// TIA Portal V19 export
FUNCTION "INTERLOCK" : Void   // FC8, LAD
{ S7_Optimized_Access := 'TRUE' }
// stored: SetENOAutomatically false
   VAR_TEMP   // added for the SCL form of the ladder/FBD networks
      _w1 : Bool;
      _w2 : Bool;
   END_VAR
BEGIN

REGION Network 1: RO-1 RESET INTERLOCK
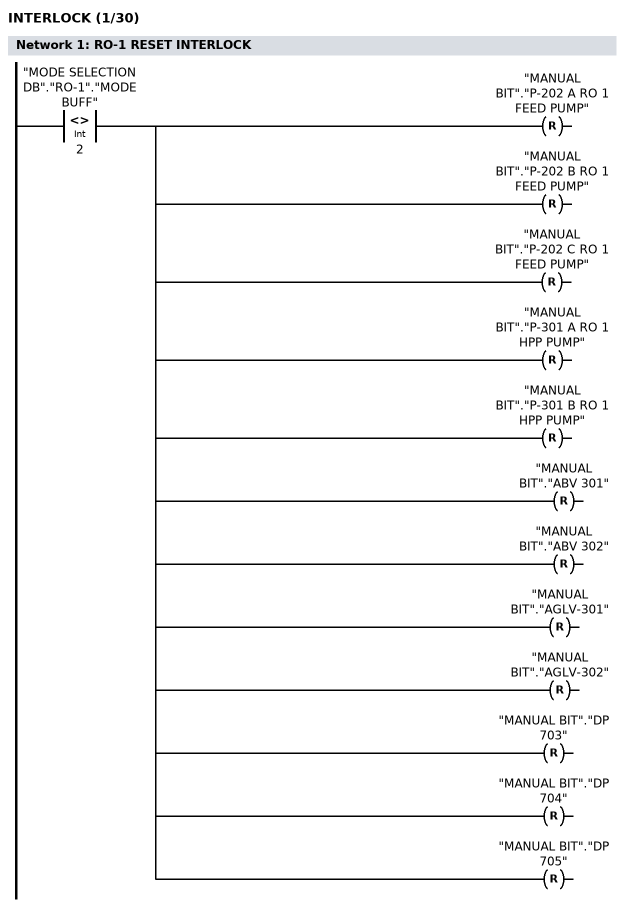
   RUNG wire#powerrail
      { S7_Templates := "SrcType := Int" } NE_Contact(in1 := "MODE SELECTION DB"."RO-1"."MODE BUFF", in2 := 2)
      wire#w1
      R_Coil( "MANUAL BIT"."P-202 A RO 1 FEED PUMP" )
   END_RUNG
   RUNG wire#w1
      R_Coil( "MANUAL BIT"."P-202 B RO 1 FEED PUMP" )
   END_RUNG
   RUNG wire#w1
      R_Coil( "MANUAL BIT"."P-202 C RO 1 FEED PUMP" )
   END_RUNG
   RUNG wire#w1
      R_Coil( "MANUAL BIT"."P-301 A RO 1 HPP PUMP" )
   END_RUNG
   RUNG wire#w1
      R_Coil( "MANUAL BIT"."P-301 B RO 1 HPP PUMP" )
   END_RUNG
   RUNG wire#w1
      R_Coil( "MANUAL BIT"."ABV 301" )
   END_RUNG
   RUNG wire#w1
      R_Coil( "MANUAL BIT"."ABV 302" )
   END_RUNG
   RUNG wire#w1
      R_Coil( "MANUAL BIT"."AGLV-301" )
   END_RUNG
   RUNG wire#w1
      R_Coil( "MANUAL BIT"."AGLV-302" )
   END_RUNG
   RUNG wire#w1
      R_Coil( "MANUAL BIT"."DP 703" )
   END_RUNG
   RUNG wire#w1
      R_Coil( "MANUAL BIT"."DP 704" )
   END_RUNG
   RUNG wire#w1
      R_Coil( "MANUAL BIT"."DP 705" )
   END_RUNG
   // the same network as SCL:
   IF "MODE SELECTION DB"."RO-1"."MODE BUFF" <> 2 THEN
       "MANUAL BIT"."P-202 A RO 1 FEED PUMP" := FALSE;
       "MANUAL BIT"."P-202 B RO 1 FEED PUMP" := FALSE;
       "MANUAL BIT"."P-202 C RO 1 FEED PUMP" := FALSE;
       "MANUAL BIT"."P-301 A RO 1 HPP PUMP" := FALSE;
       "MANUAL BIT"."P-301 B RO 1 HPP PUMP" := FALSE;
       "MANUAL BIT"."ABV 301" := FALSE;
       "MANUAL BIT"."ABV 302" := FALSE;
       "MANUAL BIT"."AGLV-301" := FALSE;
       "MANUAL BIT"."AGLV-302" := FALSE;
       "MANUAL BIT"."DP 703" := FALSE;
       "MANUAL BIT"."DP 704" := FALSE;
       "MANUAL BIT"."DP 705" := FALSE;
   END_IF;
END_REGION

REGION Network 2: RO-2 RESET INTERLOCK
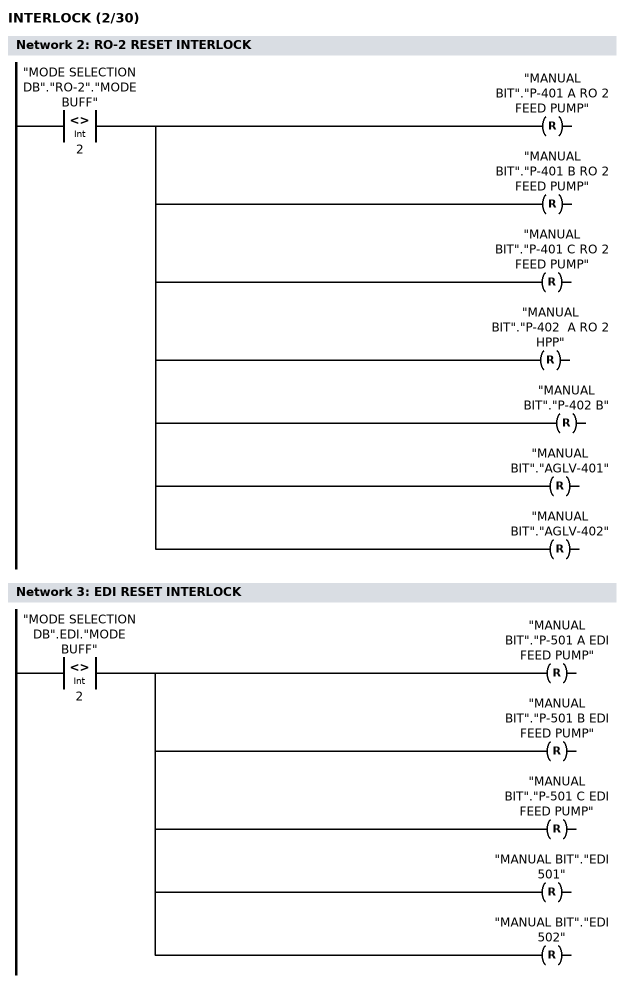
   RUNG wire#powerrail
      { S7_Templates := "SrcType := Int" } NE_Contact(in1 := "MODE SELECTION DB"."RO-2"."MODE BUFF", in2 := 2)
      wire#w1
      R_Coil( "MANUAL BIT"."P-401 A RO 2 FEED PUMP" )
   END_RUNG
   RUNG wire#w1
      R_Coil( "MANUAL BIT"."P-401 B RO 2 FEED PUMP" )
   END_RUNG
   RUNG wire#w1
      R_Coil( "MANUAL BIT"."P-401 C RO 2 FEED PUMP" )
   END_RUNG
   RUNG wire#w1
      R_Coil( "MANUAL BIT"."P-402  A RO 2 HPP" )
   END_RUNG
   RUNG wire#w1
      R_Coil( "MANUAL BIT"."P-402 B" )
   END_RUNG
   RUNG wire#w1
      R_Coil( "MANUAL BIT"."AGLV-401" )
   END_RUNG
   RUNG wire#w1
      R_Coil( "MANUAL BIT"."AGLV-402" )
   END_RUNG
   // the same network as SCL:
   IF "MODE SELECTION DB"."RO-2"."MODE BUFF" <> 2 THEN
       "MANUAL BIT"."P-401 A RO 2 FEED PUMP" := FALSE;
       "MANUAL BIT"."P-401 B RO 2 FEED PUMP" := FALSE;
       "MANUAL BIT"."P-401 C RO 2 FEED PUMP" := FALSE;
       "MANUAL BIT"."P-402  A RO 2 HPP" := FALSE;
       "MANUAL BIT"."P-402 B" := FALSE;
       "MANUAL BIT"."AGLV-401" := FALSE;
       "MANUAL BIT"."AGLV-402" := FALSE;
   END_IF;
END_REGION

REGION Network 3: EDI RESET INTERLOCK
   RUNG wire#powerrail
      { S7_Templates := "SrcType := Int" } NE_Contact(in1 := "MODE SELECTION DB".EDI."MODE BUFF", in2 := 2)
      wire#w1
      R_Coil( "MANUAL BIT"."P-501 A EDI FEED PUMP" )
   END_RUNG
   RUNG wire#w1
      R_Coil( "MANUAL BIT"."P-501 B EDI FEED PUMP" )
   END_RUNG
   RUNG wire#w1
      R_Coil( "MANUAL BIT"."P-501 C EDI FEED PUMP" )
   END_RUNG
   RUNG wire#w1
      R_Coil( "MANUAL BIT"."EDI 501" )
   END_RUNG
   RUNG wire#w1
      R_Coil( "MANUAL BIT"."EDI 502" )
   END_RUNG
   // the same network as SCL:
   IF "MODE SELECTION DB".EDI."MODE BUFF" <> 2 THEN
       "MANUAL BIT"."P-501 A EDI FEED PUMP" := FALSE;
       "MANUAL BIT"."P-501 B EDI FEED PUMP" := FALSE;
       "MANUAL BIT"."P-501 C EDI FEED PUMP" := FALSE;
       "MANUAL BIT"."EDI 501" := FALSE;
       "MANUAL BIT"."EDI 502" := FALSE;
   END_IF;
END_REGION

REGION Network 4: SELECTION PUMP INTERLOCK_
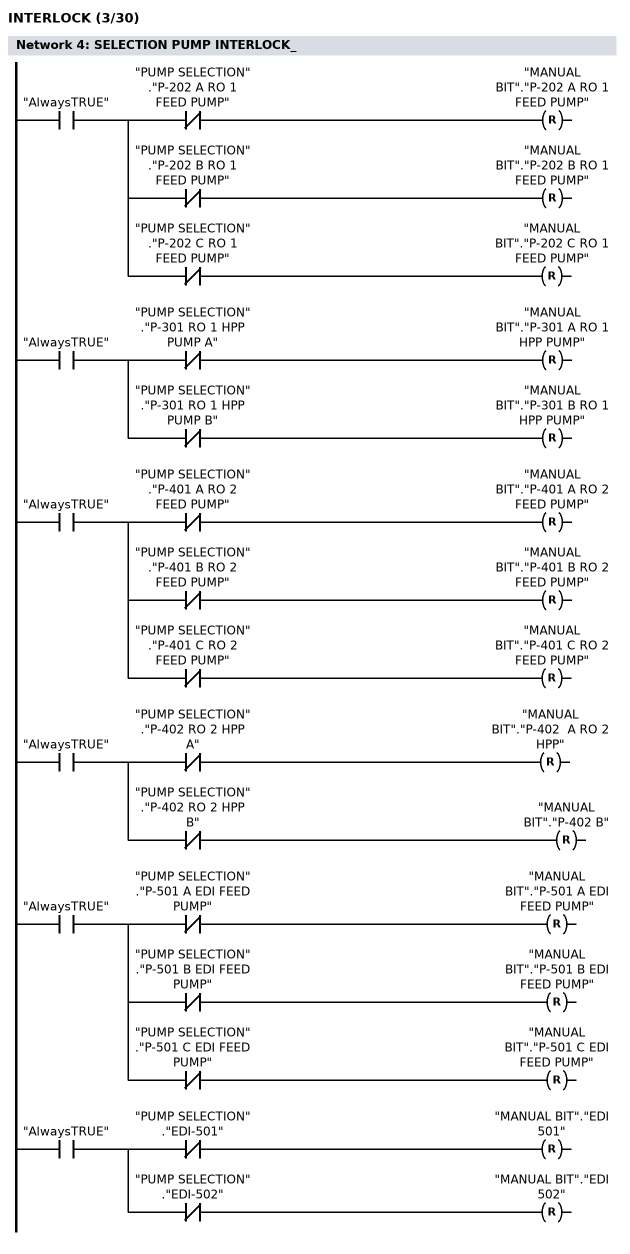
   RUNG wire#powerrail
      Contact( "AlwaysTRUE" )
      wire#w1
      I_Contact( "PUMP SELECTION"."P-202 A RO 1 FEED PUMP" )
      R_Coil( "MANUAL BIT"."P-202 A RO 1 FEED PUMP" )
   END_RUNG
   RUNG wire#w1
      I_Contact( "PUMP SELECTION"."P-202 B RO 1 FEED PUMP" )
      R_Coil( "MANUAL BIT"."P-202 B RO 1 FEED PUMP" )
   END_RUNG
   RUNG wire#w1
      I_Contact( "PUMP SELECTION"."P-202 C RO 1 FEED PUMP" )
      R_Coil( "MANUAL BIT"."P-202 C RO 1 FEED PUMP" )
   END_RUNG
   RUNG wire#powerrail
      Contact( "AlwaysTRUE" )
      wire#w2
      I_Contact( "PUMP SELECTION"."P-301 RO 1 HPP PUMP A" )
      R_Coil( "MANUAL BIT"."P-301 A RO 1 HPP PUMP" )
   END_RUNG
   RUNG wire#w2
      I_Contact( "PUMP SELECTION"."P-301 RO 1 HPP PUMP B" )
      R_Coil( "MANUAL BIT"."P-301 B RO 1 HPP PUMP" )
   END_RUNG
   RUNG wire#powerrail
      Contact( "AlwaysTRUE" )
      wire#w3
      I_Contact( "PUMP SELECTION"."P-401 A RO 2 FEED PUMP" )
      R_Coil( "MANUAL BIT"."P-401 A RO 2 FEED PUMP" )
   END_RUNG
   RUNG wire#w3
      I_Contact( "PUMP SELECTION"."P-401 B RO 2 FEED PUMP" )
      R_Coil( "MANUAL BIT"."P-401 B RO 2 FEED PUMP" )
   END_RUNG
   RUNG wire#w3
      I_Contact( "PUMP SELECTION"."P-401 C RO 2 FEED PUMP" )
      R_Coil( "MANUAL BIT"."P-401 C RO 2 FEED PUMP" )
   END_RUNG
   RUNG wire#powerrail
      Contact( "AlwaysTRUE" )
      wire#w4
      I_Contact( "PUMP SELECTION"."P-402 RO 2 HPP A" )
      R_Coil( "MANUAL BIT"."P-402  A RO 2 HPP" )
   END_RUNG
   RUNG wire#w4
      I_Contact( "PUMP SELECTION"."P-402 RO 2 HPP B" )
      R_Coil( "MANUAL BIT"."P-402 B" )
   END_RUNG
   RUNG wire#powerrail
      Contact( "AlwaysTRUE" )
      wire#w5
      I_Contact( "PUMP SELECTION"."P-501 A EDI FEED PUMP" )
      R_Coil( "MANUAL BIT"."P-501 A EDI FEED PUMP" )
   END_RUNG
   RUNG wire#w5
      I_Contact( "PUMP SELECTION"."P-501 B EDI FEED PUMP" )
      R_Coil( "MANUAL BIT"."P-501 B EDI FEED PUMP" )
   END_RUNG
   RUNG wire#w5
      I_Contact( "PUMP SELECTION"."P-501 C EDI FEED PUMP" )
      R_Coil( "MANUAL BIT"."P-501 C EDI FEED PUMP" )
   END_RUNG
   RUNG wire#powerrail
      Contact( "AlwaysTRUE" )
      wire#w6
      I_Contact( "PUMP SELECTION"."EDI-501" )
      R_Coil( "MANUAL BIT"."EDI 501" )
   END_RUNG
   RUNG wire#w6
      I_Contact( "PUMP SELECTION"."EDI-502" )
      R_Coil( "MANUAL BIT"."EDI 502" )
   END_RUNG
   // the same network as SCL:
   IF "AlwaysTRUE" AND NOT "PUMP SELECTION"."P-202 A RO 1 FEED PUMP" THEN
       "MANUAL BIT"."P-202 A RO 1 FEED PUMP" := FALSE;
   END_IF;
   IF "AlwaysTRUE" AND NOT "PUMP SELECTION"."P-202 B RO 1 FEED PUMP" THEN
       "MANUAL BIT"."P-202 B RO 1 FEED PUMP" := FALSE;
   END_IF;
   IF "AlwaysTRUE" AND NOT "PUMP SELECTION"."P-202 C RO 1 FEED PUMP" THEN
       "MANUAL BIT"."P-202 C RO 1 FEED PUMP" := FALSE;
   END_IF;
   IF "AlwaysTRUE" AND NOT "PUMP SELECTION"."P-301 RO 1 HPP PUMP A" THEN
       "MANUAL BIT"."P-301 A RO 1 HPP PUMP" := FALSE;
   END_IF;
   IF "AlwaysTRUE" AND NOT "PUMP SELECTION"."P-301 RO 1 HPP PUMP B" THEN
       "MANUAL BIT"."P-301 B RO 1 HPP PUMP" := FALSE;
   END_IF;
   IF "AlwaysTRUE" AND NOT "PUMP SELECTION"."P-401 A RO 2 FEED PUMP" THEN
       "MANUAL BIT"."P-401 A RO 2 FEED PUMP" := FALSE;
   END_IF;
   IF "AlwaysTRUE" AND NOT "PUMP SELECTION"."P-401 B RO 2 FEED PUMP" THEN
       "MANUAL BIT"."P-401 B RO 2 FEED PUMP" := FALSE;
   END_IF;
   IF "AlwaysTRUE" AND NOT "PUMP SELECTION"."P-401 C RO 2 FEED PUMP" THEN
       "MANUAL BIT"."P-401 C RO 2 FEED PUMP" := FALSE;
   END_IF;
   IF "AlwaysTRUE" AND NOT "PUMP SELECTION"."P-402 RO 2 HPP A" THEN
       "MANUAL BIT"."P-402  A RO 2 HPP" := FALSE;
   END_IF;
   IF "AlwaysTRUE" AND NOT "PUMP SELECTION"."P-402 RO 2 HPP B" THEN "MANUAL BIT"."P-402 B" := FALSE; END_IF;
   IF "AlwaysTRUE" AND NOT "PUMP SELECTION"."P-501 A EDI FEED PUMP" THEN
       "MANUAL BIT"."P-501 A EDI FEED PUMP" := FALSE;
   END_IF;
   IF "AlwaysTRUE" AND NOT "PUMP SELECTION"."P-501 B EDI FEED PUMP" THEN
       "MANUAL BIT"."P-501 B EDI FEED PUMP" := FALSE;
   END_IF;
   IF "AlwaysTRUE" AND NOT "PUMP SELECTION"."P-501 C EDI FEED PUMP" THEN
       "MANUAL BIT"."P-501 C EDI FEED PUMP" := FALSE;
   END_IF;
   IF "AlwaysTRUE" AND NOT "PUMP SELECTION"."EDI-501" THEN "MANUAL BIT"."EDI 501" := FALSE; END_IF;
   IF "AlwaysTRUE" AND NOT "PUMP SELECTION"."EDI-502" THEN "MANUAL BIT"."EDI 502" := FALSE; END_IF;
END_REGION

REGION Network 10: AUTO INTERLOCK FOR RO-1 ///////////////////////////////////////////////////////
END_REGION

REGION Network 11: CEB1 AND CEB2 SYSTEM IN RUNNING AFTER RO SYSTEM HOLD
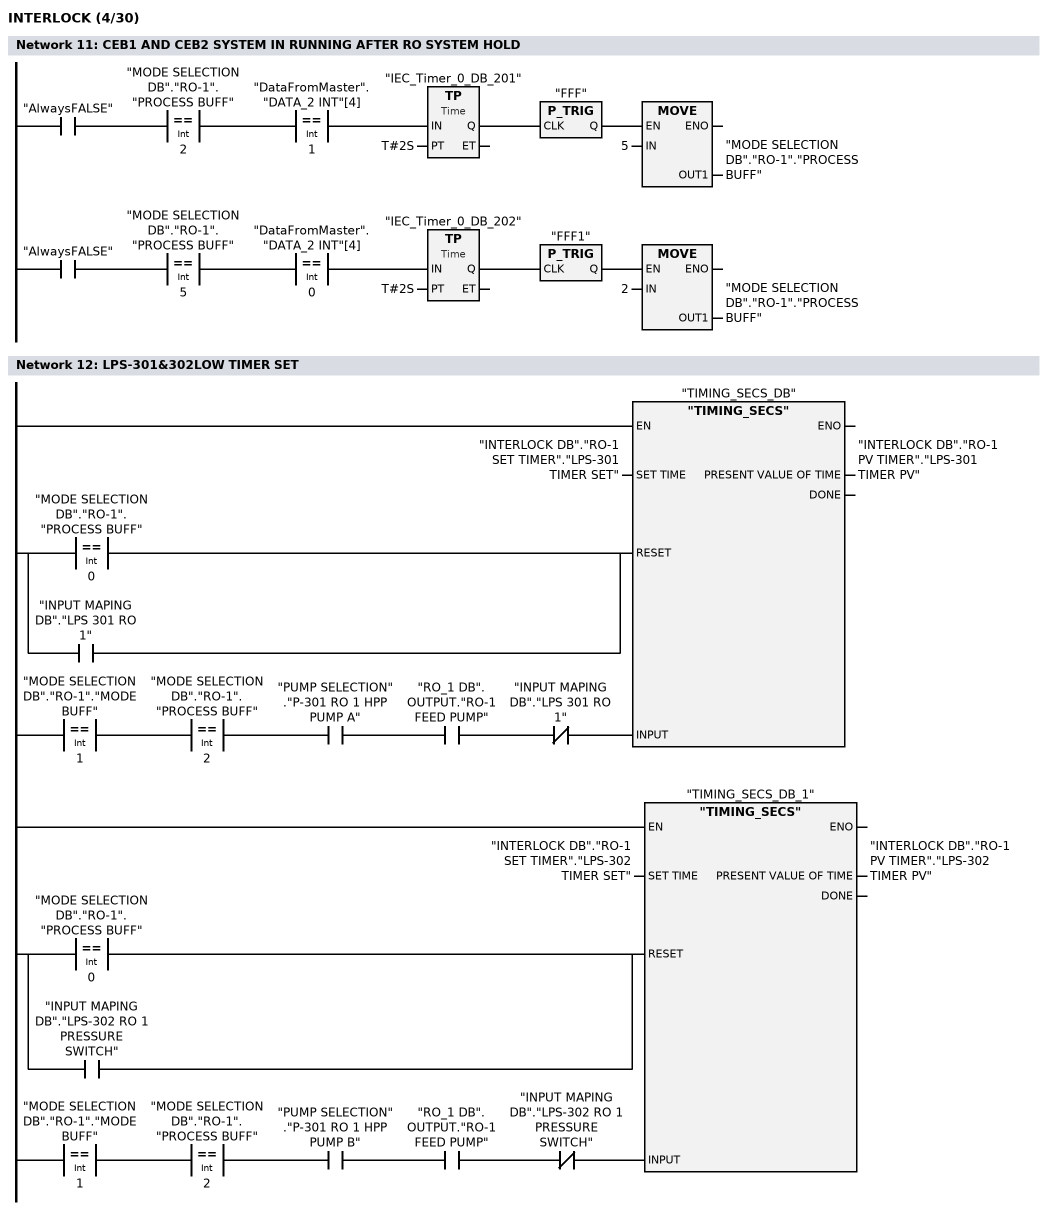
   RUNG wire#powerrail
      Contact( "AlwaysFALSE" )
      { S7_Templates := "SrcType := Int" } EQ_Contact(in1 := "MODE SELECTION DB"."RO-1"."PROCESS BUFF", in2 := 2)
      { S7_Templates := "SrcType := Int" } EQ_Contact(in1 := "DataFromMaster"."DATA_2 INT"[4], in2 := 1)
      { S7_Templates := "time_type := Time" } "IEC_Timer_0_DB_201".TP(pt := T#2S, et =>)
      P_Trig( "FFF" )
      Move(in := 5, out1 => "MODE SELECTION DB"."RO-1"."PROCESS BUFF")
   END_RUNG
   RUNG wire#powerrail
      Contact( "AlwaysFALSE" )
      { S7_Templates := "SrcType := Int" } EQ_Contact(in1 := "MODE SELECTION DB"."RO-1"."PROCESS BUFF", in2 := 5)
      { S7_Templates := "SrcType := Int" } EQ_Contact(in1 := "DataFromMaster"."DATA_2 INT"[4], in2 := 0)
      { S7_Templates := "time_type := Time" } "IEC_Timer_0_DB_202".TP(pt := T#2S, et =>)
      P_Trig( "FFF1" )
      Move(in := 2, out1 => "MODE SELECTION DB"."RO-1"."PROCESS BUFF")
   END_RUNG
   // the same network as SCL:
   "IEC_Timer_0_DB_201".TP(IN := "AlwaysFALSE" AND ("MODE SELECTION DB"."RO-1"."PROCESS BUFF" = 2) AND ("DataFromMaster"."DATA_2 INT"[4] = 1),
                           PT := T#2S);
   #_w1 := "IEC_Timer_0_DB_201".Q AND NOT "FFF";   // rising edge
   "FFF" := "IEC_Timer_0_DB_201".Q;
   IF #_w1 THEN "MODE SELECTION DB"."RO-1"."PROCESS BUFF" := 5; END_IF;
   "IEC_Timer_0_DB_202".TP(IN := "AlwaysFALSE" AND ("MODE SELECTION DB"."RO-1"."PROCESS BUFF" = 5) AND ("DataFromMaster"."DATA_2 INT"[4] = 0),
                           PT := T#2S);
   #_w2 := "IEC_Timer_0_DB_202".Q AND NOT "FFF1";   // rising edge
   "FFF1" := "IEC_Timer_0_DB_202".Q;
   IF #_w2 THEN "MODE SELECTION DB"."RO-1"."PROCESS BUFF" := 2; END_IF;
END_REGION

REGION Network 12: LPS-301&302LOW TIMER SET
   RUNG wire#powerrail
      "TIMING_SECS_DB"(RESET := wire#w1, INPUT := wire#w2, "SET TIME" := "INTERLOCK DB"."RO-1 SET TIMER"."LPS-301 TIMER SET", "PRESENT VALUE OF TIME" => "INTERLOCK DB"."RO-1 PV TIMER"."LPS-301 TIMER PV", DONE =>)
   END_RUNG
   RUNG wire#powerrail
      { S7_Templates := "SrcType := Int" } EQ_Contact(in1 := "MODE SELECTION DB"."RO-1"."PROCESS BUFF", in2 := 0)
   END_RUNG wire#w1
   RUNG wire#powerrail
      Contact( "INPUT MAPING DB"."LPS 301 RO 1" )
   END_RUNG wire#w1
   RUNG wire#powerrail
      { S7_Templates := "SrcType := Int" } EQ_Contact(in1 := "MODE SELECTION DB"."RO-1"."MODE BUFF", in2 := 1)
      { S7_Templates := "SrcType := Int" } EQ_Contact(in1 := "MODE SELECTION DB"."RO-1"."PROCESS BUFF", in2 := 2)
      Contact( "PUMP SELECTION"."P-301 RO 1 HPP PUMP A" )
      Contact( "RO_1 DB".OUTPUT."RO-1 FEED PUMP" )
      I_Contact( "INPUT MAPING DB"."LPS 301 RO 1" )
   END_RUNG wire#w2
   RUNG wire#powerrail
      "TIMING_SECS_DB_1"(RESET := wire#w3, INPUT := wire#w4, "SET TIME" := "INTERLOCK DB"."RO-1 SET TIMER"."LPS-302 TIMER SET", "PRESENT VALUE OF TIME" => "INTERLOCK DB"."RO-1 PV TIMER"."LPS-302 TIMER PV", DONE =>)
   END_RUNG
   RUNG wire#powerrail
      { S7_Templates := "SrcType := Int" } EQ_Contact(in1 := "MODE SELECTION DB"."RO-1"."PROCESS BUFF", in2 := 0)
   END_RUNG wire#w3
   RUNG wire#powerrail
      Contact( "INPUT MAPING DB"."LPS-302 RO 1 PRESSURE SWITCH" )
   END_RUNG wire#w3
   RUNG wire#powerrail
      { S7_Templates := "SrcType := Int" } EQ_Contact(in1 := "MODE SELECTION DB"."RO-1"."MODE BUFF", in2 := 1)
      { S7_Templates := "SrcType := Int" } EQ_Contact(in1 := "MODE SELECTION DB"."RO-1"."PROCESS BUFF", in2 := 2)
      Contact( "PUMP SELECTION"."P-301 RO 1 HPP PUMP B" )
      Contact( "RO_1 DB".OUTPUT."RO-1 FEED PUMP" )
      I_Contact( "INPUT MAPING DB"."LPS-302 RO 1 PRESSURE SWITCH" )
   END_RUNG wire#w4
   // the same network as SCL:
   "TIMING_SECS_DB"("SET TIME" := "INTERLOCK DB"."RO-1 SET TIMER"."LPS-301 TIMER SET",   // "TIMING_SECS"
                    RESET := ("MODE SELECTION DB"."RO-1"."PROCESS BUFF" = 0) OR "INPUT MAPING DB"."LPS 301 RO 1",
                    INPUT := ("MODE SELECTION DB"."RO-1"."MODE BUFF" = 1) AND ("MODE SELECTION DB"."RO-1"."PROCESS BUFF" = 2) AND "PUMP SELECTION"."P-301 RO 1 HPP PUMP A" AND "RO_1 DB".OUTPUT."RO-1 FEED PUMP" AND NOT "INPUT MAPING DB"."LPS 301 RO 1",
                    "PRESENT VALUE OF TIME" => "INTERLOCK DB"."RO-1 PV TIMER"."LPS-301 TIMER PV");
   "TIMING_SECS_DB_1"("SET TIME" := "INTERLOCK DB"."RO-1 SET TIMER"."LPS-302 TIMER SET",   // "TIMING_SECS"
                      RESET := ("MODE SELECTION DB"."RO-1"."PROCESS BUFF" = 0) OR "INPUT MAPING DB"."LPS-302 RO 1 PRESSURE SWITCH",
                      INPUT := ("MODE SELECTION DB"."RO-1"."MODE BUFF" = 1) AND ("MODE SELECTION DB"."RO-1"."PROCESS BUFF" = 2) AND "PUMP SELECTION"."P-301 RO 1 HPP PUMP B" AND "RO_1 DB".OUTPUT."RO-1 FEED PUMP" AND NOT "INPUT MAPING DB"."LPS-302 RO 1 PRESSURE SWITCH",
                      "PRESENT VALUE OF TIME" => "INTERLOCK DB"."RO-1 PV TIMER"."LPS-302 TIMER PV");
END_REGION

REGION Network 13: HPS-301 &302
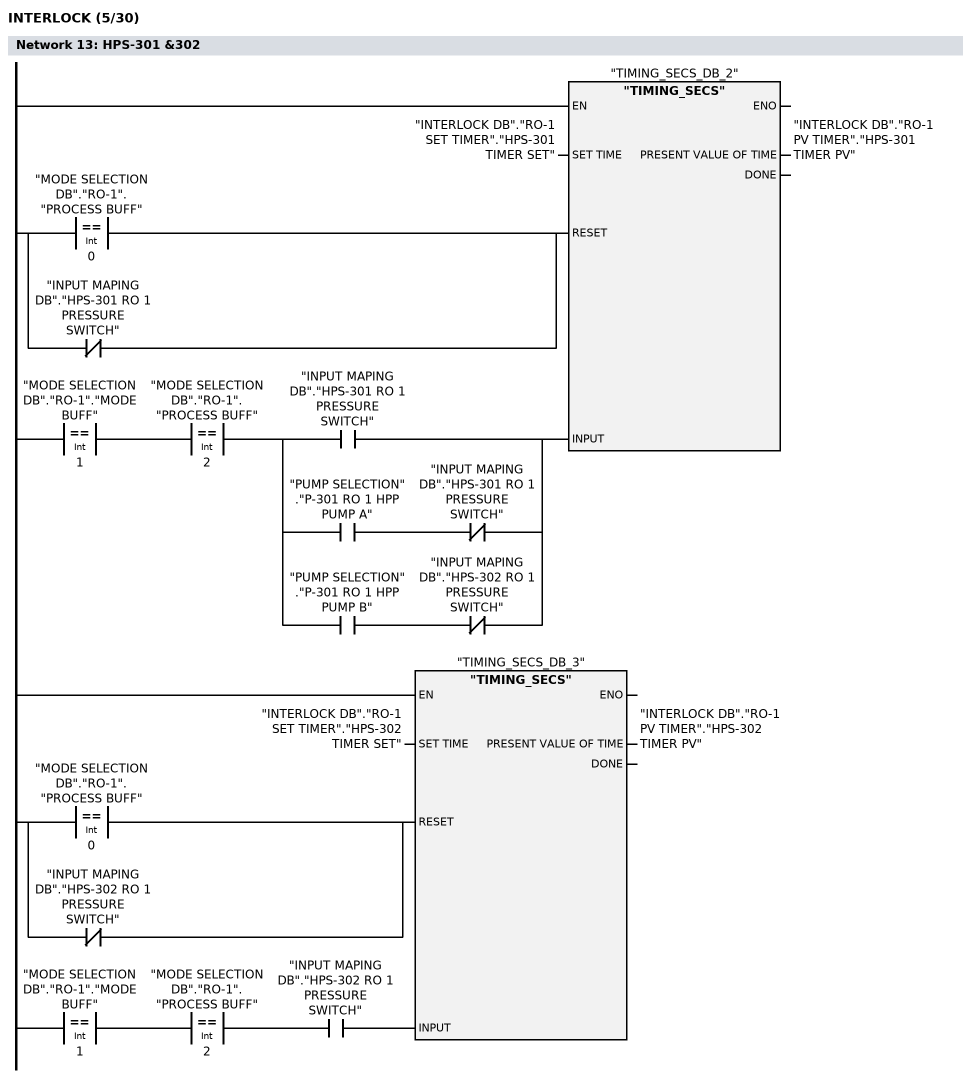
   RUNG wire#powerrail
      "TIMING_SECS_DB_2"(RESET := wire#w1, INPUT := wire#w3, "SET TIME" := "INTERLOCK DB"."RO-1 SET TIMER"."HPS-301 TIMER SET", "PRESENT VALUE OF TIME" => "INTERLOCK DB"."RO-1 PV TIMER"."HPS-301 TIMER PV", DONE =>)
   END_RUNG
   RUNG wire#powerrail
      { S7_Templates := "SrcType := Int" } EQ_Contact(in1 := "MODE SELECTION DB"."RO-1"."PROCESS BUFF", in2 := 0)
   END_RUNG wire#w1
   RUNG wire#powerrail
      I_Contact( "INPUT MAPING DB"."HPS-301 RO 1 PRESSURE SWITCH" )
   END_RUNG wire#w1
   RUNG wire#powerrail
      { S7_Templates := "SrcType := Int" } EQ_Contact(in1 := "MODE SELECTION DB"."RO-1"."MODE BUFF", in2 := 1)
      { S7_Templates := "SrcType := Int" } EQ_Contact(in1 := "MODE SELECTION DB"."RO-1"."PROCESS BUFF", in2 := 2)
      wire#w2
      Contact( "INPUT MAPING DB"."HPS-301 RO 1 PRESSURE SWITCH" )
   END_RUNG wire#w3
   RUNG wire#w2
      Contact( "PUMP SELECTION"."P-301 RO 1 HPP PUMP A" )
      I_Contact( "INPUT MAPING DB"."HPS-301 RO 1 PRESSURE SWITCH" )
   END_RUNG wire#w3
   RUNG wire#w2
      Contact( "PUMP SELECTION"."P-301 RO 1 HPP PUMP B" )
      I_Contact( "INPUT MAPING DB"."HPS-302 RO 1 PRESSURE SWITCH" )
   END_RUNG wire#w3
   RUNG wire#powerrail
      "TIMING_SECS_DB_3"(RESET := wire#w4, INPUT := wire#w5, "SET TIME" := "INTERLOCK DB"."RO-1 SET TIMER"."HPS-302 TIMER SET", "PRESENT VALUE OF TIME" => "INTERLOCK DB"."RO-1 PV TIMER"."HPS-302 TIMER PV", DONE =>)
   END_RUNG
   RUNG wire#powerrail
      { S7_Templates := "SrcType := Int" } EQ_Contact(in1 := "MODE SELECTION DB"."RO-1"."PROCESS BUFF", in2 := 0)
   END_RUNG wire#w4
   RUNG wire#powerrail
      I_Contact( "INPUT MAPING DB"."HPS-302 RO 1 PRESSURE SWITCH" )
   END_RUNG wire#w4
   RUNG wire#powerrail
      { S7_Templates := "SrcType := Int" } EQ_Contact(in1 := "MODE SELECTION DB"."RO-1"."MODE BUFF", in2 := 1)
      { S7_Templates := "SrcType := Int" } EQ_Contact(in1 := "MODE SELECTION DB"."RO-1"."PROCESS BUFF", in2 := 2)
      Contact( "INPUT MAPING DB"."HPS-302 RO 1 PRESSURE SWITCH" )
   END_RUNG wire#w5
   // the same network as SCL:
   "TIMING_SECS_DB_2"("SET TIME" := "INTERLOCK DB"."RO-1 SET TIMER"."HPS-301 TIMER SET",   // "TIMING_SECS"
                      RESET := ("MODE SELECTION DB"."RO-1"."PROCESS BUFF" = 0) OR NOT "INPUT MAPING DB"."HPS-301 RO 1 PRESSURE SWITCH",
                      INPUT := ("MODE SELECTION DB"."RO-1"."MODE BUFF" = 1) AND ("MODE SELECTION DB"."RO-1"."PROCESS BUFF" = 2) AND ("INPUT MAPING DB"."HPS-301 RO 1 PRESSURE SWITCH" OR ("PUMP SELECTION"."P-301 RO 1 HPP PUMP A" AND NOT "INPUT MAPING DB"."HPS-301 RO 1 PRESSURE SWITCH") OR ("PUMP SELECTION"."P-301 RO 1 HPP PUMP B" AND NOT "INPUT MAPING DB"."HPS-302 RO 1 PRESSURE SWITCH")),
                      "PRESENT VALUE OF TIME" => "INTERLOCK DB"."RO-1 PV TIMER"."HPS-301 TIMER PV");
   "TIMING_SECS_DB_3"("SET TIME" := "INTERLOCK DB"."RO-1 SET TIMER"."HPS-302 TIMER SET",   // "TIMING_SECS"
                      RESET := ("MODE SELECTION DB"."RO-1"."PROCESS BUFF" = 0) OR NOT "INPUT MAPING DB"."HPS-302 RO 1 PRESSURE SWITCH",
                      INPUT := ("MODE SELECTION DB"."RO-1"."MODE BUFF" = 1) AND ("MODE SELECTION DB"."RO-1"."PROCESS BUFF" = 2) AND "INPUT MAPING DB"."HPS-302 RO 1 PRESSURE SWITCH",
                      "PRESENT VALUE OF TIME" => "INTERLOCK DB"."RO-1 PV TIMER"."HPS-302 TIMER PV");
END_REGION

REGION Network 14: pH-301 HIGH/ LOW
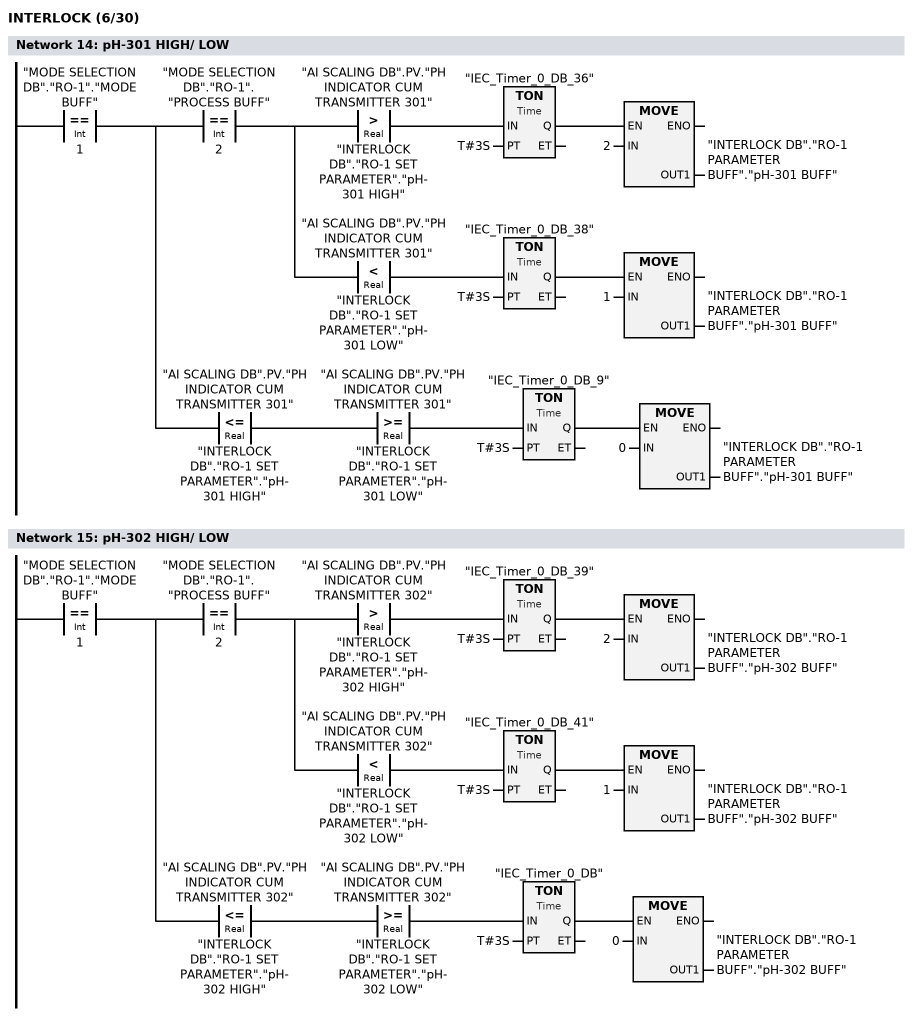
   RUNG wire#powerrail
      { S7_Templates := "SrcType := Int" } EQ_Contact(in1 := "MODE SELECTION DB"."RO-1"."MODE BUFF", in2 := 1)
      wire#w1
      { S7_Templates := "SrcType := Int" } EQ_Contact(in1 := "MODE SELECTION DB"."RO-1"."PROCESS BUFF", in2 := 2)
      wire#w2
      { S7_Templates := "SrcType := Real" } GT_Contact(in1 := "AI SCALING DB".PV."PH INDICATOR CUM TRANSMITTER 301", in2 := "INTERLOCK DB"."RO-1 SET PARAMETER"."pH-301 HIGH")
      { S7_Templates := "time_type := Time" } "IEC_Timer_0_DB_36".TON(pt := T#3S, et =>)
      Move(in := 2, out1 => "INTERLOCK DB"."RO-1 PARAMETER BUFF"."pH-301 BUFF")
   END_RUNG
   RUNG wire#w2
      { S7_Templates := "SrcType := Real" } LT_Contact(in1 := "AI SCALING DB".PV."PH INDICATOR CUM TRANSMITTER 301", in2 := "INTERLOCK DB"."RO-1 SET PARAMETER"."pH-301 LOW")
      { S7_Templates := "time_type := Time" } "IEC_Timer_0_DB_38".TON(pt := T#3S, et =>)
      Move(in := 1, out1 => "INTERLOCK DB"."RO-1 PARAMETER BUFF"."pH-301 BUFF")
   END_RUNG
   RUNG wire#w1
      { S7_Templates := "SrcType := Real" } LE_Contact(in1 := "AI SCALING DB".PV."PH INDICATOR CUM TRANSMITTER 301", in2 := "INTERLOCK DB"."RO-1 SET PARAMETER"."pH-301 HIGH")
      { S7_Templates := "SrcType := Real" } GE_Contact(in1 := "AI SCALING DB".PV."PH INDICATOR CUM TRANSMITTER 301", in2 := "INTERLOCK DB"."RO-1 SET PARAMETER"."pH-301 LOW")
      { S7_Templates := "time_type := Time" } "IEC_Timer_0_DB_9".TON(pt := T#3S, et =>)
      Move(in := 0, out1 => "INTERLOCK DB"."RO-1 PARAMETER BUFF"."pH-301 BUFF")
   END_RUNG
   // the same network as SCL:
   #_w1 := "MODE SELECTION DB"."RO-1"."MODE BUFF" = 1;
   #_w2 := #_w1 AND ("MODE SELECTION DB"."RO-1"."PROCESS BUFF" = 2);
   "IEC_Timer_0_DB_36".TON(IN := #_w2 AND ("AI SCALING DB".PV."PH INDICATOR CUM TRANSMITTER 301" > "INTERLOCK DB"."RO-1 SET PARAMETER"."pH-301 HIGH"),
                           PT := T#3S);
   IF "IEC_Timer_0_DB_36".Q THEN "INTERLOCK DB"."RO-1 PARAMETER BUFF"."pH-301 BUFF" := 2; END_IF;
   "IEC_Timer_0_DB_38".TON(IN := #_w2 AND ("AI SCALING DB".PV."PH INDICATOR CUM TRANSMITTER 301" < "INTERLOCK DB"."RO-1 SET PARAMETER"."pH-301 LOW"),
                           PT := T#3S);
   IF "IEC_Timer_0_DB_38".Q THEN "INTERLOCK DB"."RO-1 PARAMETER BUFF"."pH-301 BUFF" := 1; END_IF;
   "IEC_Timer_0_DB_9".TON(IN := #_w1 AND ("AI SCALING DB".PV."PH INDICATOR CUM TRANSMITTER 301" <= "INTERLOCK DB"."RO-1 SET PARAMETER"."pH-301 HIGH") AND ("AI SCALING DB".PV."PH INDICATOR CUM TRANSMITTER 301" >= "INTERLOCK DB"."RO-1 SET PARAMETER"."pH-301 LOW"),
                          PT := T#3S);
   IF "IEC_Timer_0_DB_9".Q THEN "INTERLOCK DB"."RO-1 PARAMETER BUFF"."pH-301 BUFF" := 0; END_IF;
END_REGION

REGION Network 15: pH-302 HIGH/ LOW
   RUNG wire#powerrail
      { S7_Templates := "SrcType := Int" } EQ_Contact(in1 := "MODE SELECTION DB"."RO-1"."MODE BUFF", in2 := 1)
      wire#w1
      { S7_Templates := "SrcType := Int" } EQ_Contact(in1 := "MODE SELECTION DB"."RO-1"."PROCESS BUFF", in2 := 2)
      wire#w2
      { S7_Templates := "SrcType := Real" } GT_Contact(in1 := "AI SCALING DB".PV."PH INDICATOR CUM TRANSMITTER 302", in2 := "INTERLOCK DB"."RO-1 SET PARAMETER"."pH-302 HIGH")
      { S7_Templates := "time_type := Time" } "IEC_Timer_0_DB_39".TON(pt := T#3S, et =>)
      Move(in := 2, out1 => "INTERLOCK DB"."RO-1 PARAMETER BUFF"."pH-302 BUFF")
   END_RUNG
   RUNG wire#w2
      { S7_Templates := "SrcType := Real" } LT_Contact(in1 := "AI SCALING DB".PV."PH INDICATOR CUM TRANSMITTER 302", in2 := "INTERLOCK DB"."RO-1 SET PARAMETER"."pH-302 LOW")
      { S7_Templates := "time_type := Time" } "IEC_Timer_0_DB_41".TON(pt := T#3S, et =>)
      Move(in := 1, out1 => "INTERLOCK DB"."RO-1 PARAMETER BUFF"."pH-302 BUFF")
   END_RUNG
   RUNG wire#w1
      { S7_Templates := "SrcType := Real" } LE_Contact(in1 := "AI SCALING DB".PV."PH INDICATOR CUM TRANSMITTER 302", in2 := "INTERLOCK DB"."RO-1 SET PARAMETER"."pH-302 HIGH")
      { S7_Templates := "SrcType := Real" } GE_Contact(in1 := "AI SCALING DB".PV."PH INDICATOR CUM TRANSMITTER 302", in2 := "INTERLOCK DB"."RO-1 SET PARAMETER"."pH-302 LOW")
      { S7_Templates := "time_type := Time" } "IEC_Timer_0_DB".TON(pt := T#3S, et =>)
      Move(in := 0, out1 => "INTERLOCK DB"."RO-1 PARAMETER BUFF"."pH-302 BUFF")
   END_RUNG
   // the same network as SCL:
   #_w1 := "MODE SELECTION DB"."RO-1"."MODE BUFF" = 1;
   #_w2 := #_w1 AND ("MODE SELECTION DB"."RO-1"."PROCESS BUFF" = 2);
   "IEC_Timer_0_DB_39".TON(IN := #_w2 AND ("AI SCALING DB".PV."PH INDICATOR CUM TRANSMITTER 302" > "INTERLOCK DB"."RO-1 SET PARAMETER"."pH-302 HIGH"),
                           PT := T#3S);
   IF "IEC_Timer_0_DB_39".Q THEN "INTERLOCK DB"."RO-1 PARAMETER BUFF"."pH-302 BUFF" := 2; END_IF;
   "IEC_Timer_0_DB_41".TON(IN := #_w2 AND ("AI SCALING DB".PV."PH INDICATOR CUM TRANSMITTER 302" < "INTERLOCK DB"."RO-1 SET PARAMETER"."pH-302 LOW"),
                           PT := T#3S);
   IF "IEC_Timer_0_DB_41".Q THEN "INTERLOCK DB"."RO-1 PARAMETER BUFF"."pH-302 BUFF" := 1; END_IF;
   "IEC_Timer_0_DB".TON(IN := #_w1 AND ("AI SCALING DB".PV."PH INDICATOR CUM TRANSMITTER 302" <= "INTERLOCK DB"."RO-1 SET PARAMETER"."pH-302 HIGH") AND ("AI SCALING DB".PV."PH INDICATOR CUM TRANSMITTER 302" >= "INTERLOCK DB"."RO-1 SET PARAMETER"."pH-302 LOW"),
                        PT := T#3S);
   IF "IEC_Timer_0_DB".Q THEN "INTERLOCK DB"."RO-1 PARAMETER BUFF"."pH-302 BUFF" := 0; END_IF;
END_REGION

REGION Network 16: CT-301 HIGH
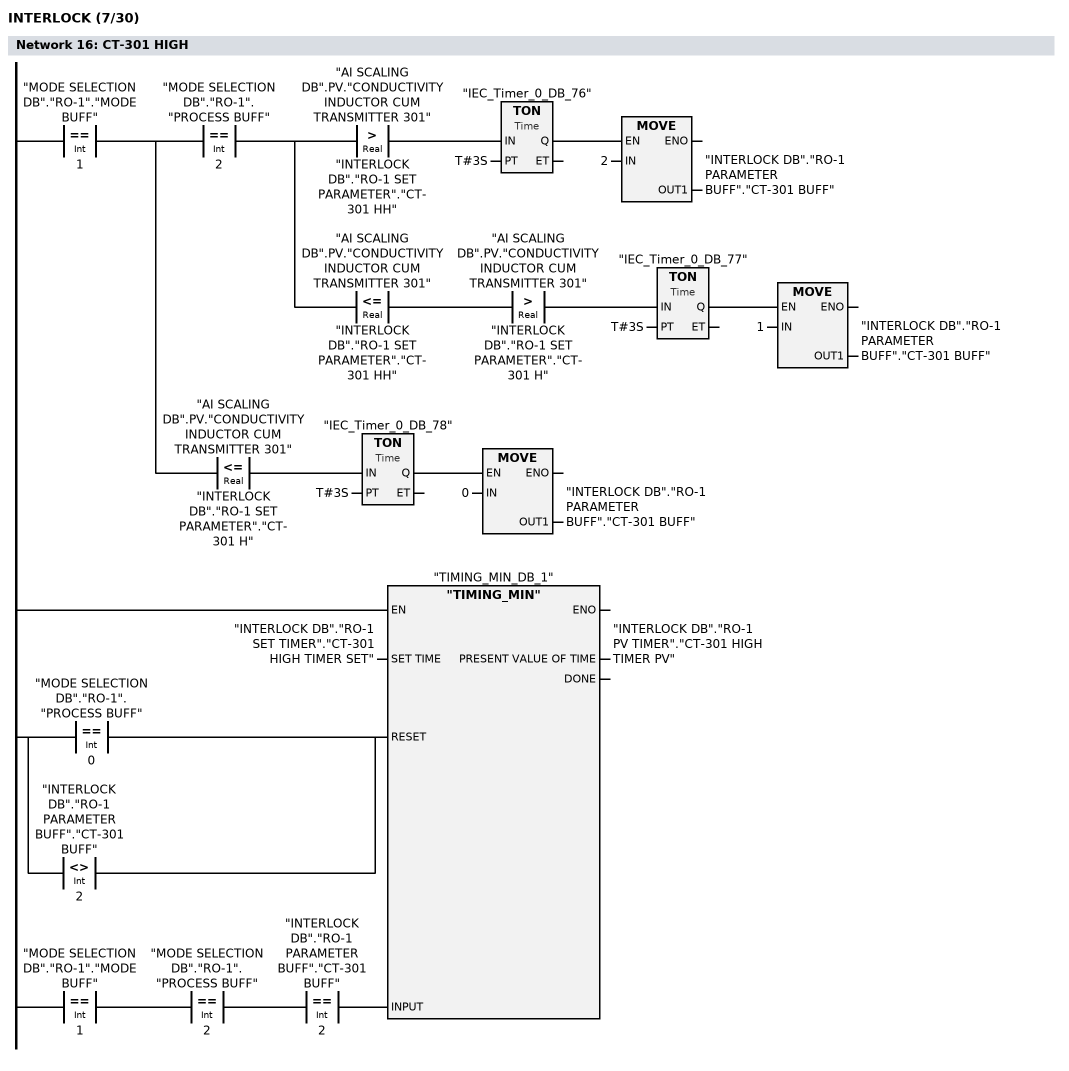
   RUNG wire#powerrail
      { S7_Templates := "SrcType := Int" } EQ_Contact(in1 := "MODE SELECTION DB"."RO-1"."MODE BUFF", in2 := 1)
      wire#w1
      { S7_Templates := "SrcType := Int" } EQ_Contact(in1 := "MODE SELECTION DB"."RO-1"."PROCESS BUFF", in2 := 2)
      wire#w2
      { S7_Templates := "SrcType := Real" } GT_Contact(in1 := "AI SCALING DB".PV."CONDUCTIVITY INDUCTOR CUM TRANSMITTER 301", in2 := "INTERLOCK DB"."RO-1 SET PARAMETER"."CT-301 HH")
      { S7_Templates := "time_type := Time" } "IEC_Timer_0_DB_76".TON(pt := T#3S, et =>)
      Move(in := 2, out1 => "INTERLOCK DB"."RO-1 PARAMETER BUFF"."CT-301 BUFF")
   END_RUNG
   RUNG wire#w2
      { S7_Templates := "SrcType := Real" } LE_Contact(in1 := "AI SCALING DB".PV."CONDUCTIVITY INDUCTOR CUM TRANSMITTER 301", in2 := "INTERLOCK DB"."RO-1 SET PARAMETER"."CT-301 HH")
      { S7_Templates := "SrcType := Real" } GT_Contact(in1 := "AI SCALING DB".PV."CONDUCTIVITY INDUCTOR CUM TRANSMITTER 301", in2 := "INTERLOCK DB"."RO-1 SET PARAMETER"."CT-301 H")
      { S7_Templates := "time_type := Time" } "IEC_Timer_0_DB_77".TON(pt := T#3S, et =>)
      Move(in := 1, out1 => "INTERLOCK DB"."RO-1 PARAMETER BUFF"."CT-301 BUFF")
   END_RUNG
   RUNG wire#w1
      { S7_Templates := "SrcType := Real" } LE_Contact(in1 := "AI SCALING DB".PV."CONDUCTIVITY INDUCTOR CUM TRANSMITTER 301", in2 := "INTERLOCK DB"."RO-1 SET PARAMETER"."CT-301 H")
      { S7_Templates := "time_type := Time" } "IEC_Timer_0_DB_78".TON(pt := T#3S, et =>)
      Move(in := 0, out1 => "INTERLOCK DB"."RO-1 PARAMETER BUFF"."CT-301 BUFF")
   END_RUNG
   RUNG wire#powerrail
      "TIMING_MIN_DB_1"(RESET := wire#w3, INPUT := wire#w4, "SET TIME" := "INTERLOCK DB"."RO-1 SET TIMER"."CT-301 HIGH TIMER SET", "PRESENT VALUE OF TIME" => "INTERLOCK DB"."RO-1 PV TIMER"."CT-301 HIGH TIMER PV", DONE =>)
   END_RUNG
   RUNG wire#powerrail
      { S7_Templates := "SrcType := Int" } EQ_Contact(in1 := "MODE SELECTION DB"."RO-1"."PROCESS BUFF", in2 := 0)
   END_RUNG wire#w3
   RUNG wire#powerrail
      { S7_Templates := "SrcType := Int" } NE_Contact(in1 := "INTERLOCK DB"."RO-1 PARAMETER BUFF"."CT-301 BUFF", in2 := 2)
   END_RUNG wire#w3
   RUNG wire#powerrail
      { S7_Templates := "SrcType := Int" } EQ_Contact(in1 := "MODE SELECTION DB"."RO-1"."MODE BUFF", in2 := 1)
      { S7_Templates := "SrcType := Int" } EQ_Contact(in1 := "MODE SELECTION DB"."RO-1"."PROCESS BUFF", in2 := 2)
      { S7_Templates := "SrcType := Int" } EQ_Contact(in1 := "INTERLOCK DB"."RO-1 PARAMETER BUFF"."CT-301 BUFF", in2 := 2)
   END_RUNG wire#w4
   // the same network as SCL:
   #_w1 := "MODE SELECTION DB"."RO-1"."MODE BUFF" = 1;
   #_w2 := #_w1 AND ("MODE SELECTION DB"."RO-1"."PROCESS BUFF" = 2);
   "IEC_Timer_0_DB_76".TON(IN := #_w2 AND ("AI SCALING DB".PV."CONDUCTIVITY INDUCTOR CUM TRANSMITTER 301" > "INTERLOCK DB"."RO-1 SET PARAMETER"."CT-301 HH"),
                           PT := T#3S);
   IF "IEC_Timer_0_DB_76".Q THEN "INTERLOCK DB"."RO-1 PARAMETER BUFF"."CT-301 BUFF" := 2; END_IF;
   "IEC_Timer_0_DB_77".TON(IN := #_w2 AND ("AI SCALING DB".PV."CONDUCTIVITY INDUCTOR CUM TRANSMITTER 301" <= "INTERLOCK DB"."RO-1 SET PARAMETER"."CT-301 HH") AND ("AI SCALING DB".PV."CONDUCTIVITY INDUCTOR CUM TRANSMITTER 301" > "INTERLOCK DB"."RO-1 SET PARAMETER"."CT-301 H"),
                           PT := T#3S);
   IF "IEC_Timer_0_DB_77".Q THEN "INTERLOCK DB"."RO-1 PARAMETER BUFF"."CT-301 BUFF" := 1; END_IF;
   "IEC_Timer_0_DB_78".TON(IN := #_w1 AND ("AI SCALING DB".PV."CONDUCTIVITY INDUCTOR CUM TRANSMITTER 301" <= "INTERLOCK DB"."RO-1 SET PARAMETER"."CT-301 H"),
                           PT := T#3S);
   IF "IEC_Timer_0_DB_78".Q THEN "INTERLOCK DB"."RO-1 PARAMETER BUFF"."CT-301 BUFF" := 0; END_IF;
   "TIMING_MIN_DB_1"("SET TIME" := "INTERLOCK DB"."RO-1 SET TIMER"."CT-301 HIGH TIMER SET",   // "TIMING_MIN"
                     RESET := ("MODE SELECTION DB"."RO-1"."PROCESS BUFF" = 0) OR ("INTERLOCK DB"."RO-1 PARAMETER BUFF"."CT-301 BUFF" <> 2),
                     INPUT := ("MODE SELECTION DB"."RO-1"."MODE BUFF" = 1) AND ("MODE SELECTION DB"."RO-1"."PROCESS BUFF" = 2) AND ("INTERLOCK DB"."RO-1 PARAMETER BUFF"."CT-301 BUFF" = 2),
                     "PRESENT VALUE OF TIME" => "INTERLOCK DB"."RO-1 PV TIMER"."CT-301 HIGH TIMER PV");
END_REGION

REGION Network 17: CT-302 HIGH
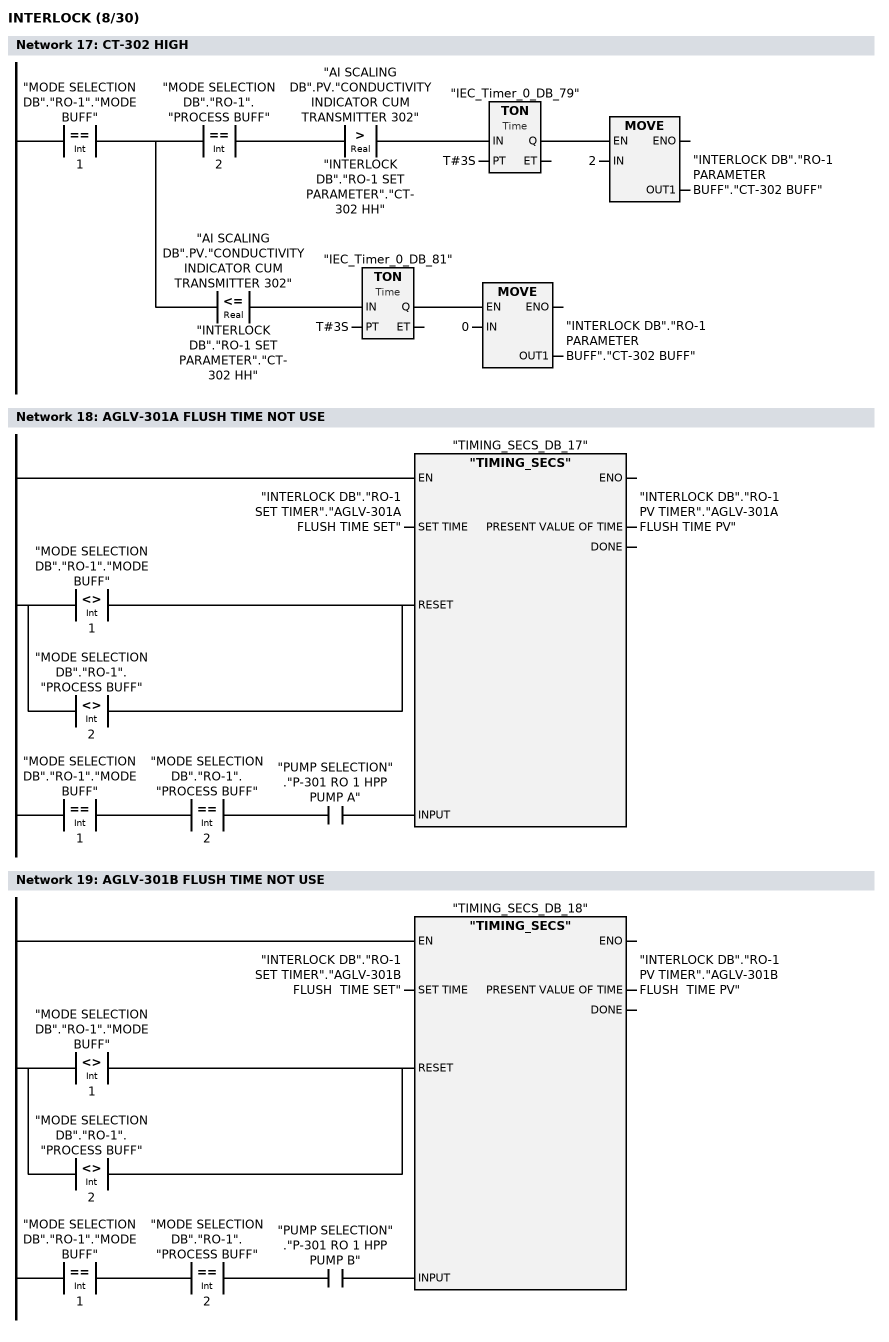
   RUNG wire#powerrail
      { S7_Templates := "SrcType := Int" } EQ_Contact(in1 := "MODE SELECTION DB"."RO-1"."MODE BUFF", in2 := 1)
      wire#w1
      { S7_Templates := "SrcType := Int" } EQ_Contact(in1 := "MODE SELECTION DB"."RO-1"."PROCESS BUFF", in2 := 2)
      { S7_Templates := "SrcType := Real" } GT_Contact(in1 := "AI SCALING DB".PV."CONDUCTIVITY INDICATOR CUM TRANSMITTER 302", in2 := "INTERLOCK DB"."RO-1 SET PARAMETER"."CT-302 HH")
      { S7_Templates := "time_type := Time" } "IEC_Timer_0_DB_79".TON(pt := T#3S, et =>)
      Move(in := 2, out1 => "INTERLOCK DB"."RO-1 PARAMETER BUFF"."CT-302 BUFF")
   END_RUNG
   RUNG wire#w1
      { S7_Templates := "SrcType := Real" } LE_Contact(in1 := "AI SCALING DB".PV."CONDUCTIVITY INDICATOR CUM TRANSMITTER 302", in2 := "INTERLOCK DB"."RO-1 SET PARAMETER"."CT-302 HH")
      { S7_Templates := "time_type := Time" } "IEC_Timer_0_DB_81".TON(pt := T#3S, et =>)
      Move(in := 0, out1 => "INTERLOCK DB"."RO-1 PARAMETER BUFF"."CT-302 BUFF")
   END_RUNG
   // the same network as SCL:
   #_w1 := "MODE SELECTION DB"."RO-1"."MODE BUFF" = 1;
   "IEC_Timer_0_DB_79".TON(IN := #_w1 AND ("MODE SELECTION DB"."RO-1"."PROCESS BUFF" = 2) AND ("AI SCALING DB".PV."CONDUCTIVITY INDICATOR CUM TRANSMITTER 302" > "INTERLOCK DB"."RO-1 SET PARAMETER"."CT-302 HH"),
                           PT := T#3S);
   IF "IEC_Timer_0_DB_79".Q THEN "INTERLOCK DB"."RO-1 PARAMETER BUFF"."CT-302 BUFF" := 2; END_IF;
   "IEC_Timer_0_DB_81".TON(IN := #_w1 AND ("AI SCALING DB".PV."CONDUCTIVITY INDICATOR CUM TRANSMITTER 302" <= "INTERLOCK DB"."RO-1 SET PARAMETER"."CT-302 HH"),
                           PT := T#3S);
   IF "IEC_Timer_0_DB_81".Q THEN "INTERLOCK DB"."RO-1 PARAMETER BUFF"."CT-302 BUFF" := 0; END_IF;
END_REGION

REGION Network 18: AGLV-301A FLUSH TIME NOT USE
   RUNG wire#powerrail
      "TIMING_SECS_DB_17"(RESET := wire#w1, INPUT := wire#w2, "SET TIME" := "INTERLOCK DB"."RO-1 SET TIMER"."AGLV-301A FLUSH TIME SET", "PRESENT VALUE OF TIME" => "INTERLOCK DB"."RO-1 PV TIMER"."AGLV-301A FLUSH TIME PV", DONE =>)
   END_RUNG
   RUNG wire#powerrail
      { S7_Templates := "SrcType := Int" } NE_Contact(in1 := "MODE SELECTION DB"."RO-1"."MODE BUFF", in2 := 1)
   END_RUNG wire#w1
   RUNG wire#powerrail
      { S7_Templates := "SrcType := Int" } NE_Contact(in1 := "MODE SELECTION DB"."RO-1"."PROCESS BUFF", in2 := 2)
   END_RUNG wire#w1
   RUNG wire#powerrail
      { S7_Templates := "SrcType := Int" } EQ_Contact(in1 := "MODE SELECTION DB"."RO-1"."MODE BUFF", in2 := 1)
      { S7_Templates := "SrcType := Int" } EQ_Contact(in1 := "MODE SELECTION DB"."RO-1"."PROCESS BUFF", in2 := 2)
      Contact( "PUMP SELECTION"."P-301 RO 1 HPP PUMP A" )
   END_RUNG wire#w2
   // the same network as SCL:
   "TIMING_SECS_DB_17"("SET TIME" := "INTERLOCK DB"."RO-1 SET TIMER"."AGLV-301A FLUSH TIME SET",   // "TIMING_SECS"
                       RESET := ("MODE SELECTION DB"."RO-1"."MODE BUFF" <> 1) OR ("MODE SELECTION DB"."RO-1"."PROCESS BUFF" <> 2),
                       INPUT := ("MODE SELECTION DB"."RO-1"."MODE BUFF" = 1) AND ("MODE SELECTION DB"."RO-1"."PROCESS BUFF" = 2) AND "PUMP SELECTION"."P-301 RO 1 HPP PUMP A",
                       "PRESENT VALUE OF TIME" => "INTERLOCK DB"."RO-1 PV TIMER"."AGLV-301A FLUSH TIME PV");
END_REGION

REGION Network 19: AGLV-301B FLUSH TIME NOT USE
   RUNG wire#powerrail
      "TIMING_SECS_DB_18"(RESET := wire#w1, INPUT := wire#w2, "SET TIME" := "INTERLOCK DB"."RO-1 SET TIMER"."AGLV-301B FLUSH  TIME SET", "PRESENT VALUE OF TIME" => "INTERLOCK DB"."RO-1 PV TIMER"."AGLV-301B FLUSH  TIME PV", DONE =>)
   END_RUNG
   RUNG wire#powerrail
      { S7_Templates := "SrcType := Int" } NE_Contact(in1 := "MODE SELECTION DB"."RO-1"."MODE BUFF", in2 := 1)
   END_RUNG wire#w1
   RUNG wire#powerrail
      { S7_Templates := "SrcType := Int" } NE_Contact(in1 := "MODE SELECTION DB"."RO-1"."PROCESS BUFF", in2 := 2)
   END_RUNG wire#w1
   RUNG wire#powerrail
      { S7_Templates := "SrcType := Int" } EQ_Contact(in1 := "MODE SELECTION DB"."RO-1"."MODE BUFF", in2 := 1)
      { S7_Templates := "SrcType := Int" } EQ_Contact(in1 := "MODE SELECTION DB"."RO-1"."PROCESS BUFF", in2 := 2)
      Contact( "PUMP SELECTION"."P-301 RO 1 HPP PUMP B" )
   END_RUNG wire#w2
   // the same network as SCL:
   "TIMING_SECS_DB_18"("SET TIME" := "INTERLOCK DB"."RO-1 SET TIMER"."AGLV-301B FLUSH  TIME SET",   // "TIMING_SECS"
                       RESET := ("MODE SELECTION DB"."RO-1"."MODE BUFF" <> 1) OR ("MODE SELECTION DB"."RO-1"."PROCESS BUFF" <> 2),
                       INPUT := ("MODE SELECTION DB"."RO-1"."MODE BUFF" = 1) AND ("MODE SELECTION DB"."RO-1"."PROCESS BUFF" = 2) AND "PUMP SELECTION"."P-301 RO 1 HPP PUMP B",
                       "PRESENT VALUE OF TIME" => "INTERLOCK DB"."RO-1 PV TIMER"."AGLV-301B FLUSH  TIME PV");
END_REGION

REGION Network 20: ORT-301
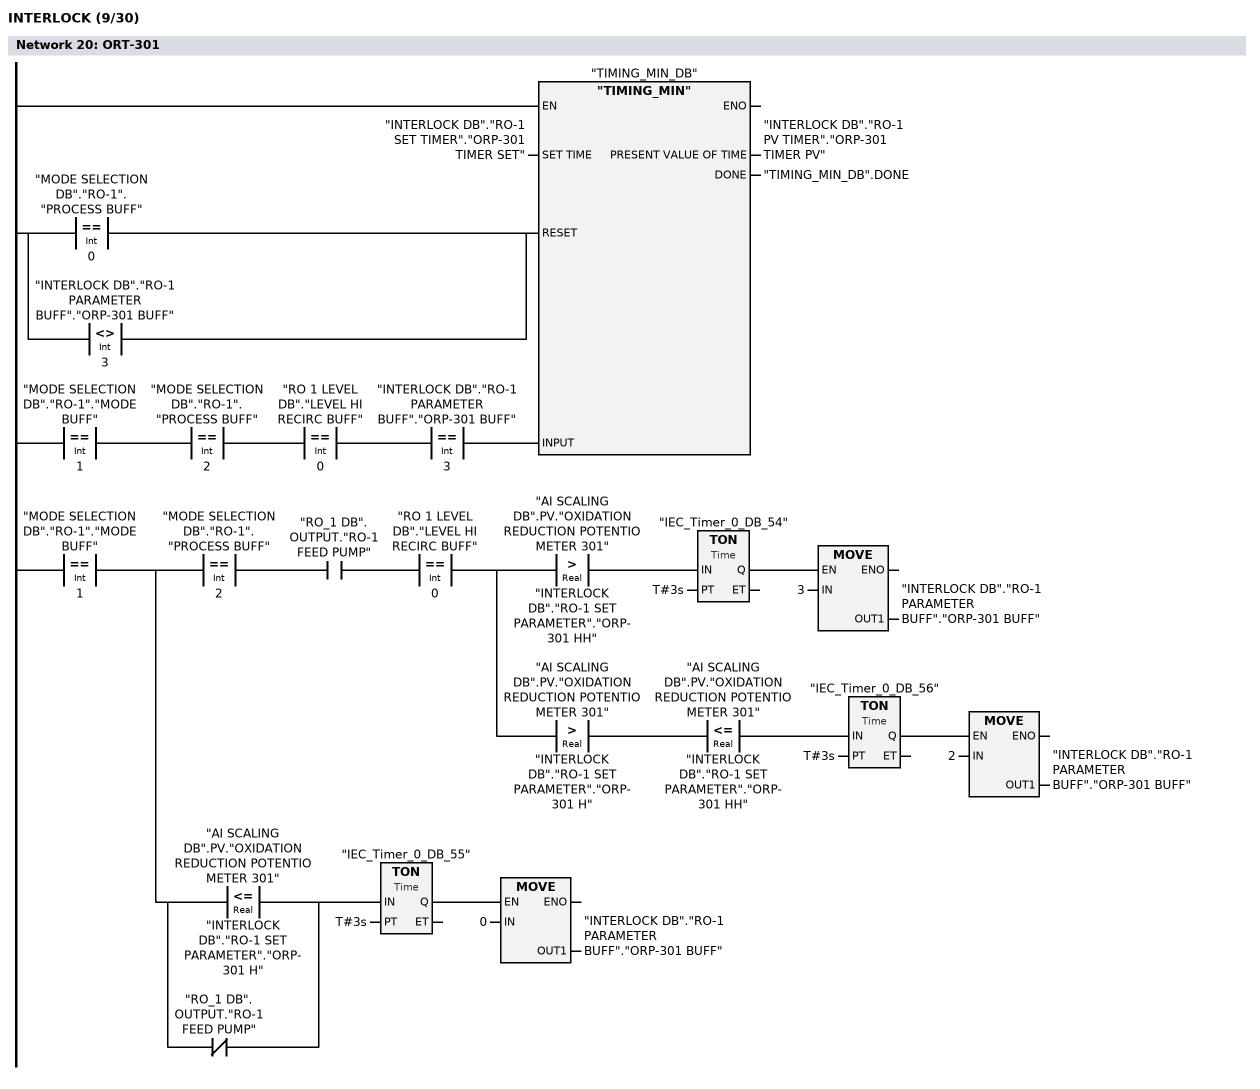
   RUNG wire#powerrail
      "TIMING_MIN_DB"(RESET := wire#w1, INPUT := wire#w2, "SET TIME" := "INTERLOCK DB"."RO-1 SET TIMER"."ORP-301 TIMER SET", "PRESENT VALUE OF TIME" => "INTERLOCK DB"."RO-1 PV TIMER"."ORP-301 TIMER PV", DONE => "TIMING_MIN_DB".DONE)
   END_RUNG
   RUNG wire#powerrail
      { S7_Templates := "SrcType := Int" } EQ_Contact(in1 := "MODE SELECTION DB"."RO-1"."PROCESS BUFF", in2 := 0)
   END_RUNG wire#w1
   RUNG wire#powerrail
      { S7_Templates := "SrcType := Int" } NE_Contact(in1 := "INTERLOCK DB"."RO-1 PARAMETER BUFF"."ORP-301 BUFF", in2 := 3)
   END_RUNG wire#w1
   RUNG wire#powerrail
      { S7_Templates := "SrcType := Int" } EQ_Contact(in1 := "MODE SELECTION DB"."RO-1"."MODE BUFF", in2 := 1)
      { S7_Templates := "SrcType := Int" } EQ_Contact(in1 := "MODE SELECTION DB"."RO-1"."PROCESS BUFF", in2 := 2)
      { S7_Templates := "SrcType := Int" } EQ_Contact(in1 := "RO 1 LEVEL DB"."LEVEL HI RECIRC BUFF", in2 := 0)
      { S7_Templates := "SrcType := Int" } EQ_Contact(in1 := "INTERLOCK DB"."RO-1 PARAMETER BUFF"."ORP-301 BUFF", in2 := 3)
   END_RUNG wire#w2
   RUNG wire#powerrail
      { S7_Templates := "SrcType := Int" } EQ_Contact(in1 := "MODE SELECTION DB"."RO-1"."MODE BUFF", in2 := 1)
      wire#w3
      { S7_Templates := "SrcType := Int" } EQ_Contact(in1 := "MODE SELECTION DB"."RO-1"."PROCESS BUFF", in2 := 2)
      Contact( "RO_1 DB".OUTPUT."RO-1 FEED PUMP" )
      { S7_Templates := "SrcType := Int" } EQ_Contact(in1 := "RO 1 LEVEL DB"."LEVEL HI RECIRC BUFF", in2 := 0)
      wire#w4
      { S7_Templates := "SrcType := Real" } GT_Contact(in1 := "AI SCALING DB".PV."OXIDATION REDUCTION POTENTIO METER 301", in2 := "INTERLOCK DB"."RO-1 SET PARAMETER"."ORP-301 HH")
      { S7_Templates := "time_type := Time" } "IEC_Timer_0_DB_54".TON(pt := T#3s, et =>)
      Move(in := 3, out1 => "INTERLOCK DB"."RO-1 PARAMETER BUFF"."ORP-301 BUFF")
   END_RUNG
   RUNG wire#w4
      { S7_Templates := "SrcType := Real" } GT_Contact(in1 := "AI SCALING DB".PV."OXIDATION REDUCTION POTENTIO METER 301", in2 := "INTERLOCK DB"."RO-1 SET PARAMETER"."ORP-301 H")
      { S7_Templates := "SrcType := Real" } LE_Contact(in1 := "AI SCALING DB".PV."OXIDATION REDUCTION POTENTIO METER 301", in2 := "INTERLOCK DB"."RO-1 SET PARAMETER"."ORP-301 HH")
      { S7_Templates := "time_type := Time" } "IEC_Timer_0_DB_56".TON(pt := T#3s, et =>)
      Move(in := 2, out1 => "INTERLOCK DB"."RO-1 PARAMETER BUFF"."ORP-301 BUFF")
   END_RUNG
   RUNG wire#w3
      { S7_Templates := "SrcType := Real" } LE_Contact(in1 := "AI SCALING DB".PV."OXIDATION REDUCTION POTENTIO METER 301", in2 := "INTERLOCK DB"."RO-1 SET PARAMETER"."ORP-301 H")
      wire#w5
      { S7_Templates := "time_type := Time" } "IEC_Timer_0_DB_55".TON(pt := T#3s, et =>)
      Move(in := 0, out1 => "INTERLOCK DB"."RO-1 PARAMETER BUFF"."ORP-301 BUFF")
   END_RUNG
   RUNG wire#w3
      I_Contact( "RO_1 DB".OUTPUT."RO-1 FEED PUMP" )
   END_RUNG wire#w5
   // the same network as SCL:
   "TIMING_MIN_DB"("SET TIME" := "INTERLOCK DB"."RO-1 SET TIMER"."ORP-301 TIMER SET",   // "TIMING_MIN"
                   RESET := ("MODE SELECTION DB"."RO-1"."PROCESS BUFF" = 0) OR ("INTERLOCK DB"."RO-1 PARAMETER BUFF"."ORP-301 BUFF" <> 3),
                   INPUT := ("MODE SELECTION DB"."RO-1"."MODE BUFF" = 1) AND ("MODE SELECTION DB"."RO-1"."PROCESS BUFF" = 2) AND ("RO 1 LEVEL DB"."LEVEL HI RECIRC BUFF" = 0) AND ("INTERLOCK DB"."RO-1 PARAMETER BUFF"."ORP-301 BUFF" = 3),
                   "PRESENT VALUE OF TIME" => "INTERLOCK DB"."RO-1 PV TIMER"."ORP-301 TIMER PV",
                   DONE => "TIMING_MIN_DB".DONE);
   #_w1 := "MODE SELECTION DB"."RO-1"."MODE BUFF" = 1;
   #_w2 := #_w1 AND ("MODE SELECTION DB"."RO-1"."PROCESS BUFF" = 2) AND "RO_1 DB".OUTPUT."RO-1 FEED PUMP" AND ("RO 1 LEVEL DB"."LEVEL HI RECIRC BUFF" = 0);
   "IEC_Timer_0_DB_54".TON(IN := #_w2 AND ("AI SCALING DB".PV."OXIDATION REDUCTION POTENTIO METER 301" > "INTERLOCK DB"."RO-1 SET PARAMETER"."ORP-301 HH"),
                           PT := T#3s);
   IF "IEC_Timer_0_DB_54".Q THEN "INTERLOCK DB"."RO-1 PARAMETER BUFF"."ORP-301 BUFF" := 3; END_IF;
   "IEC_Timer_0_DB_56".TON(IN := #_w2 AND ("AI SCALING DB".PV."OXIDATION REDUCTION POTENTIO METER 301" > "INTERLOCK DB"."RO-1 SET PARAMETER"."ORP-301 H") AND ("AI SCALING DB".PV."OXIDATION REDUCTION POTENTIO METER 301" <= "INTERLOCK DB"."RO-1 SET PARAMETER"."ORP-301 HH"),
                           PT := T#3s);
   IF "IEC_Timer_0_DB_56".Q THEN "INTERLOCK DB"."RO-1 PARAMETER BUFF"."ORP-301 BUFF" := 2; END_IF;
   "IEC_Timer_0_DB_55".TON(IN := #_w1 AND (("AI SCALING DB".PV."OXIDATION REDUCTION POTENTIO METER 301" <= "INTERLOCK DB"."RO-1 SET PARAMETER"."ORP-301 H") OR NOT "RO_1 DB".OUTPUT."RO-1 FEED PUMP"),
                           PT := T#3s);
   IF "IEC_Timer_0_DB_55".Q THEN "INTERLOCK DB"."RO-1 PARAMETER BUFF"."ORP-301 BUFF" := 0; END_IF;
END_REGION

REGION Network 22: AUTO INTERLOCK FOR RO-2 ///////////////////////////////////////////////////////
END_REGION

REGION Network 23: LPS-401&402LOW TIMER SET
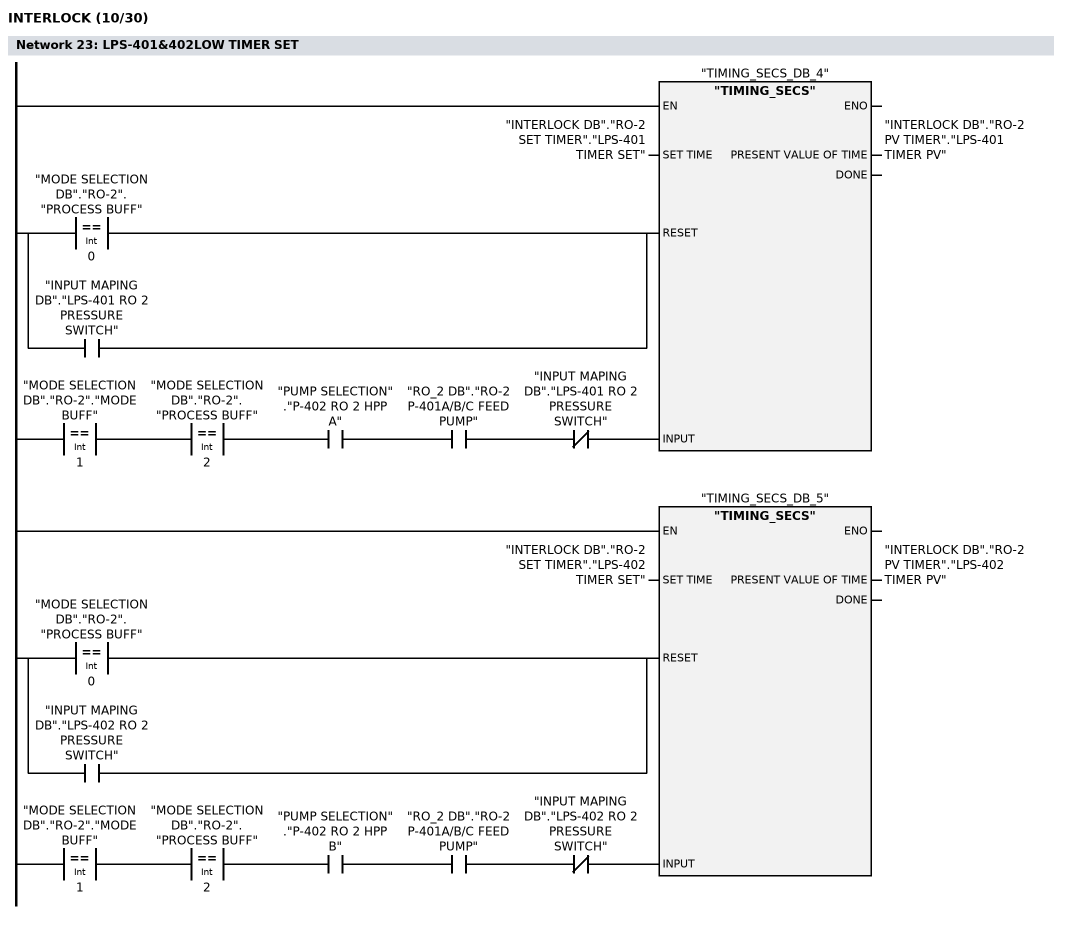
   RUNG wire#powerrail
      "TIMING_SECS_DB_4"(RESET := wire#w1, INPUT := wire#w2, "SET TIME" := "INTERLOCK DB"."RO-2 SET TIMER"."LPS-401 TIMER SET", "PRESENT VALUE OF TIME" => "INTERLOCK DB"."RO-2 PV TIMER"."LPS-401 TIMER PV", DONE =>)
   END_RUNG
   RUNG wire#powerrail
      { S7_Templates := "SrcType := Int" } EQ_Contact(in1 := "MODE SELECTION DB"."RO-2"."PROCESS BUFF", in2 := 0)
   END_RUNG wire#w1
   RUNG wire#powerrail
      Contact( "INPUT MAPING DB"."LPS-401 RO 2 PRESSURE SWITCH" )
   END_RUNG wire#w1
   RUNG wire#powerrail
      { S7_Templates := "SrcType := Int" } EQ_Contact(in1 := "MODE SELECTION DB"."RO-2"."MODE BUFF", in2 := 1)
      { S7_Templates := "SrcType := Int" } EQ_Contact(in1 := "MODE SELECTION DB"."RO-2"."PROCESS BUFF", in2 := 2)
      Contact( "PUMP SELECTION"."P-402 RO 2 HPP A" )
      Contact( "RO_2 DB"."RO-2 P-401A/B/C FEED PUMP" )
      I_Contact( "INPUT MAPING DB"."LPS-401 RO 2 PRESSURE SWITCH" )
   END_RUNG wire#w2
   RUNG wire#powerrail
      "TIMING_SECS_DB_5"(RESET := wire#w3, INPUT := wire#w4, "SET TIME" := "INTERLOCK DB"."RO-2 SET TIMER"."LPS-402 TIMER SET", "PRESENT VALUE OF TIME" => "INTERLOCK DB"."RO-2 PV TIMER"."LPS-402 TIMER PV", DONE =>)
   END_RUNG
   RUNG wire#powerrail
      { S7_Templates := "SrcType := Int" } EQ_Contact(in1 := "MODE SELECTION DB"."RO-2"."PROCESS BUFF", in2 := 0)
   END_RUNG wire#w3
   RUNG wire#powerrail
      Contact( "INPUT MAPING DB"."LPS-402 RO 2 PRESSURE SWITCH" )
   END_RUNG wire#w3
   RUNG wire#powerrail
      { S7_Templates := "SrcType := Int" } EQ_Contact(in1 := "MODE SELECTION DB"."RO-2"."MODE BUFF", in2 := 1)
      { S7_Templates := "SrcType := Int" } EQ_Contact(in1 := "MODE SELECTION DB"."RO-2"."PROCESS BUFF", in2 := 2)
      Contact( "PUMP SELECTION"."P-402 RO 2 HPP B" )
      Contact( "RO_2 DB"."RO-2 P-401A/B/C FEED PUMP" )
      I_Contact( "INPUT MAPING DB"."LPS-402 RO 2 PRESSURE SWITCH" )
   END_RUNG wire#w4
   // the same network as SCL:
   "TIMING_SECS_DB_4"("SET TIME" := "INTERLOCK DB"."RO-2 SET TIMER"."LPS-401 TIMER SET",   // "TIMING_SECS"
                      RESET := ("MODE SELECTION DB"."RO-2"."PROCESS BUFF" = 0) OR "INPUT MAPING DB"."LPS-401 RO 2 PRESSURE SWITCH",
                      INPUT := ("MODE SELECTION DB"."RO-2"."MODE BUFF" = 1) AND ("MODE SELECTION DB"."RO-2"."PROCESS BUFF" = 2) AND "PUMP SELECTION"."P-402 RO 2 HPP A" AND "RO_2 DB"."RO-2 P-401A/B/C FEED PUMP" AND NOT "INPUT MAPING DB"."LPS-401 RO 2 PRESSURE SWITCH",
                      "PRESENT VALUE OF TIME" => "INTERLOCK DB"."RO-2 PV TIMER"."LPS-401 TIMER PV");
   "TIMING_SECS_DB_5"("SET TIME" := "INTERLOCK DB"."RO-2 SET TIMER"."LPS-402 TIMER SET",   // "TIMING_SECS"
                      RESET := ("MODE SELECTION DB"."RO-2"."PROCESS BUFF" = 0) OR "INPUT MAPING DB"."LPS-402 RO 2 PRESSURE SWITCH",
                      INPUT := ("MODE SELECTION DB"."RO-2"."MODE BUFF" = 1) AND ("MODE SELECTION DB"."RO-2"."PROCESS BUFF" = 2) AND "PUMP SELECTION"."P-402 RO 2 HPP B" AND "RO_2 DB"."RO-2 P-401A/B/C FEED PUMP" AND NOT "INPUT MAPING DB"."LPS-402 RO 2 PRESSURE SWITCH",
                      "PRESENT VALUE OF TIME" => "INTERLOCK DB"."RO-2 PV TIMER"."LPS-402 TIMER PV");
END_REGION

REGION Network 24: HPS-401 &402
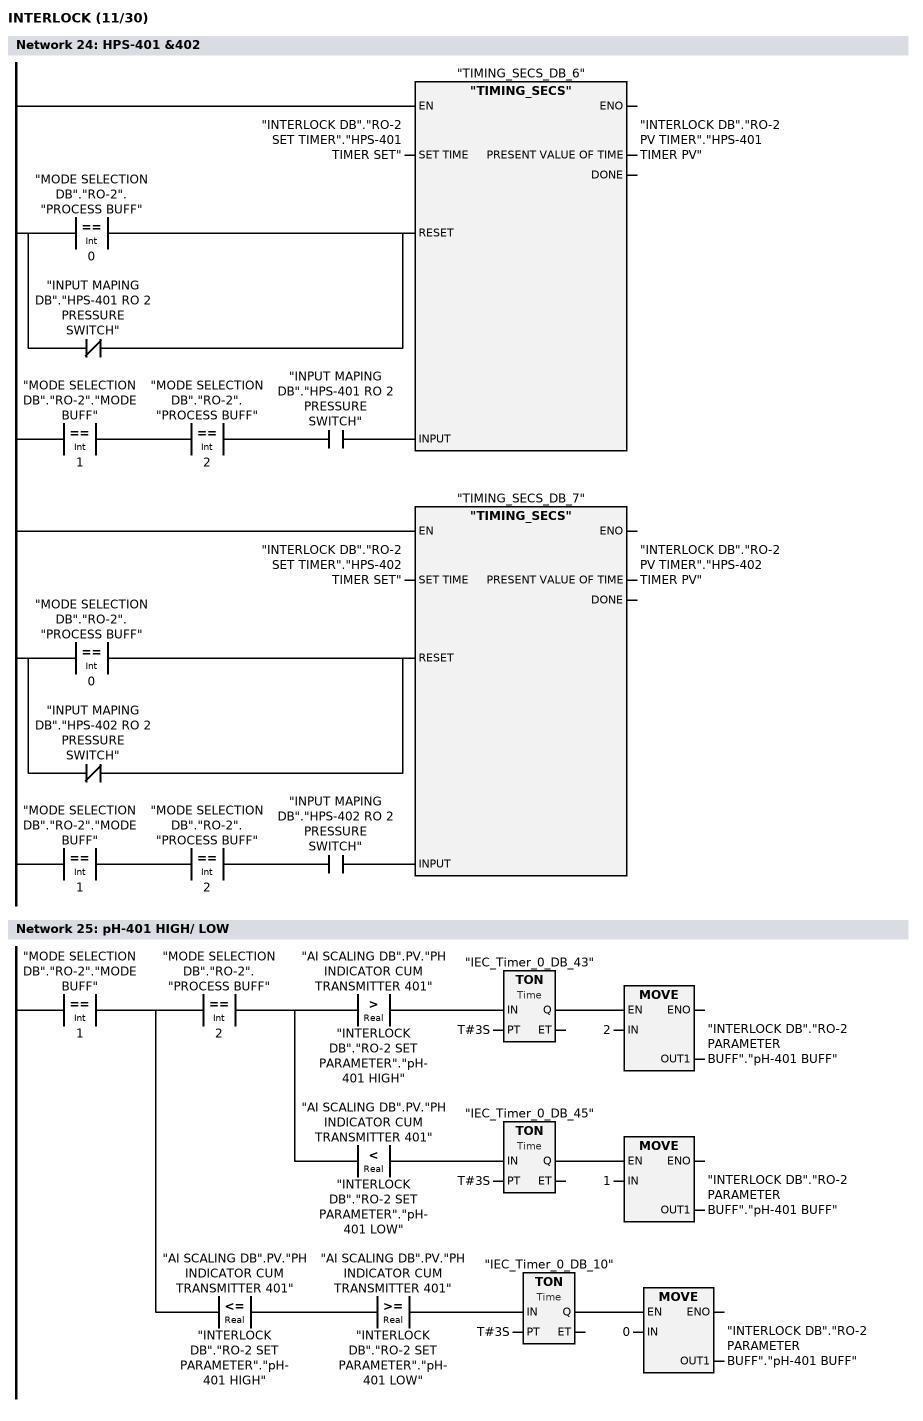
   RUNG wire#powerrail
      "TIMING_SECS_DB_6"(RESET := wire#w1, INPUT := wire#w2, "SET TIME" := "INTERLOCK DB"."RO-2 SET TIMER"."HPS-401 TIMER SET", "PRESENT VALUE OF TIME" => "INTERLOCK DB"."RO-2 PV TIMER"."HPS-401 TIMER PV", DONE =>)
   END_RUNG
   RUNG wire#powerrail
      { S7_Templates := "SrcType := Int" } EQ_Contact(in1 := "MODE SELECTION DB"."RO-2"."PROCESS BUFF", in2 := 0)
   END_RUNG wire#w1
   RUNG wire#powerrail
      I_Contact( "INPUT MAPING DB"."HPS-401 RO 2 PRESSURE SWITCH" )
   END_RUNG wire#w1
   RUNG wire#powerrail
      { S7_Templates := "SrcType := Int" } EQ_Contact(in1 := "MODE SELECTION DB"."RO-2"."MODE BUFF", in2 := 1)
      { S7_Templates := "SrcType := Int" } EQ_Contact(in1 := "MODE SELECTION DB"."RO-2"."PROCESS BUFF", in2 := 2)
      Contact( "INPUT MAPING DB"."HPS-401 RO 2 PRESSURE SWITCH" )
   END_RUNG wire#w2
   RUNG wire#powerrail
      "TIMING_SECS_DB_7"(RESET := wire#w3, INPUT := wire#w4, "SET TIME" := "INTERLOCK DB"."RO-2 SET TIMER"."HPS-402 TIMER SET", "PRESENT VALUE OF TIME" => "INTERLOCK DB"."RO-2 PV TIMER"."HPS-402 TIMER PV", DONE =>)
   END_RUNG
   RUNG wire#powerrail
      { S7_Templates := "SrcType := Int" } EQ_Contact(in1 := "MODE SELECTION DB"."RO-2"."PROCESS BUFF", in2 := 0)
   END_RUNG wire#w3
   RUNG wire#powerrail
      I_Contact( "INPUT MAPING DB"."HPS-402 RO 2 PRESSURE SWITCH" )
   END_RUNG wire#w3
   RUNG wire#powerrail
      { S7_Templates := "SrcType := Int" } EQ_Contact(in1 := "MODE SELECTION DB"."RO-2"."MODE BUFF", in2 := 1)
      { S7_Templates := "SrcType := Int" } EQ_Contact(in1 := "MODE SELECTION DB"."RO-2"."PROCESS BUFF", in2 := 2)
      Contact( "INPUT MAPING DB"."HPS-402 RO 2 PRESSURE SWITCH" )
   END_RUNG wire#w4
   // the same network as SCL:
   "TIMING_SECS_DB_6"("SET TIME" := "INTERLOCK DB"."RO-2 SET TIMER"."HPS-401 TIMER SET",   // "TIMING_SECS"
                      RESET := ("MODE SELECTION DB"."RO-2"."PROCESS BUFF" = 0) OR NOT "INPUT MAPING DB"."HPS-401 RO 2 PRESSURE SWITCH",
                      INPUT := ("MODE SELECTION DB"."RO-2"."MODE BUFF" = 1) AND ("MODE SELECTION DB"."RO-2"."PROCESS BUFF" = 2) AND "INPUT MAPING DB"."HPS-401 RO 2 PRESSURE SWITCH",
                      "PRESENT VALUE OF TIME" => "INTERLOCK DB"."RO-2 PV TIMER"."HPS-401 TIMER PV");
   "TIMING_SECS_DB_7"("SET TIME" := "INTERLOCK DB"."RO-2 SET TIMER"."HPS-402 TIMER SET",   // "TIMING_SECS"
                      RESET := ("MODE SELECTION DB"."RO-2"."PROCESS BUFF" = 0) OR NOT "INPUT MAPING DB"."HPS-402 RO 2 PRESSURE SWITCH",
                      INPUT := ("MODE SELECTION DB"."RO-2"."MODE BUFF" = 1) AND ("MODE SELECTION DB"."RO-2"."PROCESS BUFF" = 2) AND "INPUT MAPING DB"."HPS-402 RO 2 PRESSURE SWITCH",
                      "PRESENT VALUE OF TIME" => "INTERLOCK DB"."RO-2 PV TIMER"."HPS-402 TIMER PV");
END_REGION

REGION Network 25: pH-401 HIGH/ LOW
   RUNG wire#powerrail
      { S7_Templates := "SrcType := Int" } EQ_Contact(in1 := "MODE SELECTION DB"."RO-2"."MODE BUFF", in2 := 1)
      wire#w1
      { S7_Templates := "SrcType := Int" } EQ_Contact(in1 := "MODE SELECTION DB"."RO-2"."PROCESS BUFF", in2 := 2)
      wire#w2
      { S7_Templates := "SrcType := Real" } GT_Contact(in1 := "AI SCALING DB".PV."PH INDICATOR CUM TRANSMITTER 401", in2 := "INTERLOCK DB"."RO-2 SET PARAMETER"."pH-401 HIGH")
      { S7_Templates := "time_type := Time" } "IEC_Timer_0_DB_43".TON(pt := T#3S, et =>)
      Move(in := 2, out1 => "INTERLOCK DB"."RO-2 PARAMETER BUFF"."pH-401 BUFF")
   END_RUNG
   RUNG wire#w2
      { S7_Templates := "SrcType := Real" } LT_Contact(in1 := "AI SCALING DB".PV."PH INDICATOR CUM TRANSMITTER 401", in2 := "INTERLOCK DB"."RO-2 SET PARAMETER"."pH-401 LOW")
      { S7_Templates := "time_type := Time" } "IEC_Timer_0_DB_45".TON(pt := T#3S, et =>)
      Move(in := 1, out1 => "INTERLOCK DB"."RO-2 PARAMETER BUFF"."pH-401 BUFF")
   END_RUNG
   RUNG wire#w1
      { S7_Templates := "SrcType := Real" } LE_Contact(in1 := "AI SCALING DB".PV."PH INDICATOR CUM TRANSMITTER 401", in2 := "INTERLOCK DB"."RO-2 SET PARAMETER"."pH-401 HIGH")
      { S7_Templates := "SrcType := Real" } GE_Contact(in1 := "AI SCALING DB".PV."PH INDICATOR CUM TRANSMITTER 401", in2 := "INTERLOCK DB"."RO-2 SET PARAMETER"."pH-401 LOW")
      { S7_Templates := "time_type := Time" } "IEC_Timer_0_DB_10".TON(pt := T#3S, et =>)
      Move(in := 0, out1 => "INTERLOCK DB"."RO-2 PARAMETER BUFF"."pH-401 BUFF")
   END_RUNG
   // the same network as SCL:
   #_w1 := "MODE SELECTION DB"."RO-2"."MODE BUFF" = 1;
   #_w2 := #_w1 AND ("MODE SELECTION DB"."RO-2"."PROCESS BUFF" = 2);
   "IEC_Timer_0_DB_43".TON(IN := #_w2 AND ("AI SCALING DB".PV."PH INDICATOR CUM TRANSMITTER 401" > "INTERLOCK DB"."RO-2 SET PARAMETER"."pH-401 HIGH"),
                           PT := T#3S);
   IF "IEC_Timer_0_DB_43".Q THEN "INTERLOCK DB"."RO-2 PARAMETER BUFF"."pH-401 BUFF" := 2; END_IF;
   "IEC_Timer_0_DB_45".TON(IN := #_w2 AND ("AI SCALING DB".PV."PH INDICATOR CUM TRANSMITTER 401" < "INTERLOCK DB"."RO-2 SET PARAMETER"."pH-401 LOW"),
                           PT := T#3S);
   IF "IEC_Timer_0_DB_45".Q THEN "INTERLOCK DB"."RO-2 PARAMETER BUFF"."pH-401 BUFF" := 1; END_IF;
   "IEC_Timer_0_DB_10".TON(IN := #_w1 AND ("AI SCALING DB".PV."PH INDICATOR CUM TRANSMITTER 401" <= "INTERLOCK DB"."RO-2 SET PARAMETER"."pH-401 HIGH") AND ("AI SCALING DB".PV."PH INDICATOR CUM TRANSMITTER 401" >= "INTERLOCK DB"."RO-2 SET PARAMETER"."pH-401 LOW"),
                           PT := T#3S);
   IF "IEC_Timer_0_DB_10".Q THEN "INTERLOCK DB"."RO-2 PARAMETER BUFF"."pH-401 BUFF" := 0; END_IF;
END_REGION

REGION Network 26: pH-402 HIGH/ LOW
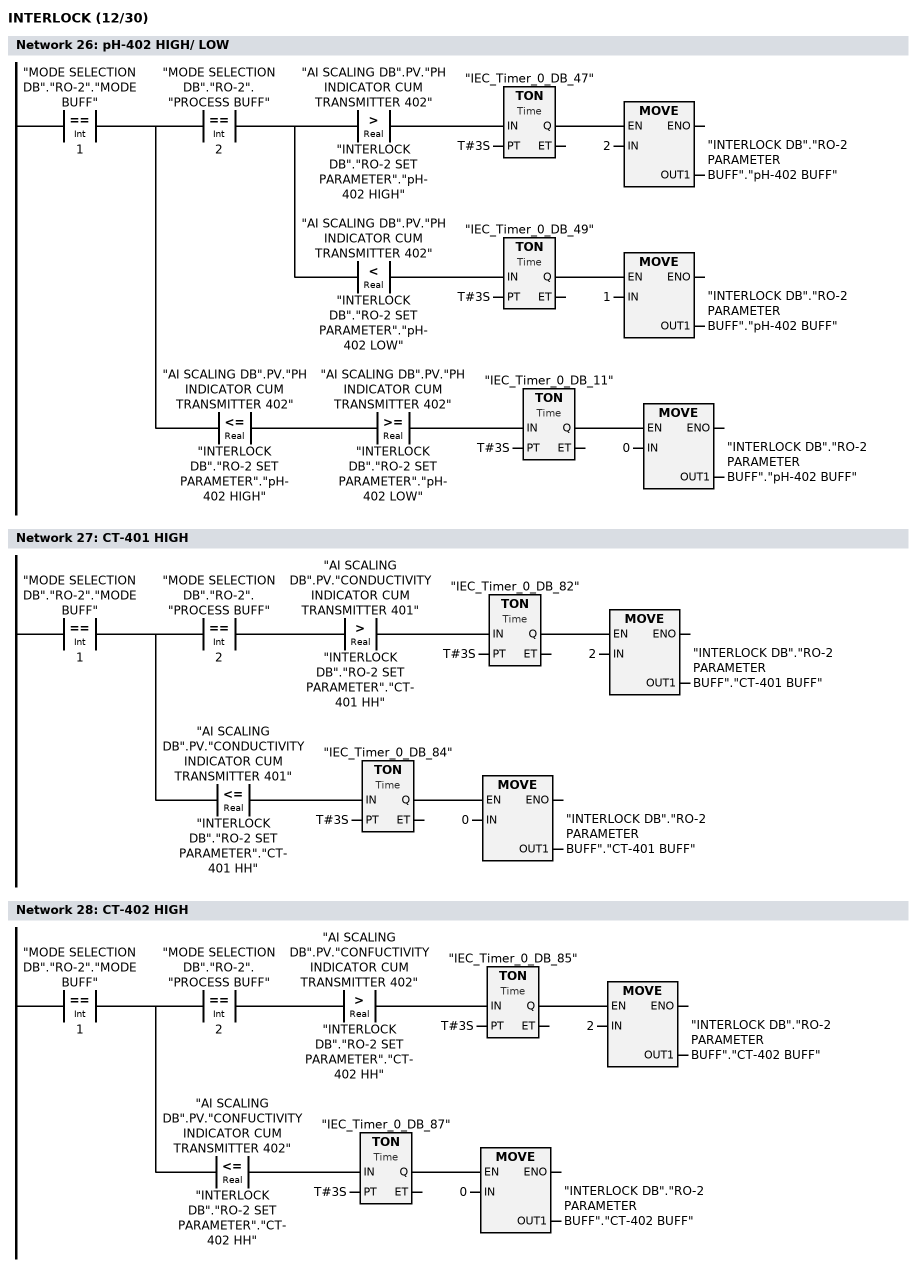
   RUNG wire#powerrail
      { S7_Templates := "SrcType := Int" } EQ_Contact(in1 := "MODE SELECTION DB"."RO-2"."MODE BUFF", in2 := 1)
      wire#w1
      { S7_Templates := "SrcType := Int" } EQ_Contact(in1 := "MODE SELECTION DB"."RO-2"."PROCESS BUFF", in2 := 2)
      wire#w2
      { S7_Templates := "SrcType := Real" } GT_Contact(in1 := "AI SCALING DB".PV."PH INDICATOR CUM TRANSMITTER 402", in2 := "INTERLOCK DB"."RO-2 SET PARAMETER"."pH-402 HIGH")
      { S7_Templates := "time_type := Time" } "IEC_Timer_0_DB_47".TON(pt := T#3S, et =>)
      Move(in := 2, out1 => "INTERLOCK DB"."RO-2 PARAMETER BUFF"."pH-402 BUFF")
   END_RUNG
   RUNG wire#w2
      { S7_Templates := "SrcType := Real" } LT_Contact(in1 := "AI SCALING DB".PV."PH INDICATOR CUM TRANSMITTER 402", in2 := "INTERLOCK DB"."RO-2 SET PARAMETER"."pH-402 LOW")
      { S7_Templates := "time_type := Time" } "IEC_Timer_0_DB_49".TON(pt := T#3S, et =>)
      Move(in := 1, out1 => "INTERLOCK DB"."RO-2 PARAMETER BUFF"."pH-402 BUFF")
   END_RUNG
   RUNG wire#w1
      { S7_Templates := "SrcType := Real" } LE_Contact(in1 := "AI SCALING DB".PV."PH INDICATOR CUM TRANSMITTER 402", in2 := "INTERLOCK DB"."RO-2 SET PARAMETER"."pH-402 HIGH")
      { S7_Templates := "SrcType := Real" } GE_Contact(in1 := "AI SCALING DB".PV."PH INDICATOR CUM TRANSMITTER 402", in2 := "INTERLOCK DB"."RO-2 SET PARAMETER"."pH-402 LOW")
      { S7_Templates := "time_type := Time" } "IEC_Timer_0_DB_11".TON(pt := T#3S, et =>)
      Move(in := 0, out1 => "INTERLOCK DB"."RO-2 PARAMETER BUFF"."pH-402 BUFF")
   END_RUNG
   // the same network as SCL:
   #_w1 := "MODE SELECTION DB"."RO-2"."MODE BUFF" = 1;
   #_w2 := #_w1 AND ("MODE SELECTION DB"."RO-2"."PROCESS BUFF" = 2);
   "IEC_Timer_0_DB_47".TON(IN := #_w2 AND ("AI SCALING DB".PV."PH INDICATOR CUM TRANSMITTER 402" > "INTERLOCK DB"."RO-2 SET PARAMETER"."pH-402 HIGH"),
                           PT := T#3S);
   IF "IEC_Timer_0_DB_47".Q THEN "INTERLOCK DB"."RO-2 PARAMETER BUFF"."pH-402 BUFF" := 2; END_IF;
   "IEC_Timer_0_DB_49".TON(IN := #_w2 AND ("AI SCALING DB".PV."PH INDICATOR CUM TRANSMITTER 402" < "INTERLOCK DB"."RO-2 SET PARAMETER"."pH-402 LOW"),
                           PT := T#3S);
   IF "IEC_Timer_0_DB_49".Q THEN "INTERLOCK DB"."RO-2 PARAMETER BUFF"."pH-402 BUFF" := 1; END_IF;
   "IEC_Timer_0_DB_11".TON(IN := #_w1 AND ("AI SCALING DB".PV."PH INDICATOR CUM TRANSMITTER 402" <= "INTERLOCK DB"."RO-2 SET PARAMETER"."pH-402 HIGH") AND ("AI SCALING DB".PV."PH INDICATOR CUM TRANSMITTER 402" >= "INTERLOCK DB"."RO-2 SET PARAMETER"."pH-402 LOW"),
                           PT := T#3S);
   IF "IEC_Timer_0_DB_11".Q THEN "INTERLOCK DB"."RO-2 PARAMETER BUFF"."pH-402 BUFF" := 0; END_IF;
END_REGION

REGION Network 27: CT-401 HIGH
   RUNG wire#powerrail
      { S7_Templates := "SrcType := Int" } EQ_Contact(in1 := "MODE SELECTION DB"."RO-2"."MODE BUFF", in2 := 1)
      wire#w1
      { S7_Templates := "SrcType := Int" } EQ_Contact(in1 := "MODE SELECTION DB"."RO-2"."PROCESS BUFF", in2 := 2)
      { S7_Templates := "SrcType := Real" } GT_Contact(in1 := "AI SCALING DB".PV."CONDUCTIVITY INDICATOR CUM TRANSMITTER 401", in2 := "INTERLOCK DB"."RO-2 SET PARAMETER"."CT-401 HH")
      { S7_Templates := "time_type := Time" } "IEC_Timer_0_DB_82".TON(pt := T#3S, et =>)
      Move(in := 2, out1 => "INTERLOCK DB"."RO-2 PARAMETER BUFF"."CT-401 BUFF")
   END_RUNG
   RUNG wire#w1
      { S7_Templates := "SrcType := Real" } LE_Contact(in1 := "AI SCALING DB".PV."CONDUCTIVITY INDICATOR CUM TRANSMITTER 401", in2 := "INTERLOCK DB"."RO-2 SET PARAMETER"."CT-401 HH")
      { S7_Templates := "time_type := Time" } "IEC_Timer_0_DB_84".TON(pt := T#3S, et =>)
      Move(in := 0, out1 => "INTERLOCK DB"."RO-2 PARAMETER BUFF"."CT-401 BUFF")
   END_RUNG
   // the same network as SCL:
   #_w1 := "MODE SELECTION DB"."RO-2"."MODE BUFF" = 1;
   "IEC_Timer_0_DB_82".TON(IN := #_w1 AND ("MODE SELECTION DB"."RO-2"."PROCESS BUFF" = 2) AND ("AI SCALING DB".PV."CONDUCTIVITY INDICATOR CUM TRANSMITTER 401" > "INTERLOCK DB"."RO-2 SET PARAMETER"."CT-401 HH"),
                           PT := T#3S);
   IF "IEC_Timer_0_DB_82".Q THEN "INTERLOCK DB"."RO-2 PARAMETER BUFF"."CT-401 BUFF" := 2; END_IF;
   "IEC_Timer_0_DB_84".TON(IN := #_w1 AND ("AI SCALING DB".PV."CONDUCTIVITY INDICATOR CUM TRANSMITTER 401" <= "INTERLOCK DB"."RO-2 SET PARAMETER"."CT-401 HH"),
                           PT := T#3S);
   IF "IEC_Timer_0_DB_84".Q THEN "INTERLOCK DB"."RO-2 PARAMETER BUFF"."CT-401 BUFF" := 0; END_IF;
END_REGION

REGION Network 28: CT-402 HIGH
   RUNG wire#powerrail
      { S7_Templates := "SrcType := Int" } EQ_Contact(in1 := "MODE SELECTION DB"."RO-2"."MODE BUFF", in2 := 1)
      wire#w1
      { S7_Templates := "SrcType := Int" } EQ_Contact(in1 := "MODE SELECTION DB"."RO-2"."PROCESS BUFF", in2 := 2)
      { S7_Templates := "SrcType := Real" } GT_Contact(in1 := "AI SCALING DB".PV."CONFUCTIVITY INDICATOR CUM TRANSMITTER 402", in2 := "INTERLOCK DB"."RO-2 SET PARAMETER"."CT-402 HH")
      { S7_Templates := "time_type := Time" } "IEC_Timer_0_DB_85".TON(pt := T#3S, et =>)
      Move(in := 2, out1 => "INTERLOCK DB"."RO-2 PARAMETER BUFF"."CT-402 BUFF")
   END_RUNG
   RUNG wire#w1
      { S7_Templates := "SrcType := Real" } LE_Contact(in1 := "AI SCALING DB".PV."CONFUCTIVITY INDICATOR CUM TRANSMITTER 402", in2 := "INTERLOCK DB"."RO-2 SET PARAMETER"."CT-402 HH")
      { S7_Templates := "time_type := Time" } "IEC_Timer_0_DB_87".TON(pt := T#3S, et =>)
      Move(in := 0, out1 => "INTERLOCK DB"."RO-2 PARAMETER BUFF"."CT-402 BUFF")
   END_RUNG
   // the same network as SCL:
   #_w1 := "MODE SELECTION DB"."RO-2"."MODE BUFF" = 1;
   "IEC_Timer_0_DB_85".TON(IN := #_w1 AND ("MODE SELECTION DB"."RO-2"."PROCESS BUFF" = 2) AND ("AI SCALING DB".PV."CONFUCTIVITY INDICATOR CUM TRANSMITTER 402" > "INTERLOCK DB"."RO-2 SET PARAMETER"."CT-402 HH"),
                           PT := T#3S);
   IF "IEC_Timer_0_DB_85".Q THEN "INTERLOCK DB"."RO-2 PARAMETER BUFF"."CT-402 BUFF" := 2; END_IF;
   "IEC_Timer_0_DB_87".TON(IN := #_w1 AND ("AI SCALING DB".PV."CONFUCTIVITY INDICATOR CUM TRANSMITTER 402" <= "INTERLOCK DB"."RO-2 SET PARAMETER"."CT-402 HH"),
                           PT := T#3S);
   IF "IEC_Timer_0_DB_87".Q THEN "INTERLOCK DB"."RO-2 PARAMETER BUFF"."CT-402 BUFF" := 0; END_IF;
END_REGION

REGION Network 29: AGLV-401A FLUSH TIME NOT USE
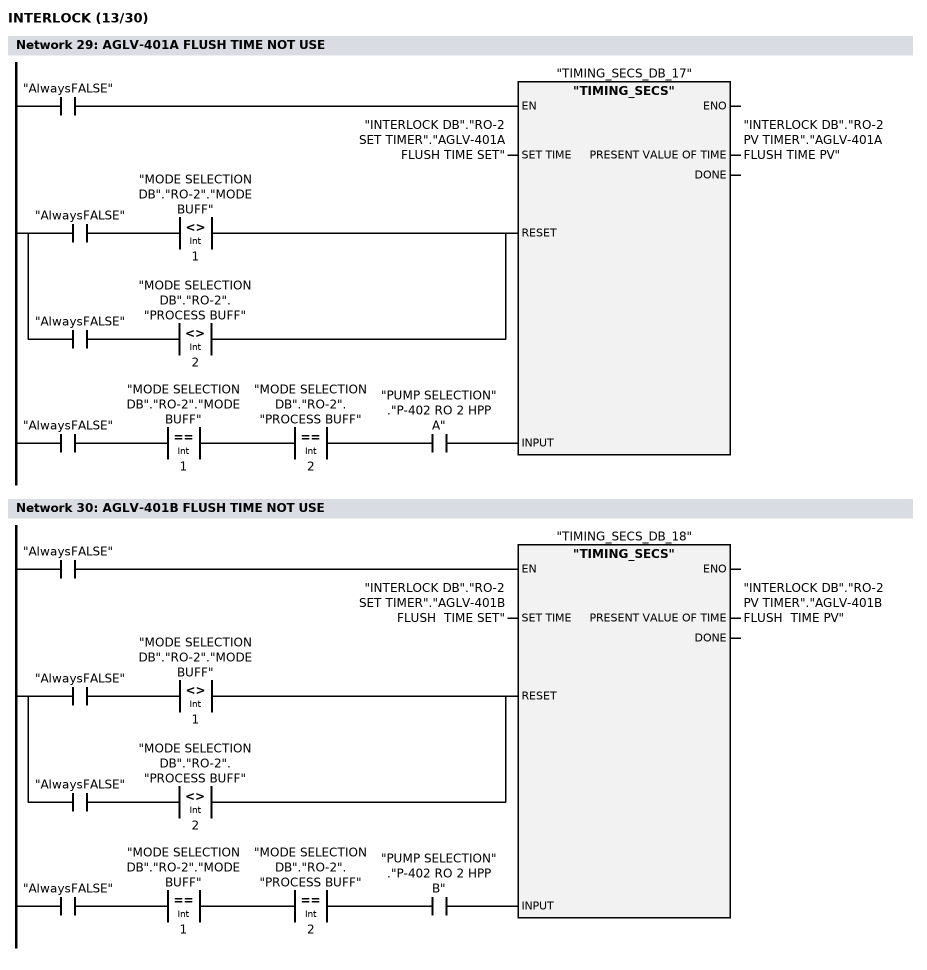
   RUNG wire#powerrail
      Contact( "AlwaysFALSE" )
      "TIMING_SECS_DB_17"(RESET := wire#w1, INPUT := wire#w2, "SET TIME" := "INTERLOCK DB"."RO-2 SET TIMER"."AGLV-401A FLUSH TIME SET", "PRESENT VALUE OF TIME" => "INTERLOCK DB"."RO-2 PV TIMER"."AGLV-401A FLUSH TIME PV", DONE =>)
   END_RUNG
   RUNG wire#powerrail
      Contact( "AlwaysFALSE" )
      { S7_Templates := "SrcType := Int" } NE_Contact(in1 := "MODE SELECTION DB"."RO-2"."MODE BUFF", in2 := 1)
   END_RUNG wire#w1
   RUNG wire#powerrail
      Contact( "AlwaysFALSE" )
      { S7_Templates := "SrcType := Int" } NE_Contact(in1 := "MODE SELECTION DB"."RO-2"."PROCESS BUFF", in2 := 2)
   END_RUNG wire#w1
   RUNG wire#powerrail
      Contact( "AlwaysFALSE" )
      { S7_Templates := "SrcType := Int" } EQ_Contact(in1 := "MODE SELECTION DB"."RO-2"."MODE BUFF", in2 := 1)
      { S7_Templates := "SrcType := Int" } EQ_Contact(in1 := "MODE SELECTION DB"."RO-2"."PROCESS BUFF", in2 := 2)
      Contact( "PUMP SELECTION"."P-402 RO 2 HPP A" )
   END_RUNG wire#w2
   // the same network as SCL:
   IF "AlwaysFALSE" THEN
       "TIMING_SECS_DB_17"("SET TIME" := "INTERLOCK DB"."RO-2 SET TIMER"."AGLV-401A FLUSH TIME SET",   // "TIMING_SECS"
                           RESET := ("AlwaysFALSE" AND ("MODE SELECTION DB"."RO-2"."MODE BUFF" <> 1)) OR ("AlwaysFALSE" AND ("MODE SELECTION DB"."RO-2"."PROCESS BUFF" <> 2)),
                           INPUT := "AlwaysFALSE" AND ("MODE SELECTION DB"."RO-2"."MODE BUFF" = 1) AND ("MODE SELECTION DB"."RO-2"."PROCESS BUFF" = 2) AND "PUMP SELECTION"."P-402 RO 2 HPP A",
                           "PRESENT VALUE OF TIME" => "INTERLOCK DB"."RO-2 PV TIMER"."AGLV-401A FLUSH TIME PV");
   END_IF;
END_REGION

REGION Network 30: AGLV-401B FLUSH TIME NOT USE
   RUNG wire#powerrail
      Contact( "AlwaysFALSE" )
      "TIMING_SECS_DB_18"(RESET := wire#w1, INPUT := wire#w2, "SET TIME" := "INTERLOCK DB"."RO-2 SET TIMER"."AGLV-401B FLUSH  TIME SET", "PRESENT VALUE OF TIME" => "INTERLOCK DB"."RO-2 PV TIMER"."AGLV-401B FLUSH  TIME PV", DONE =>)
   END_RUNG
   RUNG wire#powerrail
      Contact( "AlwaysFALSE" )
      { S7_Templates := "SrcType := Int" } NE_Contact(in1 := "MODE SELECTION DB"."RO-2"."MODE BUFF", in2 := 1)
   END_RUNG wire#w1
   RUNG wire#powerrail
      Contact( "AlwaysFALSE" )
      { S7_Templates := "SrcType := Int" } NE_Contact(in1 := "MODE SELECTION DB"."RO-2"."PROCESS BUFF", in2 := 2)
   END_RUNG wire#w1
   RUNG wire#powerrail
      Contact( "AlwaysFALSE" )
      { S7_Templates := "SrcType := Int" } EQ_Contact(in1 := "MODE SELECTION DB"."RO-2"."MODE BUFF", in2 := 1)
      { S7_Templates := "SrcType := Int" } EQ_Contact(in1 := "MODE SELECTION DB"."RO-2"."PROCESS BUFF", in2 := 2)
      Contact( "PUMP SELECTION"."P-402 RO 2 HPP B" )
   END_RUNG wire#w2
   // the same network as SCL:
   IF "AlwaysFALSE" THEN
       "TIMING_SECS_DB_18"("SET TIME" := "INTERLOCK DB"."RO-2 SET TIMER"."AGLV-401B FLUSH  TIME SET",   // "TIMING_SECS"
                           RESET := ("AlwaysFALSE" AND ("MODE SELECTION DB"."RO-2"."MODE BUFF" <> 1)) OR ("AlwaysFALSE" AND ("MODE SELECTION DB"."RO-2"."PROCESS BUFF" <> 2)),
                           INPUT := "AlwaysFALSE" AND ("MODE SELECTION DB"."RO-2"."MODE BUFF" = 1) AND ("MODE SELECTION DB"."RO-2"."PROCESS BUFF" = 2) AND "PUMP SELECTION"."P-402 RO 2 HPP B",
                           "PRESENT VALUE OF TIME" => "INTERLOCK DB"."RO-2 PV TIMER"."AGLV-401B FLUSH  TIME PV");
   END_IF;
END_REGION

REGION Network 32: AUTO INTERLOCK FOR EDI ///////////////////////////////////////////////////////
END_REGION

REGION Network 33: PT501 LOW / HIGH
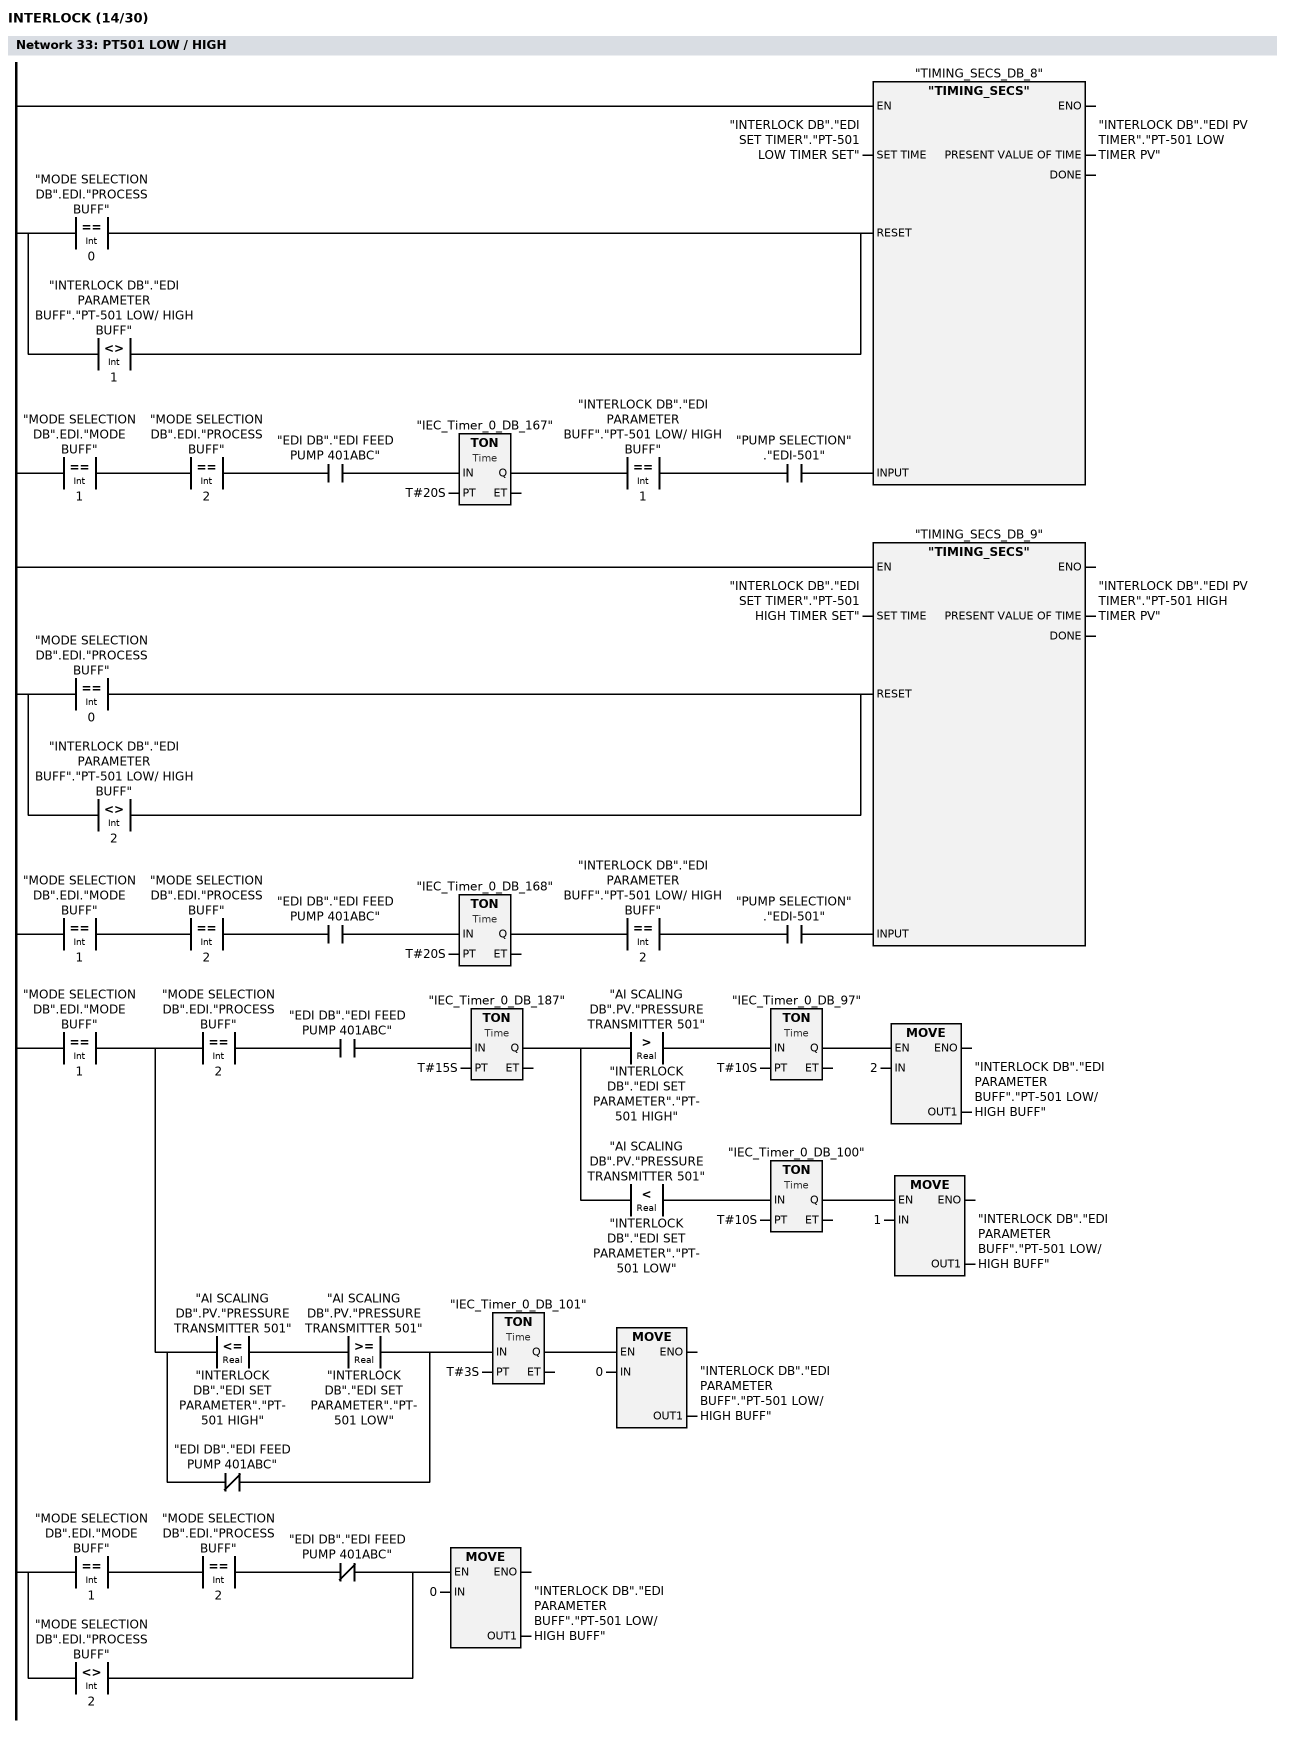
   RUNG wire#powerrail
      "TIMING_SECS_DB_8"(RESET := wire#w1, INPUT := wire#w2, "SET TIME" := "INTERLOCK DB"."EDI SET TIMER"."PT-501 LOW TIMER SET", "PRESENT VALUE OF TIME" => "INTERLOCK DB"."EDI PV TIMER"."PT-501 LOW TIMER PV", DONE =>)
   END_RUNG
   RUNG wire#powerrail
      { S7_Templates := "SrcType := Int" } EQ_Contact(in1 := "MODE SELECTION DB".EDI."PROCESS BUFF", in2 := 0)
   END_RUNG wire#w1
   RUNG wire#powerrail
      { S7_Templates := "SrcType := Int" } NE_Contact(in1 := "INTERLOCK DB"."EDI PARAMETER BUFF"."PT-501 LOW/ HIGH BUFF", in2 := 1)
   END_RUNG wire#w1
   RUNG wire#powerrail
      { S7_Templates := "SrcType := Int" } EQ_Contact(in1 := "MODE SELECTION DB".EDI."MODE BUFF", in2 := 1)
      { S7_Templates := "SrcType := Int" } EQ_Contact(in1 := "MODE SELECTION DB".EDI."PROCESS BUFF", in2 := 2)
      Contact( "EDI DB"."EDI FEED PUMP 401ABC" )
      { S7_Templates := "time_type := Time" } "IEC_Timer_0_DB_167".TON(pt := T#20S, et =>)
      { S7_Templates := "SrcType := Int" } EQ_Contact(in1 := "INTERLOCK DB"."EDI PARAMETER BUFF"."PT-501 LOW/ HIGH BUFF", in2 := 1)
      Contact( "PUMP SELECTION"."EDI-501" )
   END_RUNG wire#w2
   RUNG wire#powerrail
      "TIMING_SECS_DB_9"(RESET := wire#w3, INPUT := wire#w4, "SET TIME" := "INTERLOCK DB"."EDI SET TIMER"."PT-501 HIGH TIMER SET", "PRESENT VALUE OF TIME" => "INTERLOCK DB"."EDI PV TIMER"."PT-501 HIGH TIMER PV", DONE =>)
   END_RUNG
   RUNG wire#powerrail
      { S7_Templates := "SrcType := Int" } EQ_Contact(in1 := "MODE SELECTION DB".EDI."PROCESS BUFF", in2 := 0)
   END_RUNG wire#w3
   RUNG wire#powerrail
      { S7_Templates := "SrcType := Int" } NE_Contact(in1 := "INTERLOCK DB"."EDI PARAMETER BUFF"."PT-501 LOW/ HIGH BUFF", in2 := 2)
   END_RUNG wire#w3
   RUNG wire#powerrail
      { S7_Templates := "SrcType := Int" } EQ_Contact(in1 := "MODE SELECTION DB".EDI."MODE BUFF", in2 := 1)
      { S7_Templates := "SrcType := Int" } EQ_Contact(in1 := "MODE SELECTION DB".EDI."PROCESS BUFF", in2 := 2)
      Contact( "EDI DB"."EDI FEED PUMP 401ABC" )
      { S7_Templates := "time_type := Time" } "IEC_Timer_0_DB_168".TON(pt := T#20S, et =>)
      { S7_Templates := "SrcType := Int" } EQ_Contact(in1 := "INTERLOCK DB"."EDI PARAMETER BUFF"."PT-501 LOW/ HIGH BUFF", in2 := 2)
      Contact( "PUMP SELECTION"."EDI-501" )
   END_RUNG wire#w4
   RUNG wire#powerrail
      { S7_Templates := "SrcType := Int" } EQ_Contact(in1 := "MODE SELECTION DB".EDI."MODE BUFF", in2 := 1)
      wire#w5
      { S7_Templates := "SrcType := Int" } EQ_Contact(in1 := "MODE SELECTION DB".EDI."PROCESS BUFF", in2 := 2)
      Contact( "EDI DB"."EDI FEED PUMP 401ABC" )
      { S7_Templates := "time_type := Time" } "IEC_Timer_0_DB_187".TON(pt := T#15S, et =>)
      wire#w6
      { S7_Templates := "SrcType := Real" } GT_Contact(in1 := "AI SCALING DB".PV."PRESSURE TRANSMITTER 501", in2 := "INTERLOCK DB"."EDI SET PARAMETER"."PT-501 HIGH")
      { S7_Templates := "time_type := Time" } "IEC_Timer_0_DB_97".TON(pt := T#10S, et =>)
      Move(in := 2, out1 => "INTERLOCK DB"."EDI PARAMETER BUFF"."PT-501 LOW/ HIGH BUFF")
   END_RUNG
   RUNG wire#w6
      { S7_Templates := "SrcType := Real" } LT_Contact(in1 := "AI SCALING DB".PV."PRESSURE TRANSMITTER 501", in2 := "INTERLOCK DB"."EDI SET PARAMETER"."PT-501 LOW")
      { S7_Templates := "time_type := Time" } "IEC_Timer_0_DB_100".TON(pt := T#10S, et =>)
      Move(in := 1, out1 => "INTERLOCK DB"."EDI PARAMETER BUFF"."PT-501 LOW/ HIGH BUFF")
   END_RUNG
   RUNG wire#w5
      { S7_Templates := "SrcType := Real" } LE_Contact(in1 := "AI SCALING DB".PV."PRESSURE TRANSMITTER 501", in2 := "INTERLOCK DB"."EDI SET PARAMETER"."PT-501 HIGH")
      { S7_Templates := "SrcType := Real" } GE_Contact(in1 := "AI SCALING DB".PV."PRESSURE TRANSMITTER 501", in2 := "INTERLOCK DB"."EDI SET PARAMETER"."PT-501 LOW")
      wire#w7
      { S7_Templates := "time_type := Time" } "IEC_Timer_0_DB_101".TON(pt := T#3S, et =>)
      Move(in := 0, out1 => "INTERLOCK DB"."EDI PARAMETER BUFF"."PT-501 LOW/ HIGH BUFF")
   END_RUNG
   RUNG wire#w5
      I_Contact( "EDI DB"."EDI FEED PUMP 401ABC" )
   END_RUNG wire#w7
   RUNG wire#powerrail
      { S7_Templates := "SrcType := Int" } EQ_Contact(in1 := "MODE SELECTION DB".EDI."MODE BUFF", in2 := 1)
      { S7_Templates := "SrcType := Int" } EQ_Contact(in1 := "MODE SELECTION DB".EDI."PROCESS BUFF", in2 := 2)
      I_Contact( "EDI DB"."EDI FEED PUMP 401ABC" )
      wire#w8
      Move(in := 0, out1 => "INTERLOCK DB"."EDI PARAMETER BUFF"."PT-501 LOW/ HIGH BUFF")
   END_RUNG
   RUNG wire#powerrail
      { S7_Templates := "SrcType := Int" } NE_Contact(in1 := "MODE SELECTION DB".EDI."PROCESS BUFF", in2 := 2)
   END_RUNG wire#w8
   // the same network as SCL:
   "IEC_Timer_0_DB_167".TON(IN := ("MODE SELECTION DB".EDI."MODE BUFF" = 1) AND ("MODE SELECTION DB".EDI."PROCESS BUFF" = 2) AND "EDI DB"."EDI FEED PUMP 401ABC",
                           PT := T#20S);
   "TIMING_SECS_DB_8"("SET TIME" := "INTERLOCK DB"."EDI SET TIMER"."PT-501 LOW TIMER SET",   // "TIMING_SECS"
                      RESET := ("MODE SELECTION DB".EDI."PROCESS BUFF" = 0) OR ("INTERLOCK DB"."EDI PARAMETER BUFF"."PT-501 LOW/ HIGH BUFF" <> 1),
                      INPUT := "IEC_Timer_0_DB_167".Q AND ("INTERLOCK DB"."EDI PARAMETER BUFF"."PT-501 LOW/ HIGH BUFF" = 1) AND "PUMP SELECTION"."EDI-501",
                      "PRESENT VALUE OF TIME" => "INTERLOCK DB"."EDI PV TIMER"."PT-501 LOW TIMER PV");
   "IEC_Timer_0_DB_168".TON(IN := ("MODE SELECTION DB".EDI."MODE BUFF" = 1) AND ("MODE SELECTION DB".EDI."PROCESS BUFF" = 2) AND "EDI DB"."EDI FEED PUMP 401ABC",
                           PT := T#20S);
   "TIMING_SECS_DB_9"("SET TIME" := "INTERLOCK DB"."EDI SET TIMER"."PT-501 HIGH TIMER SET",   // "TIMING_SECS"
                      RESET := ("MODE SELECTION DB".EDI."PROCESS BUFF" = 0) OR ("INTERLOCK DB"."EDI PARAMETER BUFF"."PT-501 LOW/ HIGH BUFF" <> 2),
                      INPUT := "IEC_Timer_0_DB_168".Q AND ("INTERLOCK DB"."EDI PARAMETER BUFF"."PT-501 LOW/ HIGH BUFF" = 2) AND "PUMP SELECTION"."EDI-501",
                      "PRESENT VALUE OF TIME" => "INTERLOCK DB"."EDI PV TIMER"."PT-501 HIGH TIMER PV");
   #_w1 := "MODE SELECTION DB".EDI."MODE BUFF" = 1;
   "IEC_Timer_0_DB_187".TON(IN := #_w1 AND ("MODE SELECTION DB".EDI."PROCESS BUFF" = 2) AND "EDI DB"."EDI FEED PUMP 401ABC",
                           PT := T#15S);
   "IEC_Timer_0_DB_97".TON(IN := "IEC_Timer_0_DB_187".Q AND ("AI SCALING DB".PV."PRESSURE TRANSMITTER 501" > "INTERLOCK DB"."EDI SET PARAMETER"."PT-501 HIGH"),
                           PT := T#10S);
   IF "IEC_Timer_0_DB_97".Q THEN "INTERLOCK DB"."EDI PARAMETER BUFF"."PT-501 LOW/ HIGH BUFF" := 2; END_IF;
   "IEC_Timer_0_DB_100".TON(IN := "IEC_Timer_0_DB_187".Q AND ("AI SCALING DB".PV."PRESSURE TRANSMITTER 501" < "INTERLOCK DB"."EDI SET PARAMETER"."PT-501 LOW"),
                           PT := T#10S);
   IF "IEC_Timer_0_DB_100".Q THEN "INTERLOCK DB"."EDI PARAMETER BUFF"."PT-501 LOW/ HIGH BUFF" := 1; END_IF;
   "IEC_Timer_0_DB_101".TON(IN := #_w1 AND ((("AI SCALING DB".PV."PRESSURE TRANSMITTER 501" <= "INTERLOCK DB"."EDI SET PARAMETER"."PT-501 HIGH") AND ("AI SCALING DB".PV."PRESSURE TRANSMITTER 501" >= "INTERLOCK DB"."EDI SET PARAMETER"."PT-501 LOW")) OR NOT "EDI DB"."EDI FEED PUMP 401ABC"),
                           PT := T#3S);
   IF "IEC_Timer_0_DB_101".Q THEN "INTERLOCK DB"."EDI PARAMETER BUFF"."PT-501 LOW/ HIGH BUFF" := 0; END_IF;
   IF (("MODE SELECTION DB".EDI."MODE BUFF" = 1) AND ("MODE SELECTION DB".EDI."PROCESS BUFF" = 2) AND NOT "EDI DB"."EDI FEED PUMP 401ABC") OR ("MODE SELECTION DB".EDI."PROCESS BUFF" <> 2) THEN
       "INTERLOCK DB"."EDI PARAMETER BUFF"."PT-501 LOW/ HIGH BUFF" := 0;
   END_IF;
END_REGION

REGION Network 34: PT502 LOW / HIGH
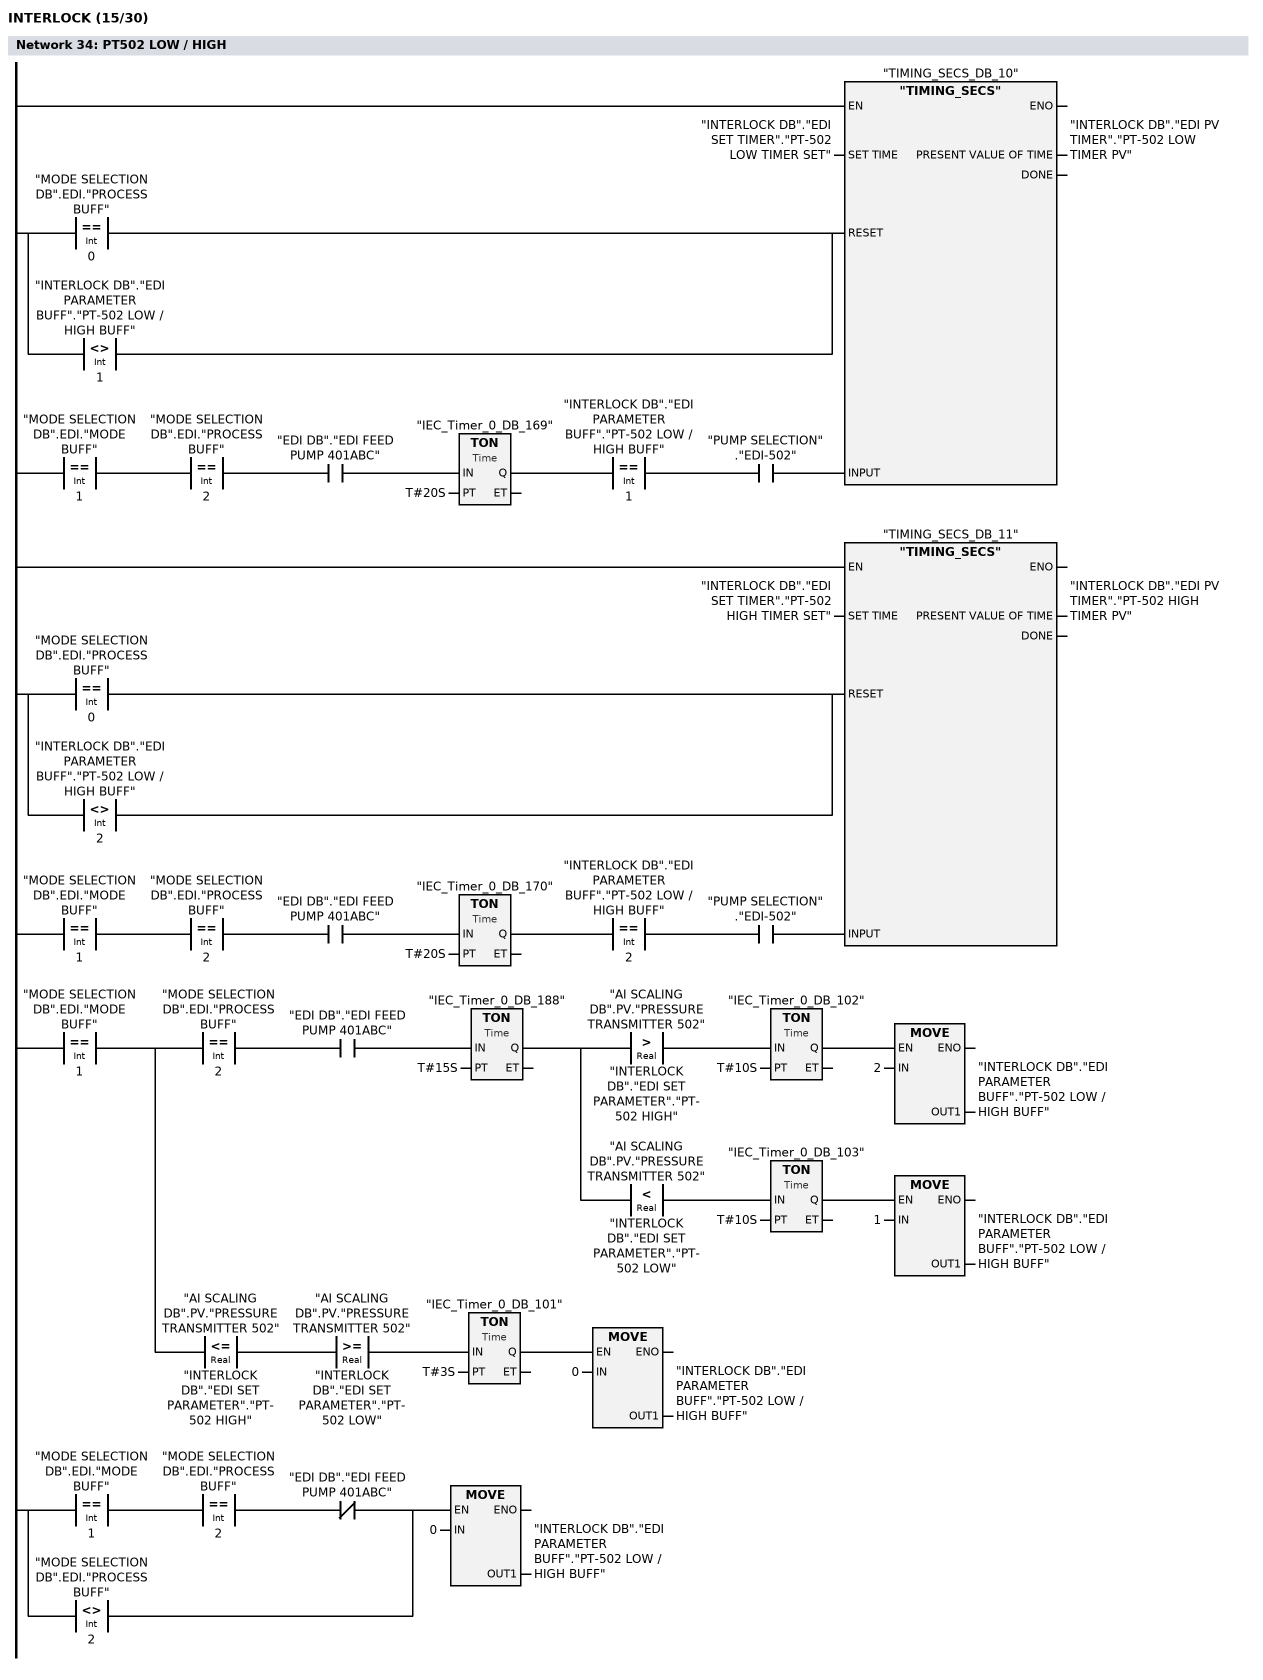
   RUNG wire#powerrail
      "TIMING_SECS_DB_10"(RESET := wire#w1, INPUT := wire#w2, "SET TIME" := "INTERLOCK DB"."EDI SET TIMER"."PT-502 LOW TIMER SET", "PRESENT VALUE OF TIME" => "INTERLOCK DB"."EDI PV TIMER"."PT-502 LOW TIMER PV", DONE =>)
   END_RUNG
   RUNG wire#powerrail
      { S7_Templates := "SrcType := Int" } EQ_Contact(in1 := "MODE SELECTION DB".EDI."PROCESS BUFF", in2 := 0)
   END_RUNG wire#w1
   RUNG wire#powerrail
      { S7_Templates := "SrcType := Int" } NE_Contact(in1 := "INTERLOCK DB"."EDI PARAMETER BUFF"."PT-502 LOW / HIGH BUFF", in2 := 1)
   END_RUNG wire#w1
   RUNG wire#powerrail
      { S7_Templates := "SrcType := Int" } EQ_Contact(in1 := "MODE SELECTION DB".EDI."MODE BUFF", in2 := 1)
      { S7_Templates := "SrcType := Int" } EQ_Contact(in1 := "MODE SELECTION DB".EDI."PROCESS BUFF", in2 := 2)
      Contact( "EDI DB"."EDI FEED PUMP 401ABC" )
      { S7_Templates := "time_type := Time" } "IEC_Timer_0_DB_169".TON(pt := T#20S, et =>)
      { S7_Templates := "SrcType := Int" } EQ_Contact(in1 := "INTERLOCK DB"."EDI PARAMETER BUFF"."PT-502 LOW / HIGH BUFF", in2 := 1)
      Contact( "PUMP SELECTION"."EDI-502" )
   END_RUNG wire#w2
   RUNG wire#powerrail
      "TIMING_SECS_DB_11"(RESET := wire#w3, INPUT := wire#w4, "SET TIME" := "INTERLOCK DB"."EDI SET TIMER"."PT-502 HIGH TIMER SET", "PRESENT VALUE OF TIME" => "INTERLOCK DB"."EDI PV TIMER"."PT-502 HIGH TIMER PV", DONE =>)
   END_RUNG
   RUNG wire#powerrail
      { S7_Templates := "SrcType := Int" } EQ_Contact(in1 := "MODE SELECTION DB".EDI."PROCESS BUFF", in2 := 0)
   END_RUNG wire#w3
   RUNG wire#powerrail
      { S7_Templates := "SrcType := Int" } NE_Contact(in1 := "INTERLOCK DB"."EDI PARAMETER BUFF"."PT-502 LOW / HIGH BUFF", in2 := 2)
   END_RUNG wire#w3
   RUNG wire#powerrail
      { S7_Templates := "SrcType := Int" } EQ_Contact(in1 := "MODE SELECTION DB".EDI."MODE BUFF", in2 := 1)
      { S7_Templates := "SrcType := Int" } EQ_Contact(in1 := "MODE SELECTION DB".EDI."PROCESS BUFF", in2 := 2)
      Contact( "EDI DB"."EDI FEED PUMP 401ABC" )
      { S7_Templates := "time_type := Time" } "IEC_Timer_0_DB_170".TON(pt := T#20S, et =>)
      { S7_Templates := "SrcType := Int" } EQ_Contact(in1 := "INTERLOCK DB"."EDI PARAMETER BUFF"."PT-502 LOW / HIGH BUFF", in2 := 2)
      Contact( "PUMP SELECTION"."EDI-502" )
   END_RUNG wire#w4
   RUNG wire#powerrail
      { S7_Templates := "SrcType := Int" } EQ_Contact(in1 := "MODE SELECTION DB".EDI."MODE BUFF", in2 := 1)
      wire#w5
      { S7_Templates := "SrcType := Int" } EQ_Contact(in1 := "MODE SELECTION DB".EDI."PROCESS BUFF", in2 := 2)
      Contact( "EDI DB"."EDI FEED PUMP 401ABC" )
      { S7_Templates := "time_type := Time" } "IEC_Timer_0_DB_188".TON(pt := T#15S, et =>)
      wire#w6
      { S7_Templates := "SrcType := Real" } GT_Contact(in1 := "AI SCALING DB".PV."PRESSURE TRANSMITTER 502", in2 := "INTERLOCK DB"."EDI SET PARAMETER"."PT-502 HIGH")
      { S7_Templates := "time_type := Time" } "IEC_Timer_0_DB_102".TON(pt := T#10S, et =>)
      Move(in := 2, out1 => "INTERLOCK DB"."EDI PARAMETER BUFF"."PT-502 LOW / HIGH BUFF")
   END_RUNG
   RUNG wire#w6
      { S7_Templates := "SrcType := Real" } LT_Contact(in1 := "AI SCALING DB".PV."PRESSURE TRANSMITTER 502", in2 := "INTERLOCK DB"."EDI SET PARAMETER"."PT-502 LOW")
      { S7_Templates := "time_type := Time" } "IEC_Timer_0_DB_103".TON(pt := T#10S, et =>)
      Move(in := 1, out1 => "INTERLOCK DB"."EDI PARAMETER BUFF"."PT-502 LOW / HIGH BUFF")
   END_RUNG
   RUNG wire#w5
      { S7_Templates := "SrcType := Real" } LE_Contact(in1 := "AI SCALING DB".PV."PRESSURE TRANSMITTER 502", in2 := "INTERLOCK DB"."EDI SET PARAMETER"."PT-502 HIGH")
      { S7_Templates := "SrcType := Real" } GE_Contact(in1 := "AI SCALING DB".PV."PRESSURE TRANSMITTER 502", in2 := "INTERLOCK DB"."EDI SET PARAMETER"."PT-502 LOW")
      { S7_Templates := "time_type := Time" } "IEC_Timer_0_DB_101".TON(pt := T#3S, et =>)
      Move(in := 0, out1 => "INTERLOCK DB"."EDI PARAMETER BUFF"."PT-502 LOW / HIGH BUFF")
   END_RUNG
   RUNG wire#powerrail
      { S7_Templates := "SrcType := Int" } EQ_Contact(in1 := "MODE SELECTION DB".EDI."MODE BUFF", in2 := 1)
      { S7_Templates := "SrcType := Int" } EQ_Contact(in1 := "MODE SELECTION DB".EDI."PROCESS BUFF", in2 := 2)
      I_Contact( "EDI DB"."EDI FEED PUMP 401ABC" )
      wire#w7
      Move(in := 0, out1 => "INTERLOCK DB"."EDI PARAMETER BUFF"."PT-502 LOW / HIGH BUFF")
   END_RUNG
   RUNG wire#powerrail
      { S7_Templates := "SrcType := Int" } NE_Contact(in1 := "MODE SELECTION DB".EDI."PROCESS BUFF", in2 := 2)
   END_RUNG wire#w7
   // the same network as SCL:
   "IEC_Timer_0_DB_169".TON(IN := ("MODE SELECTION DB".EDI."MODE BUFF" = 1) AND ("MODE SELECTION DB".EDI."PROCESS BUFF" = 2) AND "EDI DB"."EDI FEED PUMP 401ABC",
                           PT := T#20S);
   "TIMING_SECS_DB_10"("SET TIME" := "INTERLOCK DB"."EDI SET TIMER"."PT-502 LOW TIMER SET",   // "TIMING_SECS"
                       RESET := ("MODE SELECTION DB".EDI."PROCESS BUFF" = 0) OR ("INTERLOCK DB"."EDI PARAMETER BUFF"."PT-502 LOW / HIGH BUFF" <> 1),
                       INPUT := "IEC_Timer_0_DB_169".Q AND ("INTERLOCK DB"."EDI PARAMETER BUFF"."PT-502 LOW / HIGH BUFF" = 1) AND "PUMP SELECTION"."EDI-502",
                       "PRESENT VALUE OF TIME" => "INTERLOCK DB"."EDI PV TIMER"."PT-502 LOW TIMER PV");
   "IEC_Timer_0_DB_170".TON(IN := ("MODE SELECTION DB".EDI."MODE BUFF" = 1) AND ("MODE SELECTION DB".EDI."PROCESS BUFF" = 2) AND "EDI DB"."EDI FEED PUMP 401ABC",
                           PT := T#20S);
   "TIMING_SECS_DB_11"("SET TIME" := "INTERLOCK DB"."EDI SET TIMER"."PT-502 HIGH TIMER SET",   // "TIMING_SECS"
                       RESET := ("MODE SELECTION DB".EDI."PROCESS BUFF" = 0) OR ("INTERLOCK DB"."EDI PARAMETER BUFF"."PT-502 LOW / HIGH BUFF" <> 2),
                       INPUT := "IEC_Timer_0_DB_170".Q AND ("INTERLOCK DB"."EDI PARAMETER BUFF"."PT-502 LOW / HIGH BUFF" = 2) AND "PUMP SELECTION"."EDI-502",
                       "PRESENT VALUE OF TIME" => "INTERLOCK DB"."EDI PV TIMER"."PT-502 HIGH TIMER PV");
   #_w1 := "MODE SELECTION DB".EDI."MODE BUFF" = 1;
   "IEC_Timer_0_DB_188".TON(IN := #_w1 AND ("MODE SELECTION DB".EDI."PROCESS BUFF" = 2) AND "EDI DB"."EDI FEED PUMP 401ABC",
                           PT := T#15S);
   "IEC_Timer_0_DB_102".TON(IN := "IEC_Timer_0_DB_188".Q AND ("AI SCALING DB".PV."PRESSURE TRANSMITTER 502" > "INTERLOCK DB"."EDI SET PARAMETER"."PT-502 HIGH"),
                           PT := T#10S);
   IF "IEC_Timer_0_DB_102".Q THEN "INTERLOCK DB"."EDI PARAMETER BUFF"."PT-502 LOW / HIGH BUFF" := 2; END_IF;
   "IEC_Timer_0_DB_103".TON(IN := "IEC_Timer_0_DB_188".Q AND ("AI SCALING DB".PV."PRESSURE TRANSMITTER 502" < "INTERLOCK DB"."EDI SET PARAMETER"."PT-502 LOW"),
                           PT := T#10S);
   IF "IEC_Timer_0_DB_103".Q THEN "INTERLOCK DB"."EDI PARAMETER BUFF"."PT-502 LOW / HIGH BUFF" := 1; END_IF;
   "IEC_Timer_0_DB_101".TON(IN := #_w1 AND ("AI SCALING DB".PV."PRESSURE TRANSMITTER 502" <= "INTERLOCK DB"."EDI SET PARAMETER"."PT-502 HIGH") AND ("AI SCALING DB".PV."PRESSURE TRANSMITTER 502" >= "INTERLOCK DB"."EDI SET PARAMETER"."PT-502 LOW"),
                           PT := T#3S);
   IF "IEC_Timer_0_DB_101".Q THEN "INTERLOCK DB"."EDI PARAMETER BUFF"."PT-502 LOW / HIGH BUFF" := 0; END_IF;
   IF (("MODE SELECTION DB".EDI."MODE BUFF" = 1) AND ("MODE SELECTION DB".EDI."PROCESS BUFF" = 2) AND NOT "EDI DB"."EDI FEED PUMP 401ABC") OR ("MODE SELECTION DB".EDI."PROCESS BUFF" <> 2) THEN
       "INTERLOCK DB"."EDI PARAMETER BUFF"."PT-502 LOW / HIGH BUFF" := 0;
   END_IF;
END_REGION

REGION Network 35: PT503 HIGH
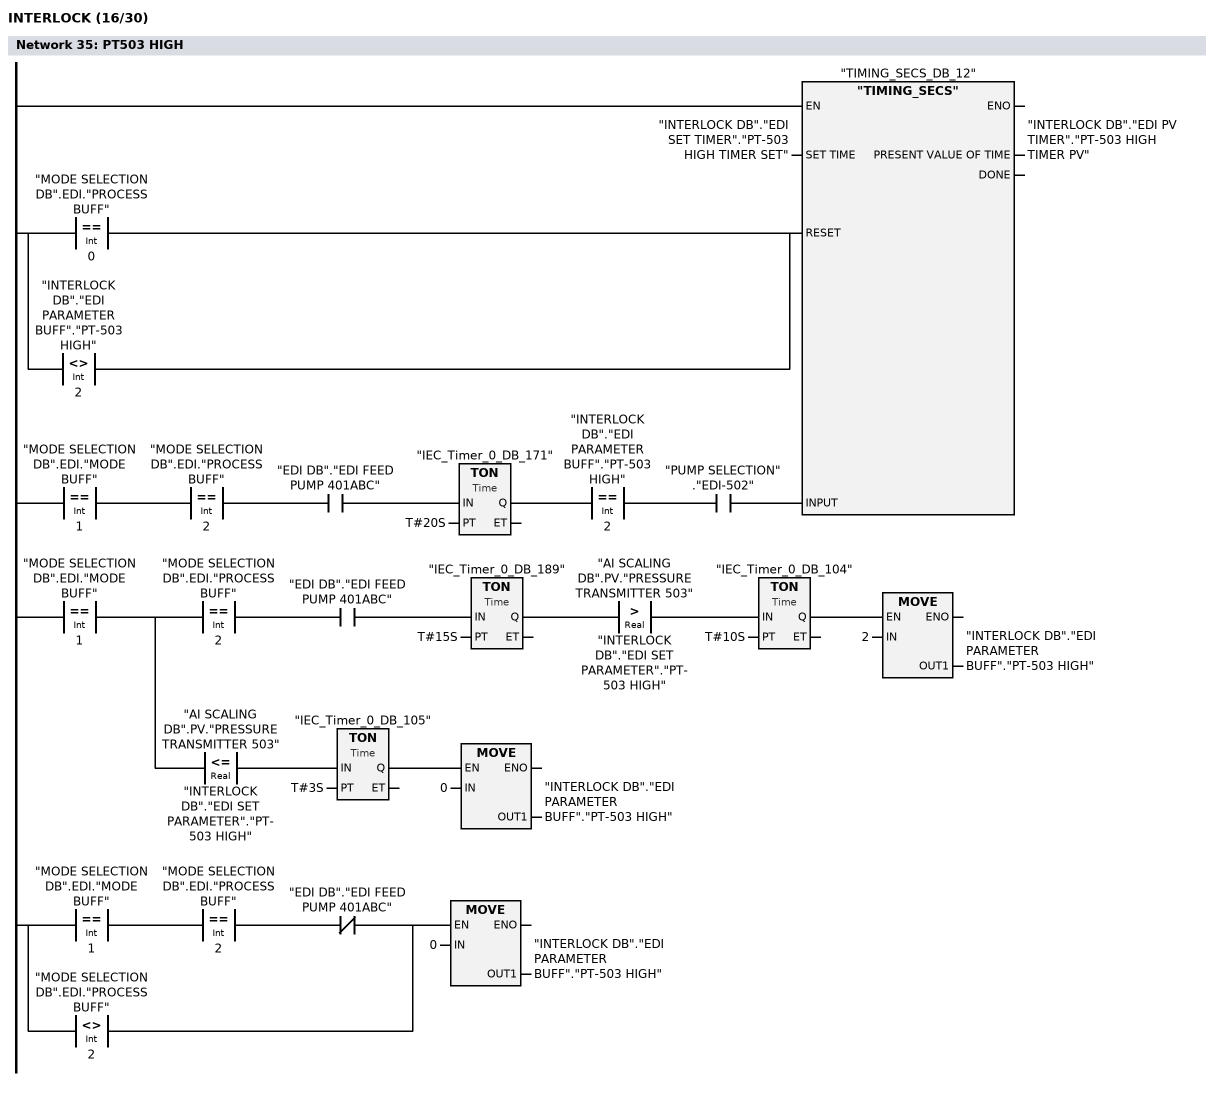
   RUNG wire#powerrail
      "TIMING_SECS_DB_12"(RESET := wire#w1, INPUT := wire#w2, "SET TIME" := "INTERLOCK DB"."EDI SET TIMER"."PT-503 HIGH TIMER SET", "PRESENT VALUE OF TIME" => "INTERLOCK DB"."EDI PV TIMER"."PT-503 HIGH TIMER PV", DONE =>)
   END_RUNG
   RUNG wire#powerrail
      { S7_Templates := "SrcType := Int" } EQ_Contact(in1 := "MODE SELECTION DB".EDI."PROCESS BUFF", in2 := 0)
   END_RUNG wire#w1
   RUNG wire#powerrail
      { S7_Templates := "SrcType := Int" } NE_Contact(in1 := "INTERLOCK DB"."EDI PARAMETER BUFF"."PT-503 HIGH", in2 := 2)
   END_RUNG wire#w1
   RUNG wire#powerrail
      { S7_Templates := "SrcType := Int" } EQ_Contact(in1 := "MODE SELECTION DB".EDI."MODE BUFF", in2 := 1)
      { S7_Templates := "SrcType := Int" } EQ_Contact(in1 := "MODE SELECTION DB".EDI."PROCESS BUFF", in2 := 2)
      Contact( "EDI DB"."EDI FEED PUMP 401ABC" )
      { S7_Templates := "time_type := Time" } "IEC_Timer_0_DB_171".TON(pt := T#20S, et =>)
      { S7_Templates := "SrcType := Int" } EQ_Contact(in1 := "INTERLOCK DB"."EDI PARAMETER BUFF"."PT-503 HIGH", in2 := 2)
      Contact( "PUMP SELECTION"."EDI-502" )
   END_RUNG wire#w2
   RUNG wire#powerrail
      { S7_Templates := "SrcType := Int" } EQ_Contact(in1 := "MODE SELECTION DB".EDI."MODE BUFF", in2 := 1)
      wire#w3
      { S7_Templates := "SrcType := Int" } EQ_Contact(in1 := "MODE SELECTION DB".EDI."PROCESS BUFF", in2 := 2)
      Contact( "EDI DB"."EDI FEED PUMP 401ABC" )
      { S7_Templates := "time_type := Time" } "IEC_Timer_0_DB_189".TON(pt := T#15S, et =>)
      { S7_Templates := "SrcType := Real" } GT_Contact(in1 := "AI SCALING DB".PV."PRESSURE TRANSMITTER 503", in2 := "INTERLOCK DB"."EDI SET PARAMETER"."PT-503 HIGH")
      { S7_Templates := "time_type := Time" } "IEC_Timer_0_DB_104".TON(pt := T#10S, et =>)
      Move(in := 2, out1 => "INTERLOCK DB"."EDI PARAMETER BUFF"."PT-503 HIGH")
   END_RUNG
   RUNG wire#w3
      { S7_Templates := "SrcType := Real" } LE_Contact(in1 := "AI SCALING DB".PV."PRESSURE TRANSMITTER 503", in2 := "INTERLOCK DB"."EDI SET PARAMETER"."PT-503 HIGH")
      { S7_Templates := "time_type := Time" } "IEC_Timer_0_DB_105".TON(pt := T#3S, et =>)
      Move(in := 0, out1 => "INTERLOCK DB"."EDI PARAMETER BUFF"."PT-503 HIGH")
   END_RUNG
   RUNG wire#powerrail
      { S7_Templates := "SrcType := Int" } EQ_Contact(in1 := "MODE SELECTION DB".EDI."MODE BUFF", in2 := 1)
      { S7_Templates := "SrcType := Int" } EQ_Contact(in1 := "MODE SELECTION DB".EDI."PROCESS BUFF", in2 := 2)
      I_Contact( "EDI DB"."EDI FEED PUMP 401ABC" )
      wire#w4
      Move(in := 0, out1 => "INTERLOCK DB"."EDI PARAMETER BUFF"."PT-503 HIGH")
   END_RUNG
   RUNG wire#powerrail
      { S7_Templates := "SrcType := Int" } NE_Contact(in1 := "MODE SELECTION DB".EDI."PROCESS BUFF", in2 := 2)
   END_RUNG wire#w4
   // the same network as SCL:
   "IEC_Timer_0_DB_171".TON(IN := ("MODE SELECTION DB".EDI."MODE BUFF" = 1) AND ("MODE SELECTION DB".EDI."PROCESS BUFF" = 2) AND "EDI DB"."EDI FEED PUMP 401ABC",
                           PT := T#20S);
   "TIMING_SECS_DB_12"("SET TIME" := "INTERLOCK DB"."EDI SET TIMER"."PT-503 HIGH TIMER SET",   // "TIMING_SECS"
                       RESET := ("MODE SELECTION DB".EDI."PROCESS BUFF" = 0) OR ("INTERLOCK DB"."EDI PARAMETER BUFF"."PT-503 HIGH" <> 2),
                       INPUT := "IEC_Timer_0_DB_171".Q AND ("INTERLOCK DB"."EDI PARAMETER BUFF"."PT-503 HIGH" = 2) AND "PUMP SELECTION"."EDI-502",
                       "PRESENT VALUE OF TIME" => "INTERLOCK DB"."EDI PV TIMER"."PT-503 HIGH TIMER PV");
   #_w1 := "MODE SELECTION DB".EDI."MODE BUFF" = 1;
   "IEC_Timer_0_DB_189".TON(IN := #_w1 AND ("MODE SELECTION DB".EDI."PROCESS BUFF" = 2) AND "EDI DB"."EDI FEED PUMP 401ABC",
                           PT := T#15S);
   "IEC_Timer_0_DB_104".TON(IN := "IEC_Timer_0_DB_189".Q AND ("AI SCALING DB".PV."PRESSURE TRANSMITTER 503" > "INTERLOCK DB"."EDI SET PARAMETER"."PT-503 HIGH"),
                           PT := T#10S);
   IF "IEC_Timer_0_DB_104".Q THEN "INTERLOCK DB"."EDI PARAMETER BUFF"."PT-503 HIGH" := 2; END_IF;
   "IEC_Timer_0_DB_105".TON(IN := #_w1 AND ("AI SCALING DB".PV."PRESSURE TRANSMITTER 503" <= "INTERLOCK DB"."EDI SET PARAMETER"."PT-503 HIGH"),
                           PT := T#3S);
   IF "IEC_Timer_0_DB_105".Q THEN "INTERLOCK DB"."EDI PARAMETER BUFF"."PT-503 HIGH" := 0; END_IF;
   IF (("MODE SELECTION DB".EDI."MODE BUFF" = 1) AND ("MODE SELECTION DB".EDI."PROCESS BUFF" = 2) AND NOT "EDI DB"."EDI FEED PUMP 401ABC") OR ("MODE SELECTION DB".EDI."PROCESS BUFF" <> 2) THEN
       "INTERLOCK DB"."EDI PARAMETER BUFF"."PT-503 HIGH" := 0;
   END_IF;
END_REGION

REGION Network 36: PT504 HIGH
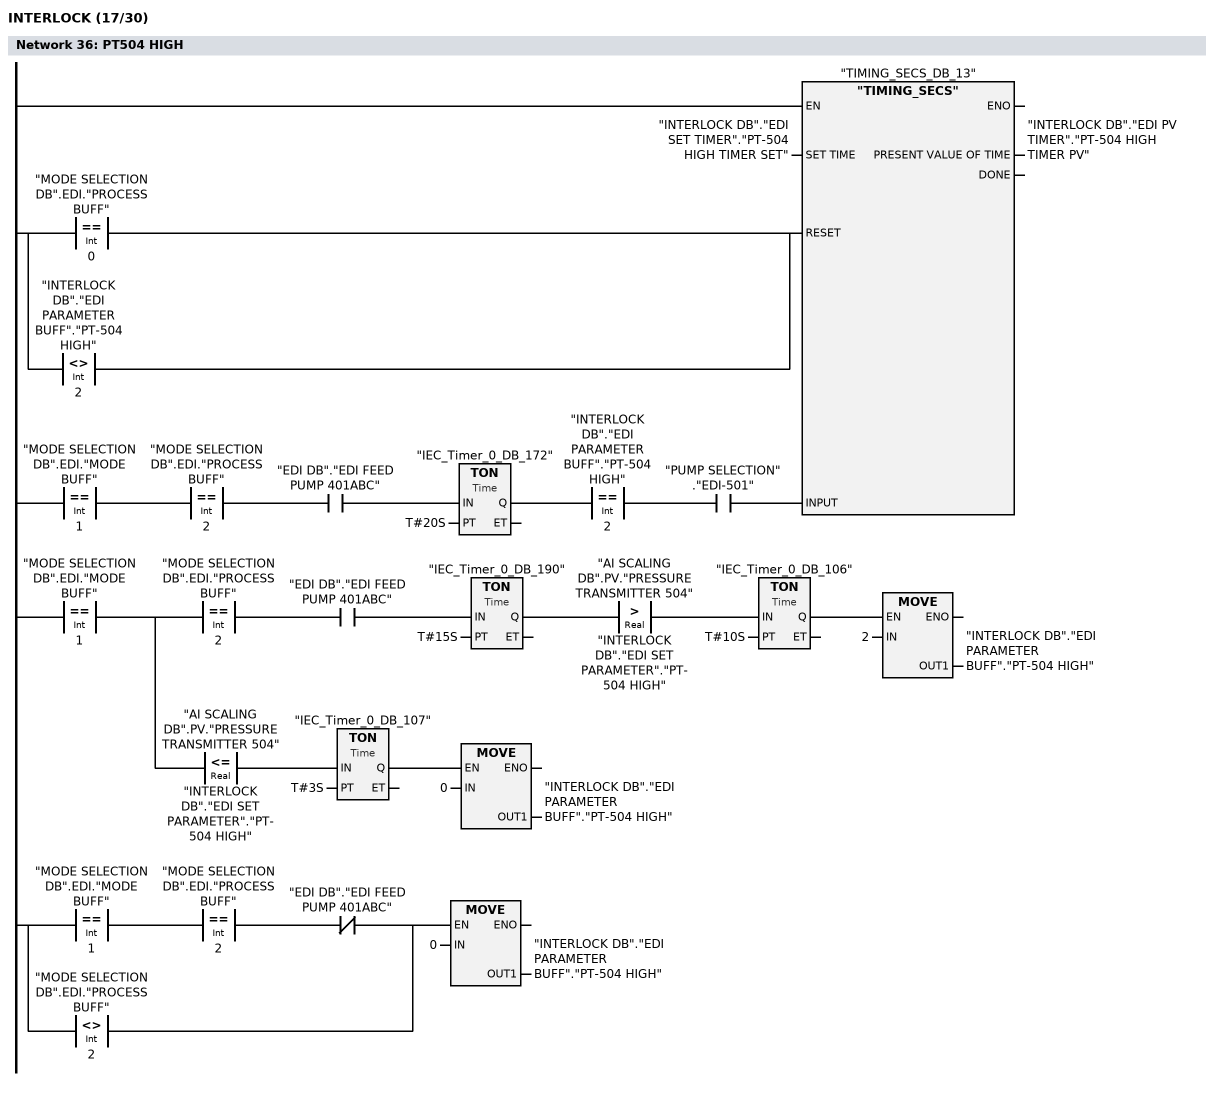
   RUNG wire#powerrail
      "TIMING_SECS_DB_13"(RESET := wire#w1, INPUT := wire#w2, "SET TIME" := "INTERLOCK DB"."EDI SET TIMER"."PT-504 HIGH TIMER SET", "PRESENT VALUE OF TIME" => "INTERLOCK DB"."EDI PV TIMER"."PT-504 HIGH TIMER PV", DONE =>)
   END_RUNG
   RUNG wire#powerrail
      { S7_Templates := "SrcType := Int" } EQ_Contact(in1 := "MODE SELECTION DB".EDI."PROCESS BUFF", in2 := 0)
   END_RUNG wire#w1
   RUNG wire#powerrail
      { S7_Templates := "SrcType := Int" } NE_Contact(in1 := "INTERLOCK DB"."EDI PARAMETER BUFF"."PT-504 HIGH", in2 := 2)
   END_RUNG wire#w1
   RUNG wire#powerrail
      { S7_Templates := "SrcType := Int" } EQ_Contact(in1 := "MODE SELECTION DB".EDI."MODE BUFF", in2 := 1)
      { S7_Templates := "SrcType := Int" } EQ_Contact(in1 := "MODE SELECTION DB".EDI."PROCESS BUFF", in2 := 2)
      Contact( "EDI DB"."EDI FEED PUMP 401ABC" )
      { S7_Templates := "time_type := Time" } "IEC_Timer_0_DB_172".TON(pt := T#20S, et =>)
      { S7_Templates := "SrcType := Int" } EQ_Contact(in1 := "INTERLOCK DB"."EDI PARAMETER BUFF"."PT-504 HIGH", in2 := 2)
      Contact( "PUMP SELECTION"."EDI-501" )
   END_RUNG wire#w2
   RUNG wire#powerrail
      { S7_Templates := "SrcType := Int" } EQ_Contact(in1 := "MODE SELECTION DB".EDI."MODE BUFF", in2 := 1)
      wire#w3
      { S7_Templates := "SrcType := Int" } EQ_Contact(in1 := "MODE SELECTION DB".EDI."PROCESS BUFF", in2 := 2)
      Contact( "EDI DB"."EDI FEED PUMP 401ABC" )
      { S7_Templates := "time_type := Time" } "IEC_Timer_0_DB_190".TON(pt := T#15S, et =>)
      { S7_Templates := "SrcType := Real" } GT_Contact(in1 := "AI SCALING DB".PV."PRESSURE TRANSMITTER 504", in2 := "INTERLOCK DB"."EDI SET PARAMETER"."PT-504 HIGH")
      { S7_Templates := "time_type := Time" } "IEC_Timer_0_DB_106".TON(pt := T#10S, et =>)
      Move(in := 2, out1 => "INTERLOCK DB"."EDI PARAMETER BUFF"."PT-504 HIGH")
   END_RUNG
   RUNG wire#w3
      { S7_Templates := "SrcType := Real" } LE_Contact(in1 := "AI SCALING DB".PV."PRESSURE TRANSMITTER 504", in2 := "INTERLOCK DB"."EDI SET PARAMETER"."PT-504 HIGH")
      { S7_Templates := "time_type := Time" } "IEC_Timer_0_DB_107".TON(pt := T#3S, et =>)
      Move(in := 0, out1 => "INTERLOCK DB"."EDI PARAMETER BUFF"."PT-504 HIGH")
   END_RUNG
   RUNG wire#powerrail
      { S7_Templates := "SrcType := Int" } EQ_Contact(in1 := "MODE SELECTION DB".EDI."MODE BUFF", in2 := 1)
      { S7_Templates := "SrcType := Int" } EQ_Contact(in1 := "MODE SELECTION DB".EDI."PROCESS BUFF", in2 := 2)
      I_Contact( "EDI DB"."EDI FEED PUMP 401ABC" )
      wire#w4
      Move(in := 0, out1 => "INTERLOCK DB"."EDI PARAMETER BUFF"."PT-504 HIGH")
   END_RUNG
   RUNG wire#powerrail
      { S7_Templates := "SrcType := Int" } NE_Contact(in1 := "MODE SELECTION DB".EDI."PROCESS BUFF", in2 := 2)
   END_RUNG wire#w4
   // the same network as SCL:
   "IEC_Timer_0_DB_172".TON(IN := ("MODE SELECTION DB".EDI."MODE BUFF" = 1) AND ("MODE SELECTION DB".EDI."PROCESS BUFF" = 2) AND "EDI DB"."EDI FEED PUMP 401ABC",
                           PT := T#20S);
   "TIMING_SECS_DB_13"("SET TIME" := "INTERLOCK DB"."EDI SET TIMER"."PT-504 HIGH TIMER SET",   // "TIMING_SECS"
                       RESET := ("MODE SELECTION DB".EDI."PROCESS BUFF" = 0) OR ("INTERLOCK DB"."EDI PARAMETER BUFF"."PT-504 HIGH" <> 2),
                       INPUT := "IEC_Timer_0_DB_172".Q AND ("INTERLOCK DB"."EDI PARAMETER BUFF"."PT-504 HIGH" = 2) AND "PUMP SELECTION"."EDI-501",
                       "PRESENT VALUE OF TIME" => "INTERLOCK DB"."EDI PV TIMER"."PT-504 HIGH TIMER PV");
   #_w1 := "MODE SELECTION DB".EDI."MODE BUFF" = 1;
   "IEC_Timer_0_DB_190".TON(IN := #_w1 AND ("MODE SELECTION DB".EDI."PROCESS BUFF" = 2) AND "EDI DB"."EDI FEED PUMP 401ABC",
                           PT := T#15S);
   "IEC_Timer_0_DB_106".TON(IN := "IEC_Timer_0_DB_190".Q AND ("AI SCALING DB".PV."PRESSURE TRANSMITTER 504" > "INTERLOCK DB"."EDI SET PARAMETER"."PT-504 HIGH"),
                           PT := T#10S);
   IF "IEC_Timer_0_DB_106".Q THEN "INTERLOCK DB"."EDI PARAMETER BUFF"."PT-504 HIGH" := 2; END_IF;
   "IEC_Timer_0_DB_107".TON(IN := #_w1 AND ("AI SCALING DB".PV."PRESSURE TRANSMITTER 504" <= "INTERLOCK DB"."EDI SET PARAMETER"."PT-504 HIGH"),
                           PT := T#3S);
   IF "IEC_Timer_0_DB_107".Q THEN "INTERLOCK DB"."EDI PARAMETER BUFF"."PT-504 HIGH" := 0; END_IF;
   IF (("MODE SELECTION DB".EDI."MODE BUFF" = 1) AND ("MODE SELECTION DB".EDI."PROCESS BUFF" = 2) AND NOT "EDI DB"."EDI FEED PUMP 401ABC") OR ("MODE SELECTION DB".EDI."PROCESS BUFF" <> 2) THEN
       "INTERLOCK DB"."EDI PARAMETER BUFF"."PT-504 HIGH" := 0;
   END_IF;
END_REGION

REGION Network 37: PT505 HIGH
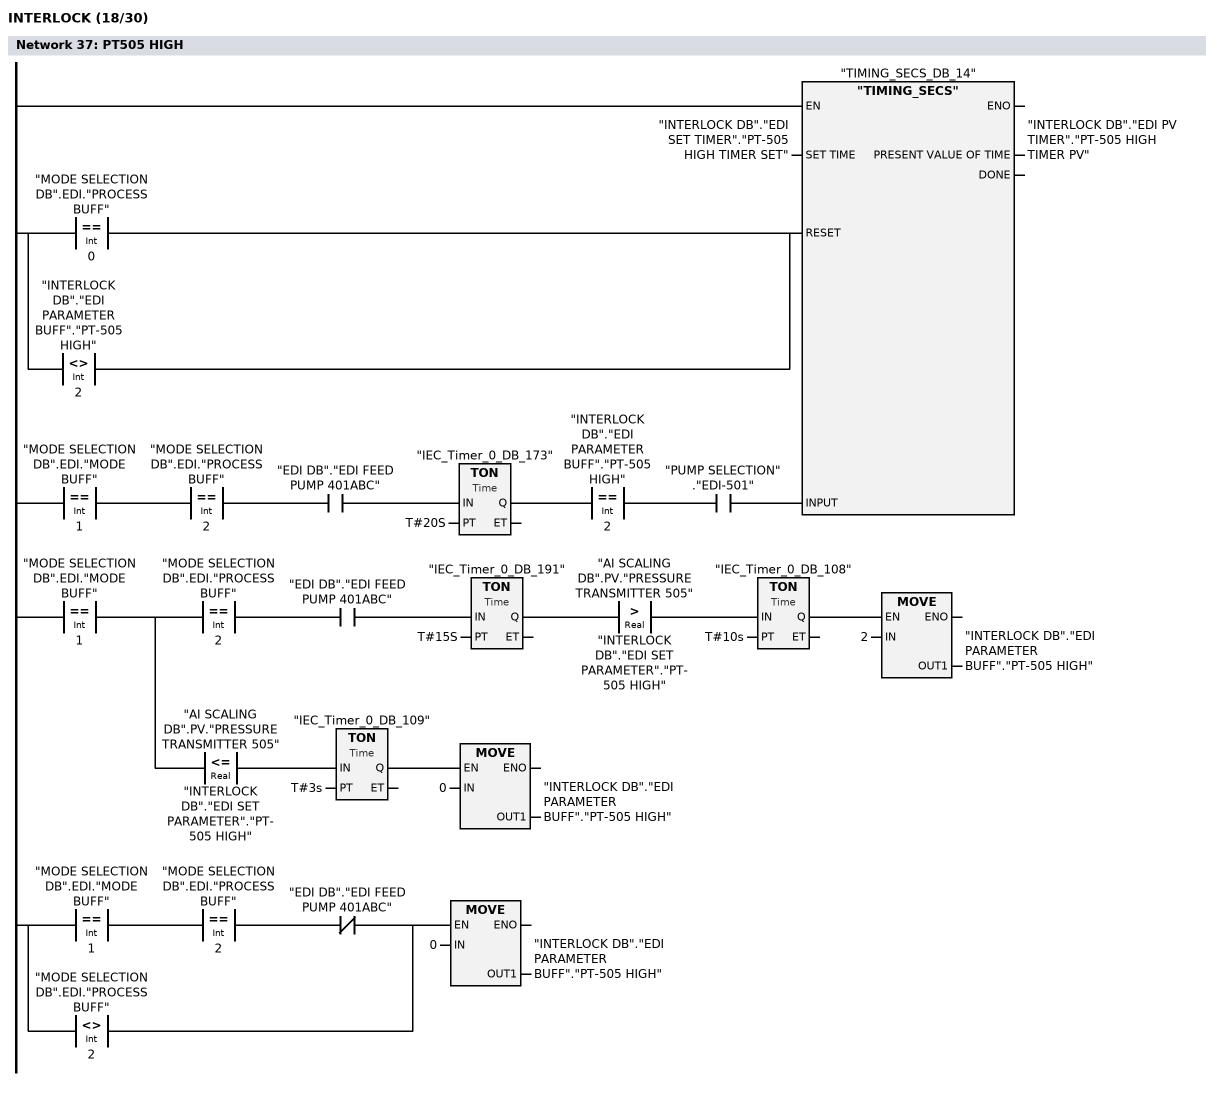
   RUNG wire#powerrail
      "TIMING_SECS_DB_14"(RESET := wire#w1, INPUT := wire#w2, "SET TIME" := "INTERLOCK DB"."EDI SET TIMER"."PT-505 HIGH TIMER SET", "PRESENT VALUE OF TIME" => "INTERLOCK DB"."EDI PV TIMER"."PT-505 HIGH TIMER PV", DONE =>)
   END_RUNG
   RUNG wire#powerrail
      { S7_Templates := "SrcType := Int" } EQ_Contact(in1 := "MODE SELECTION DB".EDI."PROCESS BUFF", in2 := 0)
   END_RUNG wire#w1
   RUNG wire#powerrail
      { S7_Templates := "SrcType := Int" } NE_Contact(in1 := "INTERLOCK DB"."EDI PARAMETER BUFF"."PT-505 HIGH", in2 := 2)
   END_RUNG wire#w1
   RUNG wire#powerrail
      { S7_Templates := "SrcType := Int" } EQ_Contact(in1 := "MODE SELECTION DB".EDI."MODE BUFF", in2 := 1)
      { S7_Templates := "SrcType := Int" } EQ_Contact(in1 := "MODE SELECTION DB".EDI."PROCESS BUFF", in2 := 2)
      Contact( "EDI DB"."EDI FEED PUMP 401ABC" )
      { S7_Templates := "time_type := Time" } "IEC_Timer_0_DB_173".TON(pt := T#20S, et =>)
      { S7_Templates := "SrcType := Int" } EQ_Contact(in1 := "INTERLOCK DB"."EDI PARAMETER BUFF"."PT-505 HIGH", in2 := 2)
      Contact( "PUMP SELECTION"."EDI-501" )
   END_RUNG wire#w2
   RUNG wire#powerrail
      { S7_Templates := "SrcType := Int" } EQ_Contact(in1 := "MODE SELECTION DB".EDI."MODE BUFF", in2 := 1)
      wire#w3
      { S7_Templates := "SrcType := Int" } EQ_Contact(in1 := "MODE SELECTION DB".EDI."PROCESS BUFF", in2 := 2)
      Contact( "EDI DB"."EDI FEED PUMP 401ABC" )
      { S7_Templates := "time_type := Time" } "IEC_Timer_0_DB_191".TON(pt := T#15S, et =>)
      { S7_Templates := "SrcType := Real" } GT_Contact(in1 := "AI SCALING DB".PV."PRESSURE TRANSMITTER 505", in2 := "INTERLOCK DB"."EDI SET PARAMETER"."PT-505 HIGH")
      { S7_Templates := "time_type := Time" } "IEC_Timer_0_DB_108".TON(pt := T#10s, et =>)
      Move(in := 2, out1 => "INTERLOCK DB"."EDI PARAMETER BUFF"."PT-505 HIGH")
   END_RUNG
   RUNG wire#w3
      { S7_Templates := "SrcType := Real" } LE_Contact(in1 := "AI SCALING DB".PV."PRESSURE TRANSMITTER 505", in2 := "INTERLOCK DB"."EDI SET PARAMETER"."PT-505 HIGH")
      { S7_Templates := "time_type := Time" } "IEC_Timer_0_DB_109".TON(pt := T#3s, et =>)
      Move(in := 0, out1 => "INTERLOCK DB"."EDI PARAMETER BUFF"."PT-505 HIGH")
   END_RUNG
   RUNG wire#powerrail
      { S7_Templates := "SrcType := Int" } EQ_Contact(in1 := "MODE SELECTION DB".EDI."MODE BUFF", in2 := 1)
      { S7_Templates := "SrcType := Int" } EQ_Contact(in1 := "MODE SELECTION DB".EDI."PROCESS BUFF", in2 := 2)
      I_Contact( "EDI DB"."EDI FEED PUMP 401ABC" )
      wire#w4
      Move(in := 0, out1 => "INTERLOCK DB"."EDI PARAMETER BUFF"."PT-505 HIGH")
   END_RUNG
   RUNG wire#powerrail
      { S7_Templates := "SrcType := Int" } NE_Contact(in1 := "MODE SELECTION DB".EDI."PROCESS BUFF", in2 := 2)
   END_RUNG wire#w4
   // the same network as SCL:
   "IEC_Timer_0_DB_173".TON(IN := ("MODE SELECTION DB".EDI."MODE BUFF" = 1) AND ("MODE SELECTION DB".EDI."PROCESS BUFF" = 2) AND "EDI DB"."EDI FEED PUMP 401ABC",
                           PT := T#20S);
   "TIMING_SECS_DB_14"("SET TIME" := "INTERLOCK DB"."EDI SET TIMER"."PT-505 HIGH TIMER SET",   // "TIMING_SECS"
                       RESET := ("MODE SELECTION DB".EDI."PROCESS BUFF" = 0) OR ("INTERLOCK DB"."EDI PARAMETER BUFF"."PT-505 HIGH" <> 2),
                       INPUT := "IEC_Timer_0_DB_173".Q AND ("INTERLOCK DB"."EDI PARAMETER BUFF"."PT-505 HIGH" = 2) AND "PUMP SELECTION"."EDI-501",
                       "PRESENT VALUE OF TIME" => "INTERLOCK DB"."EDI PV TIMER"."PT-505 HIGH TIMER PV");
   #_w1 := "MODE SELECTION DB".EDI."MODE BUFF" = 1;
   "IEC_Timer_0_DB_191".TON(IN := #_w1 AND ("MODE SELECTION DB".EDI."PROCESS BUFF" = 2) AND "EDI DB"."EDI FEED PUMP 401ABC",
                           PT := T#15S);
   "IEC_Timer_0_DB_108".TON(IN := "IEC_Timer_0_DB_191".Q AND ("AI SCALING DB".PV."PRESSURE TRANSMITTER 505" > "INTERLOCK DB"."EDI SET PARAMETER"."PT-505 HIGH"),
                           PT := T#10s);
   IF "IEC_Timer_0_DB_108".Q THEN "INTERLOCK DB"."EDI PARAMETER BUFF"."PT-505 HIGH" := 2; END_IF;
   "IEC_Timer_0_DB_109".TON(IN := #_w1 AND ("AI SCALING DB".PV."PRESSURE TRANSMITTER 505" <= "INTERLOCK DB"."EDI SET PARAMETER"."PT-505 HIGH"),
                           PT := T#3s);
   IF "IEC_Timer_0_DB_109".Q THEN "INTERLOCK DB"."EDI PARAMETER BUFF"."PT-505 HIGH" := 0; END_IF;
   IF (("MODE SELECTION DB".EDI."MODE BUFF" = 1) AND ("MODE SELECTION DB".EDI."PROCESS BUFF" = 2) AND NOT "EDI DB"."EDI FEED PUMP 401ABC") OR ("MODE SELECTION DB".EDI."PROCESS BUFF" <> 2) THEN
       "INTERLOCK DB"."EDI PARAMETER BUFF"."PT-505 HIGH" := 0;
   END_IF;
END_REGION

REGION Network 38: PT506 HIGH
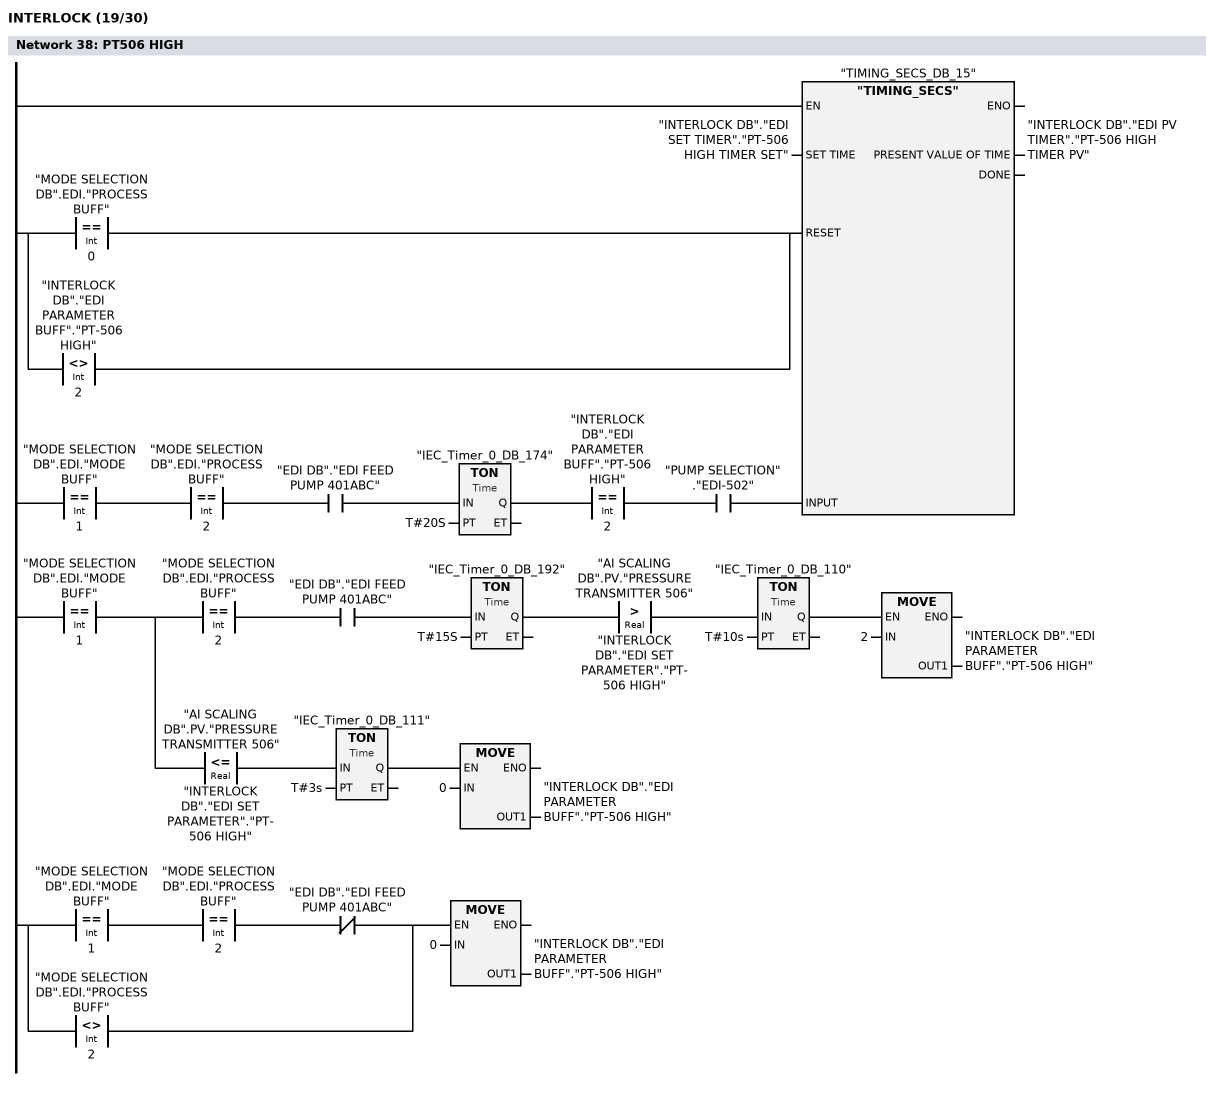
   RUNG wire#powerrail
      "TIMING_SECS_DB_15"(RESET := wire#w1, INPUT := wire#w2, "SET TIME" := "INTERLOCK DB"."EDI SET TIMER"."PT-506 HIGH TIMER SET", "PRESENT VALUE OF TIME" => "INTERLOCK DB"."EDI PV TIMER"."PT-506 HIGH TIMER PV", DONE =>)
   END_RUNG
   RUNG wire#powerrail
      { S7_Templates := "SrcType := Int" } EQ_Contact(in1 := "MODE SELECTION DB".EDI."PROCESS BUFF", in2 := 0)
   END_RUNG wire#w1
   RUNG wire#powerrail
      { S7_Templates := "SrcType := Int" } NE_Contact(in1 := "INTERLOCK DB"."EDI PARAMETER BUFF"."PT-506 HIGH", in2 := 2)
   END_RUNG wire#w1
   RUNG wire#powerrail
      { S7_Templates := "SrcType := Int" } EQ_Contact(in1 := "MODE SELECTION DB".EDI."MODE BUFF", in2 := 1)
      { S7_Templates := "SrcType := Int" } EQ_Contact(in1 := "MODE SELECTION DB".EDI."PROCESS BUFF", in2 := 2)
      Contact( "EDI DB"."EDI FEED PUMP 401ABC" )
      { S7_Templates := "time_type := Time" } "IEC_Timer_0_DB_174".TON(pt := T#20S, et =>)
      { S7_Templates := "SrcType := Int" } EQ_Contact(in1 := "INTERLOCK DB"."EDI PARAMETER BUFF"."PT-506 HIGH", in2 := 2)
      Contact( "PUMP SELECTION"."EDI-502" )
   END_RUNG wire#w2
   RUNG wire#powerrail
      { S7_Templates := "SrcType := Int" } EQ_Contact(in1 := "MODE SELECTION DB".EDI."MODE BUFF", in2 := 1)
      wire#w3
      { S7_Templates := "SrcType := Int" } EQ_Contact(in1 := "MODE SELECTION DB".EDI."PROCESS BUFF", in2 := 2)
      Contact( "EDI DB"."EDI FEED PUMP 401ABC" )
      { S7_Templates := "time_type := Time" } "IEC_Timer_0_DB_192".TON(pt := T#15S, et =>)
      { S7_Templates := "SrcType := Real" } GT_Contact(in1 := "AI SCALING DB".PV."PRESSURE TRANSMITTER 506", in2 := "INTERLOCK DB"."EDI SET PARAMETER"."PT-506 HIGH")
      { S7_Templates := "time_type := Time" } "IEC_Timer_0_DB_110".TON(pt := T#10s, et =>)
      Move(in := 2, out1 => "INTERLOCK DB"."EDI PARAMETER BUFF"."PT-506 HIGH")
   END_RUNG
   RUNG wire#w3
      { S7_Templates := "SrcType := Real" } LE_Contact(in1 := "AI SCALING DB".PV."PRESSURE TRANSMITTER 506", in2 := "INTERLOCK DB"."EDI SET PARAMETER"."PT-506 HIGH")
      { S7_Templates := "time_type := Time" } "IEC_Timer_0_DB_111".TON(pt := T#3s, et =>)
      Move(in := 0, out1 => "INTERLOCK DB"."EDI PARAMETER BUFF"."PT-506 HIGH")
   END_RUNG
   RUNG wire#powerrail
      { S7_Templates := "SrcType := Int" } EQ_Contact(in1 := "MODE SELECTION DB".EDI."MODE BUFF", in2 := 1)
      { S7_Templates := "SrcType := Int" } EQ_Contact(in1 := "MODE SELECTION DB".EDI."PROCESS BUFF", in2 := 2)
      I_Contact( "EDI DB"."EDI FEED PUMP 401ABC" )
      wire#w4
      Move(in := 0, out1 => "INTERLOCK DB"."EDI PARAMETER BUFF"."PT-506 HIGH")
   END_RUNG
   RUNG wire#powerrail
      { S7_Templates := "SrcType := Int" } NE_Contact(in1 := "MODE SELECTION DB".EDI."PROCESS BUFF", in2 := 2)
   END_RUNG wire#w4
   // the same network as SCL:
   "IEC_Timer_0_DB_174".TON(IN := ("MODE SELECTION DB".EDI."MODE BUFF" = 1) AND ("MODE SELECTION DB".EDI."PROCESS BUFF" = 2) AND "EDI DB"."EDI FEED PUMP 401ABC",
                           PT := T#20S);
   "TIMING_SECS_DB_15"("SET TIME" := "INTERLOCK DB"."EDI SET TIMER"."PT-506 HIGH TIMER SET",   // "TIMING_SECS"
                       RESET := ("MODE SELECTION DB".EDI."PROCESS BUFF" = 0) OR ("INTERLOCK DB"."EDI PARAMETER BUFF"."PT-506 HIGH" <> 2),
                       INPUT := "IEC_Timer_0_DB_174".Q AND ("INTERLOCK DB"."EDI PARAMETER BUFF"."PT-506 HIGH" = 2) AND "PUMP SELECTION"."EDI-502",
                       "PRESENT VALUE OF TIME" => "INTERLOCK DB"."EDI PV TIMER"."PT-506 HIGH TIMER PV");
   #_w1 := "MODE SELECTION DB".EDI."MODE BUFF" = 1;
   "IEC_Timer_0_DB_192".TON(IN := #_w1 AND ("MODE SELECTION DB".EDI."PROCESS BUFF" = 2) AND "EDI DB"."EDI FEED PUMP 401ABC",
                           PT := T#15S);
   "IEC_Timer_0_DB_110".TON(IN := "IEC_Timer_0_DB_192".Q AND ("AI SCALING DB".PV."PRESSURE TRANSMITTER 506" > "INTERLOCK DB"."EDI SET PARAMETER"."PT-506 HIGH"),
                           PT := T#10s);
   IF "IEC_Timer_0_DB_110".Q THEN "INTERLOCK DB"."EDI PARAMETER BUFF"."PT-506 HIGH" := 2; END_IF;
   "IEC_Timer_0_DB_111".TON(IN := #_w1 AND ("AI SCALING DB".PV."PRESSURE TRANSMITTER 506" <= "INTERLOCK DB"."EDI SET PARAMETER"."PT-506 HIGH"),
                           PT := T#3s);
   IF "IEC_Timer_0_DB_111".Q THEN "INTERLOCK DB"."EDI PARAMETER BUFF"."PT-506 HIGH" := 0; END_IF;
   IF (("MODE SELECTION DB".EDI."MODE BUFF" = 1) AND ("MODE SELECTION DB".EDI."PROCESS BUFF" = 2) AND NOT "EDI DB"."EDI FEED PUMP 401ABC") OR ("MODE SELECTION DB".EDI."PROCESS BUFF" <> 2) THEN
       "INTERLOCK DB"."EDI PARAMETER BUFF"."PT-506 HIGH" := 0;
   END_IF;
END_REGION

REGION Network 39: FIT-501 LOW
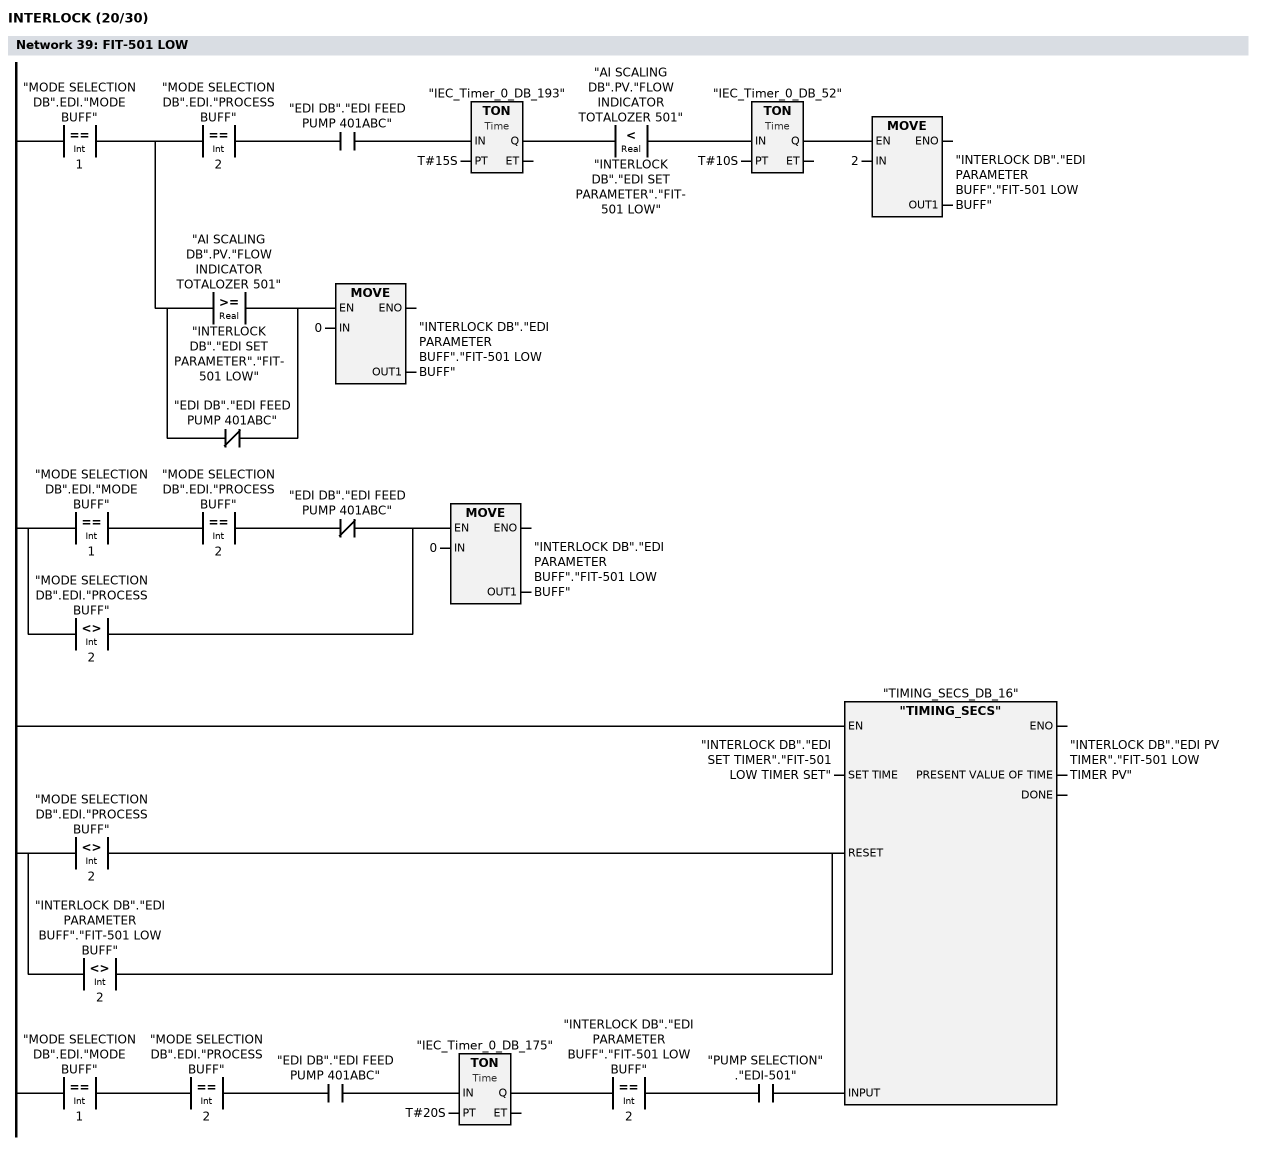
   RUNG wire#powerrail
      { S7_Templates := "SrcType := Int" } EQ_Contact(in1 := "MODE SELECTION DB".EDI."MODE BUFF", in2 := 1)
      wire#w1
      { S7_Templates := "SrcType := Int" } EQ_Contact(in1 := "MODE SELECTION DB".EDI."PROCESS BUFF", in2 := 2)
      Contact( "EDI DB"."EDI FEED PUMP 401ABC" )
      { S7_Templates := "time_type := Time" } "IEC_Timer_0_DB_193".TON(pt := T#15S, et =>)
      { S7_Templates := "SrcType := Real" } LT_Contact(in1 := "AI SCALING DB".PV."FLOW INDICATOR TOTALOZER 501", in2 := "INTERLOCK DB"."EDI SET PARAMETER"."FIT-501 LOW")
      { S7_Templates := "time_type := Time" } "IEC_Timer_0_DB_52".TON(pt := T#10S, et =>)
      Move(in := 2, out1 => "INTERLOCK DB"."EDI PARAMETER BUFF"."FIT-501 LOW BUFF")
   END_RUNG
   RUNG wire#w1
      { S7_Templates := "SrcType := Real" } GE_Contact(in1 := "AI SCALING DB".PV."FLOW INDICATOR TOTALOZER 501", in2 := "INTERLOCK DB"."EDI SET PARAMETER"."FIT-501 LOW")
      wire#w2
      Move(in := 0, out1 => "INTERLOCK DB"."EDI PARAMETER BUFF"."FIT-501 LOW BUFF")
   END_RUNG
   RUNG wire#w1
      I_Contact( "EDI DB"."EDI FEED PUMP 401ABC" )
   END_RUNG wire#w2
   RUNG wire#powerrail
      { S7_Templates := "SrcType := Int" } EQ_Contact(in1 := "MODE SELECTION DB".EDI."MODE BUFF", in2 := 1)
      { S7_Templates := "SrcType := Int" } EQ_Contact(in1 := "MODE SELECTION DB".EDI."PROCESS BUFF", in2 := 2)
      I_Contact( "EDI DB"."EDI FEED PUMP 401ABC" )
      wire#w3
      Move(in := 0, out1 => "INTERLOCK DB"."EDI PARAMETER BUFF"."FIT-501 LOW BUFF")
   END_RUNG
   RUNG wire#powerrail
      { S7_Templates := "SrcType := Int" } NE_Contact(in1 := "MODE SELECTION DB".EDI."PROCESS BUFF", in2 := 2)
   END_RUNG wire#w3
   RUNG wire#powerrail
      "TIMING_SECS_DB_16"(RESET := wire#w4, INPUT := wire#w5, "SET TIME" := "INTERLOCK DB"."EDI SET TIMER"."FIT-501 LOW TIMER SET", "PRESENT VALUE OF TIME" => "INTERLOCK DB"."EDI PV TIMER"."FIT-501 LOW TIMER PV", DONE =>)
   END_RUNG
   RUNG wire#powerrail
      { S7_Templates := "SrcType := Int" } NE_Contact(in1 := "MODE SELECTION DB".EDI."PROCESS BUFF", in2 := 2)
   END_RUNG wire#w4
   RUNG wire#powerrail
      { S7_Templates := "SrcType := Int" } NE_Contact(in1 := "INTERLOCK DB"."EDI PARAMETER BUFF"."FIT-501 LOW BUFF", in2 := 2)
   END_RUNG wire#w4
   RUNG wire#powerrail
      { S7_Templates := "SrcType := Int" } EQ_Contact(in1 := "MODE SELECTION DB".EDI."MODE BUFF", in2 := 1)
      { S7_Templates := "SrcType := Int" } EQ_Contact(in1 := "MODE SELECTION DB".EDI."PROCESS BUFF", in2 := 2)
      Contact( "EDI DB"."EDI FEED PUMP 401ABC" )
      { S7_Templates := "time_type := Time" } "IEC_Timer_0_DB_175".TON(pt := T#20S, et =>)
      { S7_Templates := "SrcType := Int" } EQ_Contact(in1 := "INTERLOCK DB"."EDI PARAMETER BUFF"."FIT-501 LOW BUFF", in2 := 2)
      Contact( "PUMP SELECTION"."EDI-501" )
   END_RUNG wire#w5
   // the same network as SCL:
   #_w1 := "MODE SELECTION DB".EDI."MODE BUFF" = 1;
   "IEC_Timer_0_DB_193".TON(IN := #_w1 AND ("MODE SELECTION DB".EDI."PROCESS BUFF" = 2) AND "EDI DB"."EDI FEED PUMP 401ABC",
                           PT := T#15S);
   "IEC_Timer_0_DB_52".TON(IN := "IEC_Timer_0_DB_193".Q AND ("AI SCALING DB".PV."FLOW INDICATOR TOTALOZER 501" < "INTERLOCK DB"."EDI SET PARAMETER"."FIT-501 LOW"),
                           PT := T#10S);
   IF "IEC_Timer_0_DB_52".Q THEN "INTERLOCK DB"."EDI PARAMETER BUFF"."FIT-501 LOW BUFF" := 2; END_IF;
   IF #_w1 AND (("AI SCALING DB".PV."FLOW INDICATOR TOTALOZER 501" >= "INTERLOCK DB"."EDI SET PARAMETER"."FIT-501 LOW") OR NOT "EDI DB"."EDI FEED PUMP 401ABC") THEN
       "INTERLOCK DB"."EDI PARAMETER BUFF"."FIT-501 LOW BUFF" := 0;
   END_IF;
   IF (("MODE SELECTION DB".EDI."MODE BUFF" = 1) AND ("MODE SELECTION DB".EDI."PROCESS BUFF" = 2) AND NOT "EDI DB"."EDI FEED PUMP 401ABC") OR ("MODE SELECTION DB".EDI."PROCESS BUFF" <> 2) THEN
       "INTERLOCK DB"."EDI PARAMETER BUFF"."FIT-501 LOW BUFF" := 0;
   END_IF;
   "IEC_Timer_0_DB_175".TON(IN := ("MODE SELECTION DB".EDI."MODE BUFF" = 1) AND ("MODE SELECTION DB".EDI."PROCESS BUFF" = 2) AND "EDI DB"."EDI FEED PUMP 401ABC",
                           PT := T#20S);
   "TIMING_SECS_DB_16"("SET TIME" := "INTERLOCK DB"."EDI SET TIMER"."FIT-501 LOW TIMER SET",   // "TIMING_SECS"
                       RESET := ("MODE SELECTION DB".EDI."PROCESS BUFF" <> 2) OR ("INTERLOCK DB"."EDI PARAMETER BUFF"."FIT-501 LOW BUFF" <> 2),
                       INPUT := "IEC_Timer_0_DB_175".Q AND ("INTERLOCK DB"."EDI PARAMETER BUFF"."FIT-501 LOW BUFF" = 2) AND "PUMP SELECTION"."EDI-501",
                       "PRESENT VALUE OF TIME" => "INTERLOCK DB"."EDI PV TIMER"."FIT-501 LOW TIMER PV");
END_REGION

REGION Network 40: FIT-502 LOW
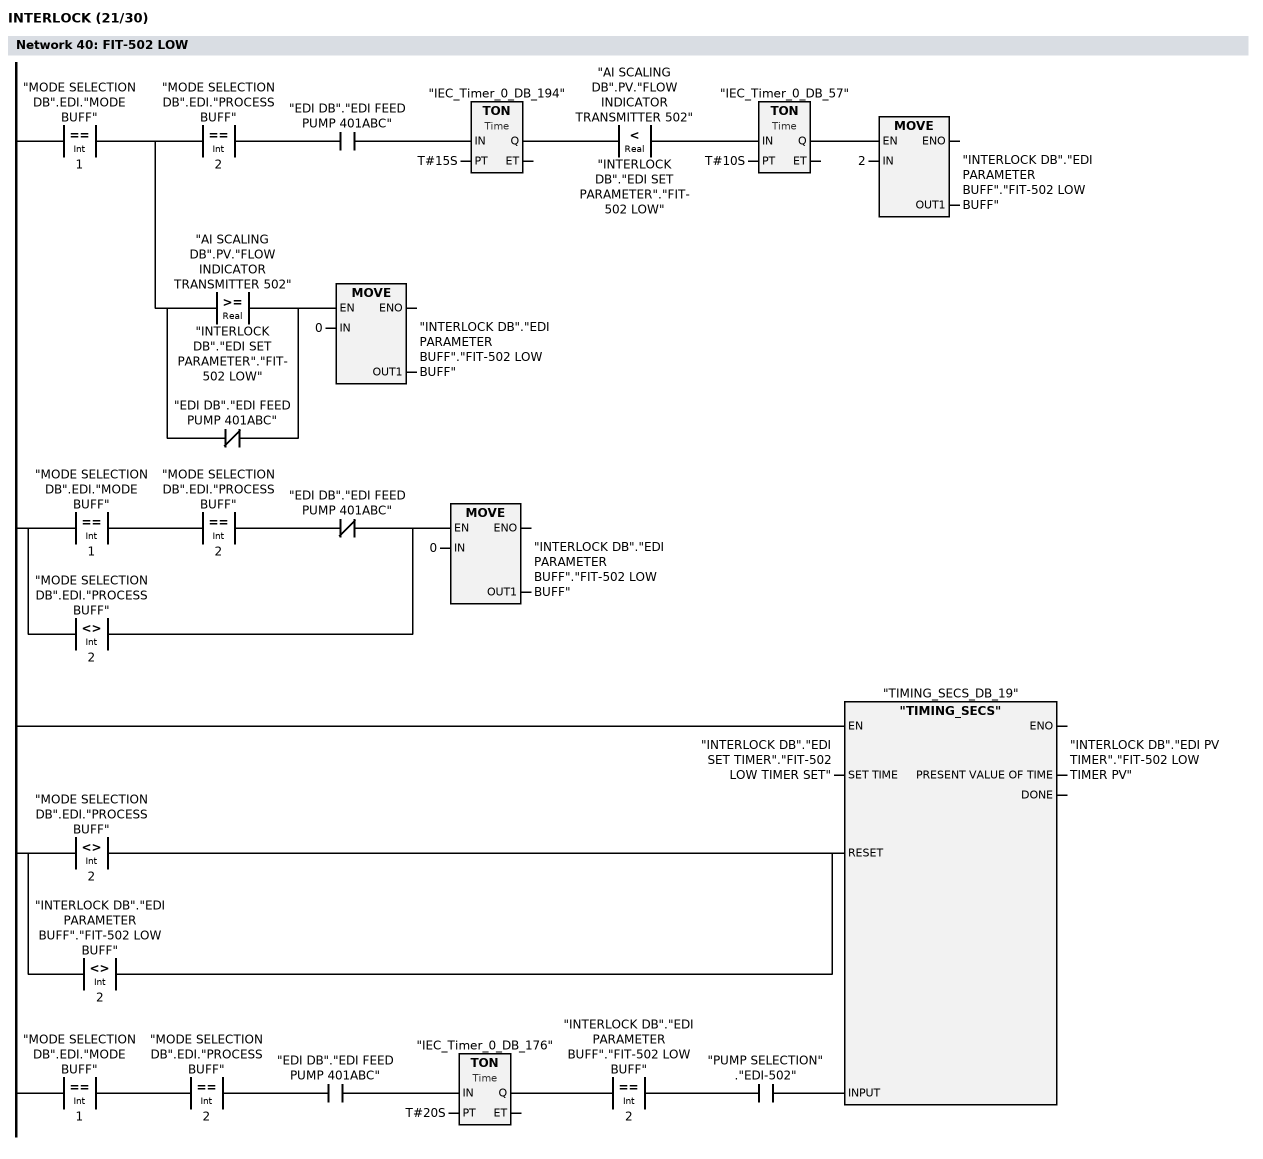
   RUNG wire#powerrail
      { S7_Templates := "SrcType := Int" } EQ_Contact(in1 := "MODE SELECTION DB".EDI."MODE BUFF", in2 := 1)
      wire#w1
      { S7_Templates := "SrcType := Int" } EQ_Contact(in1 := "MODE SELECTION DB".EDI."PROCESS BUFF", in2 := 2)
      Contact( "EDI DB"."EDI FEED PUMP 401ABC" )
      { S7_Templates := "time_type := Time" } "IEC_Timer_0_DB_194".TON(pt := T#15S, et =>)
      { S7_Templates := "SrcType := Real" } LT_Contact(in1 := "AI SCALING DB".PV."FLOW INDICATOR TRANSMITTER 502", in2 := "INTERLOCK DB"."EDI SET PARAMETER"."FIT-502 LOW")
      { S7_Templates := "time_type := Time" } "IEC_Timer_0_DB_57".TON(pt := T#10S, et =>)
      Move(in := 2, out1 => "INTERLOCK DB"."EDI PARAMETER BUFF"."FIT-502 LOW  BUFF")
   END_RUNG
   RUNG wire#w1
      { S7_Templates := "SrcType := Real" } GE_Contact(in1 := "AI SCALING DB".PV."FLOW INDICATOR TRANSMITTER 502", in2 := "INTERLOCK DB"."EDI SET PARAMETER"."FIT-502 LOW")
      wire#w2
      Move(in := 0, out1 => "INTERLOCK DB"."EDI PARAMETER BUFF"."FIT-502 LOW  BUFF")
   END_RUNG
   RUNG wire#w1
      I_Contact( "EDI DB"."EDI FEED PUMP 401ABC" )
   END_RUNG wire#w2
   RUNG wire#powerrail
      { S7_Templates := "SrcType := Int" } EQ_Contact(in1 := "MODE SELECTION DB".EDI."MODE BUFF", in2 := 1)
      { S7_Templates := "SrcType := Int" } EQ_Contact(in1 := "MODE SELECTION DB".EDI."PROCESS BUFF", in2 := 2)
      I_Contact( "EDI DB"."EDI FEED PUMP 401ABC" )
      wire#w3
      Move(in := 0, out1 => "INTERLOCK DB"."EDI PARAMETER BUFF"."FIT-502 LOW  BUFF")
   END_RUNG
   RUNG wire#powerrail
      { S7_Templates := "SrcType := Int" } NE_Contact(in1 := "MODE SELECTION DB".EDI."PROCESS BUFF", in2 := 2)
   END_RUNG wire#w3
   RUNG wire#powerrail
      "TIMING_SECS_DB_19"(RESET := wire#w4, INPUT := wire#w5, "SET TIME" := "INTERLOCK DB"."EDI SET TIMER"."FIT-502 LOW TIMER SET", "PRESENT VALUE OF TIME" => "INTERLOCK DB"."EDI PV TIMER"."FIT-502 LOW TIMER PV", DONE =>)
   END_RUNG
   RUNG wire#powerrail
      { S7_Templates := "SrcType := Int" } NE_Contact(in1 := "MODE SELECTION DB".EDI."PROCESS BUFF", in2 := 2)
   END_RUNG wire#w4
   RUNG wire#powerrail
      { S7_Templates := "SrcType := Int" } NE_Contact(in1 := "INTERLOCK DB"."EDI PARAMETER BUFF"."FIT-502 LOW  BUFF", in2 := 2)
   END_RUNG wire#w4
   RUNG wire#powerrail
      { S7_Templates := "SrcType := Int" } EQ_Contact(in1 := "MODE SELECTION DB".EDI."MODE BUFF", in2 := 1)
      { S7_Templates := "SrcType := Int" } EQ_Contact(in1 := "MODE SELECTION DB".EDI."PROCESS BUFF", in2 := 2)
      Contact( "EDI DB"."EDI FEED PUMP 401ABC" )
      { S7_Templates := "time_type := Time" } "IEC_Timer_0_DB_176".TON(pt := T#20S, et =>)
      { S7_Templates := "SrcType := Int" } EQ_Contact(in1 := "INTERLOCK DB"."EDI PARAMETER BUFF"."FIT-502 LOW  BUFF", in2 := 2)
      Contact( "PUMP SELECTION"."EDI-502" )
   END_RUNG wire#w5
   // the same network as SCL:
   #_w1 := "MODE SELECTION DB".EDI."MODE BUFF" = 1;
   "IEC_Timer_0_DB_194".TON(IN := #_w1 AND ("MODE SELECTION DB".EDI."PROCESS BUFF" = 2) AND "EDI DB"."EDI FEED PUMP 401ABC",
                           PT := T#15S);
   "IEC_Timer_0_DB_57".TON(IN := "IEC_Timer_0_DB_194".Q AND ("AI SCALING DB".PV."FLOW INDICATOR TRANSMITTER 502" < "INTERLOCK DB"."EDI SET PARAMETER"."FIT-502 LOW"),
                           PT := T#10S);
   IF "IEC_Timer_0_DB_57".Q THEN "INTERLOCK DB"."EDI PARAMETER BUFF"."FIT-502 LOW  BUFF" := 2; END_IF;
   IF #_w1 AND (("AI SCALING DB".PV."FLOW INDICATOR TRANSMITTER 502" >= "INTERLOCK DB"."EDI SET PARAMETER"."FIT-502 LOW") OR NOT "EDI DB"."EDI FEED PUMP 401ABC") THEN
       "INTERLOCK DB"."EDI PARAMETER BUFF"."FIT-502 LOW  BUFF" := 0;
   END_IF;
   IF (("MODE SELECTION DB".EDI."MODE BUFF" = 1) AND ("MODE SELECTION DB".EDI."PROCESS BUFF" = 2) AND NOT "EDI DB"."EDI FEED PUMP 401ABC") OR ("MODE SELECTION DB".EDI."PROCESS BUFF" <> 2) THEN
       "INTERLOCK DB"."EDI PARAMETER BUFF"."FIT-502 LOW  BUFF" := 0;
   END_IF;
   "IEC_Timer_0_DB_176".TON(IN := ("MODE SELECTION DB".EDI."MODE BUFF" = 1) AND ("MODE SELECTION DB".EDI."PROCESS BUFF" = 2) AND "EDI DB"."EDI FEED PUMP 401ABC",
                           PT := T#20S);
   "TIMING_SECS_DB_19"("SET TIME" := "INTERLOCK DB"."EDI SET TIMER"."FIT-502 LOW TIMER SET",   // "TIMING_SECS"
                       RESET := ("MODE SELECTION DB".EDI."PROCESS BUFF" <> 2) OR ("INTERLOCK DB"."EDI PARAMETER BUFF"."FIT-502 LOW  BUFF" <> 2),
                       INPUT := "IEC_Timer_0_DB_176".Q AND ("INTERLOCK DB"."EDI PARAMETER BUFF"."FIT-502 LOW  BUFF" = 2) AND "PUMP SELECTION"."EDI-502",
                       "PRESENT VALUE OF TIME" => "INTERLOCK DB"."EDI PV TIMER"."FIT-502 LOW TIMER PV");
END_REGION

